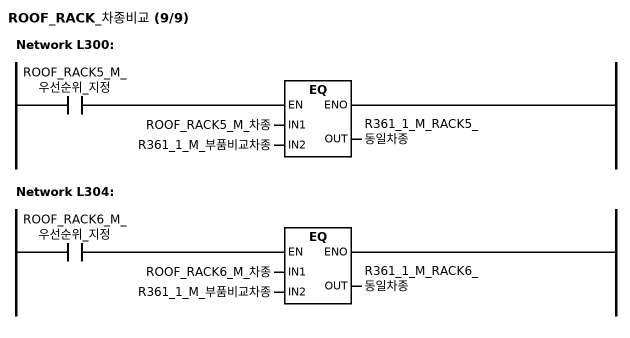
(* [picture p96: ROOF_RACK_차종비교 rungs L300-L304] *)
(* Rung L300 *)
IF ROOF_RACK5_M_우선순위_지정 THEN R361_1_M_RACK5_동일차종 := ROOF_RACK5_M_차종 = R361_1_M_부품비교차종; END_IF;
(* Rung L304 *)
IF ROOF_RACK6_M_우선순위_지정 THEN R361_1_M_RACK6_동일차종 := ROOF_RACK6_M_차종 = R361_1_M_부품비교차종; END_IF;
END_PROGRAM

PROGRAM ROOF_RACK_로보트 (* task: 스캔 프로그램 *)
VAR_EXTERNAL RETAIN
    ALWAYS_OFF : BOOL; (* AT %MW3.0 *) (* 항시 OFF *)
    ALWAYS_ON : BOOL; (* AT %MW3.1 *) (* 항시 ON *)
    MCP_M_부저_정지 : BOOL; (* AT %MW350.5 *) (* MCP 부저정지 *)
    MCP_M_비상정지 : BOOL; (* AT %MW350.7 *) (* MCP 비상정지 이상 *)
    R361_1_M_RACK3_동일차종 : BOOL; (* AT %MW1565.2 *)
    R361_1_M_RACK3_프로그램_OK : BOOL; (* AT %MW1563.2 *)
    R361_1_M_RACK4_동일차종 : BOOL; (* AT %MW1565.3 *)
    R361_1_M_RACK4_프로그램_OK : BOOL; (* AT %MW1563.3 *)
    R361_1_M_RACK5_동일차종 : BOOL; (* AT %MW1565.4 *)
    R361_1_M_RACK5_프로그램_OK : BOOL; (* AT %MW1563.4 *)
    R361_1_M_RACK6_동일차종 : BOOL; (* AT %MW1565.5 *)
    R361_1_M_RACK6_프로그램_OK : BOOL; (* AT %MW1563.5 *)
    R361_1_M_기동_랙번호 : WORD; (* AT %MW1534 *)
    R361_1_M_차종1_AX : BOOL; (* AT %MW10001.0 *) (* R361 1 M 차종1 AX *)
    R361_1_M_차종6_썬루프 : BOOL; (* AT %MW10003.4 *) (* R361 1 M 차종6 썬루프 *)
    R361_1_M_차종6_일반루프 : BOOL; (* AT %MW10003.3 *) (* R361 1 M 차종6 일반루프 *)
    R361_1_M_차종_OPT1_R_RACK_무 : BOOL; (* AT %MW10005.3 *) (* R361 1 M 차종 OPT1 R RACK 무 *)
    R361_1_M_차종_OPT1_R_RACK_유 : BOOL; (* AT %MW10005.2 *) (* R361 1 M 차종 OPT1 R RACK 유 *)
    R361_1_M_차종_유 : BOOL; (* AT %MW1502.0 *)
    R361_2_M_RACK1_동일차종 : BOOL; (* AT %MW1565.0 *)
    R361_2_M_RACK1_프로그램_OK : BOOL; (* AT %MW1563.0 *)
    R361_2_M_RACK2_동일차종 : BOOL; (* AT %MW1565.1 *)
    R361_2_M_RACK2_프로그램_OK : BOOL; (* AT %MW1563.1 *)
    R361_2_M_기동_랙번호 : WORD; (* AT %MW1535 *)
    R361_2_M_차종1_AX : BOOL; (* AT %MW10021.0 *) (* R361 2 M 차종1 AX *)
    R361_2_M_차종6_썬루프 : BOOL; (* AT %MW10023.4 *) (* R361 2 M 차종6 썬루프 *)
    R361_2_M_차종6_일반루프 : BOOL; (* AT %MW10023.3 *) (* R361 2 M 차종6 일반루프 *)
    R361_2_M_차종_OPT1_R_RACK_유 : BOOL; (* AT %MW10025.2 *) (* R361 2 M 차종 OPT1 R RACK 유 *)
    R361_2_M_차종_유 : BOOL; (* AT %MW1502.2 *)
    ROOF_RACK1_M_PLT_이상 : BOOL; (* AT %MW1514.0 *)
    ROOF_RACK1_M_랙감지_유 : BOOL; (* AT %MW1501.0 *)
    ROOF_RACK1_M_막장감지_유 : BOOL; (* AT %MW1503.0 *)
    ROOF_RACK1_M_우선순위_지정 : BOOL; (* AT %MW1564.0 *)
    ROOF_RACK1_M_차종_무 : BOOL; (* AT %MW1540.1 *)
    ROOF_RACK1_M_카운트_리셋요구_SET : BOOL; (* AT %MW1566.0 *)
    ROOF_RACK2_M_PLT_이상 : BOOL; (* AT %MW1514.1 *)
    ROOF_RACK2_M_랙감지_유 : BOOL; (* AT %MW1501.2 *)
    ROOF_RACK2_M_막장감지_유 : BOOL; (* AT %MW1503.2 *)
    ROOF_RACK2_M_우선순위_지정 : BOOL; (* AT %MW1564.1 *)
    ROOF_RACK2_M_차종_무 : BOOL; (* AT %MW1540.3 *)
    ROOF_RACK2_M_카운트_리셋요구_SET : BOOL; (* AT %MW1566.1 *)
    ROOF_RACK3_M_PLT_이상 : BOOL; (* AT %MW1514.2 *)
    ROOF_RACK3_M_랙감지_유 : BOOL; (* AT %MW1501.4 *)
    ROOF_RACK3_M_막장감지_유 : BOOL; (* AT %MW1503.4 *)
    ROOF_RACK3_M_우선순위_지정 : BOOL; (* AT %MW1564.2 *)
    ROOF_RACK3_M_차종_무 : BOOL; (* AT %MW1540.5 *)
    ROOF_RACK3_M_카운트_리셋요구_SET : BOOL; (* AT %MW1566.2 *)
    ROOF_RACK4_M_PLT_이상 : BOOL; (* AT %MW1514.3 *)
    ROOF_RACK4_M_랙감지_유 : BOOL; (* AT %MW1501.6 *)
    ROOF_RACK4_M_막장감지_유 : BOOL; (* AT %MW1503.6 *)
    ROOF_RACK4_M_우선순위_지정 : BOOL; (* AT %MW1564.3 *)
    ROOF_RACK4_M_차종_무 : BOOL; (* AT %MW1540.7 *)
    ROOF_RACK4_M_카운트_리셋요구_SET : BOOL; (* AT %MW1566.3 *)
    ROOF_RACK5_M_PLT_이상 : BOOL; (* AT %MW1514.4 *)
    ROOF_RACK5_M_랙감지_유 : BOOL; (* AT %MW1501.8 *)
    ROOF_RACK5_M_막장감지_유 : BOOL; (* AT %MW1503.8 *)
    ROOF_RACK5_M_우선순위_지정 : BOOL; (* AT %MW1564.4 *)
    ROOF_RACK5_M_차종_무 : BOOL; (* AT %MW1540.9 *)
    ROOF_RACK5_M_카운트_리셋요구_SET : BOOL; (* AT %MW1566.4 *)
    ROOF_RACK6_M_PLT_이상 : BOOL; (* AT %MW1514.5 *)
    ROOF_RACK6_M_랙감지_유 : BOOL; (* AT %MW1501.10 *)
    ROOF_RACK6_M_막장감지_유 : BOOL; (* AT %MW1503.10 *)
    ROOF_RACK6_M_우선순위_지정 : BOOL; (* AT %MW1564.5 *)
    ROOF_RACK6_M_차종_무 : BOOL; (* AT %MW1540.11 *)
    ROOF_RACK6_M_카운트_리셋요구_SET : BOOL; (* AT %MW1566.5 *)
    ROOF_RACK_M_수동모드 : BOOL; (* AT %MW1500.3 *)
    ROOF_RACK_M_자동_START : BOOL; (* AT %MW1500.5 *)
    ROOF_RACK_M_자동_운전중 : BOOL; (* AT %MW1500.4 *)
    ROOF_RACK_M_작업완료_SET_PLS : BOOL; (* AT %MW1500.8 *)
    ROOF_RACK_M_작업완료_리셋_PLS : BOOL; (* AT %MW1500.9 *)
    ROOF_RACK_M_총괄_이상 : BOOL; (* AT %MW1509.0 *)
    S364_M_R361_2_로딩완료 : BOOL; (* AT %MW2001.2 *)
    S364_M_공정_제품감지_무 : BOOL; (* AT %MW2002.5 *) (* S364_M_공정_제품감지_무 *)
    S364_M_공정_제품감지_유 : BOOL; (* AT %MW2002.4 *) (* S364_M_공정_제품감지_유 *)
    S364_M_공정_차종_AX : BOOL; (* AT %MW2002.3 *) (* S364_M_공정_차종_AX *)
    S364_M_공정_차종_무 : BOOL; (* AT %MW2002.1 *) (* S364_M_공정_차종_무 *)
    S364_M_공정_차종_유 : BOOL; (* AT %MW2002.0 *) (* S364_M_공정_차종_유 *)
    S364_M_자동_START : BOOL; (* AT %MW2000.5 *) (* S364 자동운전중 *)
    S364_M_자동_운전중 : BOOL; (* AT %MW2000.4 *) (* S364 자동운전중 *)
    S364_M_작업_완료 : BOOL; (* AT %MW2001.0 *) (* S364_M_작업_완료 *)
    S364_M_총괄_이상 : BOOL; (* AT %MW2009.0 *) (* S364_M_총괄_이상 *)
    S365_M_R361_1_안착완료 : BOOL; (* AT %MW2501.1 *)
    S365_M_공정_제품감지_무 : BOOL; (* AT %MW2501.4 *) (* S365_M_공정_제품감지_무 *)
    S365_M_공정_제품감지_유 : BOOL; (* AT %MW2501.3 *) (* S365_M_공정_제품감지_유 *)
    S365_M_공정_차종_무 : BOOL; (* AT %MW2502.1 *) (* S365_M_공정_차종_무 *)
    S365_M_공정_차종_유 : BOOL; (* AT %MW2502.0 *) (* S365_M_공정_차종_유 *)
    S365_M_작업_완료 : BOOL; (* AT %MW2501.0 *) (* S365_M_작업_완료 *)
    S366_M_R361_1_ROOF_로딩완료 : BOOL; (* AT %MW3001.2 *)
    S366_M_R361_1_동일차종_OK : BOOL; (* AT %MW3005.8 *)
    S366_M_R363_2_RAIL_로딩완료 : BOOL; (* AT %MW3001.1 *)
    S366_M_ROOF_로딩가능 : BOOL; (* AT %MW3004.9 *)
    S366_M_공정_FRT_PNL_제품감지_무 : BOOL; (* AT %MW3002.13 *)
    S366_M_공정_RR_PNL_제품감지_무 : BOOL; (* AT %MW3002.15 *)
    S366_M_공정_제품감지_유 : BOOL; (* AT %MW3001.6 *) (* S366_M_공정_제품감지_유 *)
    S366_M_작업_완료 : BOOL; (* AT %MW3001.0 *) (* S366_M_작업_완료 *)
    S367_M_R361_1_로딩가능 : BOOL; (* AT %MW3504.8 *)
    S367_M_공정_제품감지_무 : BOOL; (* AT %MW3501.6 *) (* S367_M_공정_제품감지_무 *)
    S367_M_공정_차종_무 : BOOL; (* AT %MW3502.1 *) (* S367_M_공정_차종_무 *)
    S367_M_작업_완료 : BOOL; (* AT %MW3501.0 *) (* S367_M_작업_완료 *)
    전체_M_GATE_비상정지_정상 : BOOL; (* AT %MW308.4 *) (* 전체 M GATE 비상정지 정상 *)
    전체_M_GATE_자동기동 : BOOL; (* AT %MW308.1 *) (* 전체_M_자동_운전 *)
    전체_M_운전준비_보조 : BOOL; (* AT %MW308.5 *)
    전체_M_이상_리셋 : BOOL; (* AT %MW308.2 *) (* ALL공정 PB 이상리셋 *)
    전체_공정_M_총괄_비상정지_정상 : BOOL; (* AT %MW304.1 *)
END_VAR
VAR
    INST : TON;
    INST1 : FB494_Robot_Hyundai_HMMI_v1;
    INST2 : FB494_Robot_Hyundai_HMMI_v1;
    INST3 : TON;
    INST4 : TON;
    INST5 : TON;
    INST6 : TON;
    INST7 : TON;
    INST8 : TON;
    INST9 : TON;
    R361_1_M_RB_PROG_NO : INT;
    R361_2_M_RB_PROG_NO : INT;
    로보트제외 : BOOL;
END_VAR
VAR_EXTERNAL
    MCP_PBL_운전준비_ON : BOOL; (* AT %MW87630.0 *) (* MCP_PBL_운전준비_ON *)
    R361_1_I_RB_INPUT : ARRAY[0..3] OF WORD; (* AT %MW84010 *) (* R361_1_I_RB_INPUT *)
    R361_1_I_RB__PLT_카운터리셋완료 : BOOL; (* AT %MW84013.10 *) (* R361_1_I_RB__PLT_카운터리셋완료 *)
    R361_1_I_RB_상호인터록_INT1 : BOOL; (* AT %MW84013.0 *) (* R361_1_I_RB_상호인터록_INT1 *)
    R361_1_M_I_RB_1차_작업완료 : BOOL; (* AT %MW20011.2 *) (* R361_1_M_I_RB_1차_작업완료 *)
    R361_1_M_I_RB_2차_작업완료 : BOOL; (* AT %MW20011.3 *) (* R361_1_M_I_RB_2차_작업완료 *)
    R361_1_M_I_RB_3차_작업완료 : BOOL; (* AT %MW20011.4 *) (* R361_1_M_I_RB_3차_작업완료 *)
    R361_1_M_I_RB_4차_작업완료 : BOOL; (* AT %MW20011.5 *) (* R361_1_M_I_RB_4차_작업완료 *)
    R361_1_M_I_RB_5차_작업완료 : BOOL; (* AT %MW20011.6 *) (* R361_1_M_I_RB_5차_작업완료 *)
    R361_1_M_I_RB_6차_작업완료 : BOOL; (* AT %MW20011.7 *) (* R361_1_M_I_RB_6차_작업완료 *)
    R361_1_M_I_RB_7차_작업완료 : BOOL; (* AT %MW20011.8 *) (* R361_1_M_I_RB_7차_작업완료 *)
    R361_1_M_I_RB_PAUSE_보조 : BOOL; (* AT %MW20010.5 *) (* R361_1_M_I_RB_PAUSE_보조 *)
    R361_1_M_I_RB_PLC_RUN_CHK_이상 : BOOL; (* AT %MW20010.7 *) (* R361_1_M_I_RB_PLC_RUN_CHK_이상 *)
    R361_1_M_I_RB_간섭무_1 : BOOL; (* AT %MW20012.0 *) (* R361_1_M_I_RB_간섭무_1 *)
    R361_1_M_I_RB_간섭무_10 : BOOL; (* AT %MW20012.9 *) (* R361_1_M_I_RB_간섭무_10 *)
    R361_1_M_I_RB_간섭무_11 : BOOL; (* AT %MW20012.10 *) (* R361_1_M_I_RB_간섭무_11 *)
    R361_1_M_I_RB_간섭무_12 : BOOL; (* AT %MW20012.11 *) (* R361_1_M_I_RB_간섭무_12 *)
    R361_1_M_I_RB_간섭무_2 : BOOL; (* AT %MW20012.1 *) (* R361_1_M_I_RB_간섭무_2 *)
    R361_1_M_I_RB_간섭무_3 : BOOL; (* AT %MW20012.2 *) (* R361_1_M_I_RB_간섭무_3 *)
    R361_1_M_I_RB_간섭무_4 : BOOL; (* AT %MW20012.3 *) (* R361_1_M_I_RB_간섭무_4 *)
    R361_1_M_I_RB_간섭무_5 : BOOL; (* AT %MW20012.4 *) (* R361_1_M_I_RB_간섭무_5 *)
    R361_1_M_I_RB_간섭무_6 : BOOL; (* AT %MW20012.5 *) (* R361_1_M_I_RB_간섭무_6 *)
    R361_1_M_I_RB_간섭무_7 : BOOL; (* AT %MW20012.6 *) (* R361_1_M_I_RB_간섭무_7 *)
    R361_1_M_I_RB_간섭무_8 : BOOL; (* AT %MW20012.7 *) (* R361_1_M_I_RB_간섭무_8 *)
    R361_1_M_I_RB_간섭무_9 : BOOL; (* AT %MW20012.8 *) (* R361_1_M_I_RB_간섭무_9 *)
    R361_1_M_I_RB_비상정지 : BOOL; (* AT %MW20010.4 *) (* R361_1_M_I_RB_비상정지 *)
    R361_1_M_I_RB_운전준비 : BOOL; (* AT %MW20010.0 *) (* R361_1_M_I_RB_운전준비 *)
    R361_1_M_I_RB_원위치 : BOOL; (* AT %MW20010.3 *) (* R361_1_M_I_RB_원위치 *)
    R361_1_M_I_RB_이상 : BOOL; (* AT %MW20010.2 *) (* R361_1_M_I_RB_이상 *)
    R361_1_M_I_RB_자동 : BOOL; (* AT %MW20010.1 *) (* R361_1_M_I_RB_자동 *)
    R361_1_M_I_RB_최종작업완료 : BOOL; (* AT %MW20011.0 *) (* R361_1_M_I_RB_최종작업완료 *)
    R361_1_M_I_RB_프로그램_이상 : BOOL; (* AT %MW20010.6 *) (* R361_1_M_I_RB_프로그램_이상 *)
    R361_1_M_O_RB_1_CYCLE_SET : BOOL; (* AT %MW21010.3 *) (* R361_1_M_O_RB_1_CYCLE_SET *)
    R361_1_M_O_RB_1차_작업완료_리셋 : BOOL; (* AT %MW21012.0 *) (* R361_1_M_O_RB_1차_작업완료_리셋 *)
    R361_1_M_O_RB_2차_작업완료_리셋 : BOOL; (* AT %MW21012.1 *) (* R361_1_M_O_RB_2차_작업완료_리셋 *)
    R361_1_M_O_RB_2차_진입OK : BOOL; (* AT %MW21011.8 *) (* R361_1_M_O_RB_2차_진입OK *)
    R361_1_M_O_RB_3차_작업완료_리셋 : BOOL; (* AT %MW21012.2 *) (* R361_1_M_O_RB_3차_작업완료_리셋 *)
    R361_1_M_O_RB_3차_진입OK : BOOL; (* AT %MW21011.9 *) (* R361_1_M_O_RB_3차_진입OK *)
    R361_1_M_O_RB_4차_작업완료_리셋 : BOOL; (* AT %MW21012.3 *) (* R361_1_M_O_RB_4차_작업완료_리셋 *)
    R361_1_M_O_RB_4차_진입OK : BOOL; (* AT %MW21011.10 *) (* R361_1_M_O_RB_4차_진입OK *)
    R361_1_M_O_RB_5차_작업완료_리셋 : BOOL; (* AT %MW21012.4 *) (* R361_1_M_O_RB_5차_작업완료_리셋 *)
    R361_1_M_O_RB_5차_진입OK : BOOL; (* AT %MW21011.11 *) (* R361_1_M_O_RB_5차_진입OK *)
    R361_1_M_O_RB_6차_작업완료_리셋 : BOOL; (* AT %MW21012.5 *) (* R361_1_M_O_RB_6차_작업완료_리셋 *)
    R361_1_M_O_RB_6차_진입OK : BOOL; (* AT %MW21011.12 *) (* R361_1_M_O_RB_6차_진입OK *)
    R361_1_M_O_RB_7차_작업완료_리셋 : BOOL; (* AT %MW21012.6 *) (* R361_1_M_O_RB_7차_작업완료_리셋 *)
    R361_1_M_O_RB_7차_진입OK : BOOL; (* AT %MW21011.13 *) (* R361_1_M_O_RB_7차_진입OK *)
    R361_1_M_O_RB_ATD_OK : BOOL; (* AT %MW21010.6 *) (* R361_1_M_O_RB_ATD_OK *)
    R361_1_M_O_RB_PLT_10_진입OK : BOOL; (* AT %MW21013.10 *) (* R361_1_M_O_RB_PLT_10_진입OK *)
    R361_1_M_O_RB_PLT_11_진입OK : BOOL; (* AT %MW21013.11 *) (* R361_1_M_O_RB_PLT_11_진입OK *)
    R361_1_M_O_RB_PLT_12_진입OK : BOOL; (* AT %MW21013.12 *) (* R361_1_M_O_RB_PLT_12_진입OK *)
    R361_1_M_O_RB_PLT_1_진입OK : BOOL; (* AT %MW21013.1 *) (* R361_1_M_O_RB_PLT_1_진입OK *)
    R361_1_M_O_RB_PLT_2_진입OK : BOOL; (* AT %MW21013.2 *) (* R361_1_M_O_RB_PLT_2_진입OK *)
    R361_1_M_O_RB_PLT_3_진입OK : BOOL; (* AT %MW21013.3 *) (* R361_1_M_O_RB_PLT_3_진입OK *)
    R361_1_M_O_RB_PLT_4_진입OK : BOOL; (* AT %MW21013.4 *) (* R361_1_M_O_RB_PLT_4_진입OK *)
    R361_1_M_O_RB_PLT_5_진입OK : BOOL; (* AT %MW21013.5 *) (* R361_1_M_O_RB_PLT_5_진입OK *)
    R361_1_M_O_RB_PLT_6_진입OK : BOOL; (* AT %MW21013.6 *) (* R361_1_M_O_RB_PLT_6_진입OK *)
    R361_1_M_O_RB_PLT_7_진입OK : BOOL; (* AT %MW21013.7 *) (* R361_1_M_O_RB_PLT_7_진입OK *)
    R361_1_M_O_RB_PLT_8_진입OK : BOOL; (* AT %MW21013.8 *) (* R361_1_M_O_RB_PLT_8_진입OK *)
    R361_1_M_O_RB_PLT_9_진입OK : BOOL; (* AT %MW21013.9 *) (* R361_1_M_O_RB_PLT_9_진입OK *)
    R361_1_M_O_RB_PLT_카운터리셋_보조 : BOOL; (* AT %MW21010.10 *) (* R361_1_M_O_RB_PLT_카운터리셋_보조 *)
    R361_1_M_O_RB_PROG_NO : WORD; (* AT %MW21014 *)
    R361_1_M_O_RB_RESTART_OK : BOOL; (* AT %MW21010.2 *) (* R361_1_M_O_RB_RESTART_OK *)
    R361_1_M_O_RB_START_OK : BOOL; (* AT %MW21010.0 *) (* R361_1_M_O_RB_START_OK *)
    R361_1_M_O_RB_TEST_MODE_5000회 : BOOL; (* AT %MW21010.12 *) (* R361_1_M_O_RB_TEST_MODE_5000회 *)
    R361_1_M_O_RB_TIP_교체_시작 : BOOL; (* AT %MW21010.7 *) (* R361_1_M_O_RB_TIP_교체_시작 *)
    R361_1_M_O_RB_TIP_교체_완료 : BOOL; (* AT %MW21010.8 *) (* R361_1_M_O_RB_TIP_교체_완료 *)
    R361_1_M_O_RB_VIP_MODE : BOOL; (* AT %MW21010.11 *) (* R361_1_M_O_RB_VIP_MODE *)
    R361_1_M_O_RB_냉각수_차단_요청 : BOOL; (* AT %MW21010.9 *) (* R361_1_M_O_RB_냉각수_차단_요청 *)
    R361_1_M_O_RB_진입OK_AX차종 : BOOL; (* AT %MW21011.0 *) (* R361_1_M_O_RB_진입OK_AX차종 *)
    R361_1_M_O_RB_진입OK_B차종 : BOOL; (* AT %MW21011.1 *) (* R361_1_M_O_RB_진입OK_B차종 *)
    R361_1_M_O_RB_진입OK_C차종 : BOOL; (* AT %MW21011.2 *) (* R361_1_M_O_RB_진입OK_C차종 *)
    R361_1_M_O_RB_진입OK_D차종 : BOOL; (* AT %MW21011.3 *) (* R361_1_M_O_RB_진입OK_D차종 *)
    R361_1_M_O_RB_진입OK_E차종 : BOOL; (* AT %MW21011.4 *) (* R361_1_M_O_RB_진입OK_E차종 *)
    R361_1_M_O_RB_진입OK_F차종 : BOOL; (* AT %MW21011.5 *) (* R361_1_M_O_RB_진입OK_F차종 *)
    R361_1_M_O_RB_진입OK_G차종 : BOOL; (* AT %MW21011.6 *) (* R361_1_M_O_RB_진입OK_G차종 *)
    R361_1_M_O_RB_진입OK_H차종 : BOOL; (* AT %MW21011.7 *) (* R361_1_M_O_RB_진입OK_H차종 *)
    R361_1_M_O_RB_최종_작업완료_리셋 : BOOL; (* AT %MW21010.5 *) (* R361_1_M_O_RB_최종_작업완료_리셋 *)
    R361_1_M_O_RB_프로그램_OK : BOOL; (* AT %MW21010.1 *) (* R361_1_M_O_RB_프로그램_OK *)
    R361_1_O_RB_OUTPUT : ARRAY[0..3] OF WORD; (* AT %MW94010 *) (* R361_1_O_RB_OUTPUT *)
    R361_1_O_RB_PLT_카운터_리셋_요구 : BOOL; (* AT %MW94013.10 *) (* R361_1_O_RB_PLT_카운터_리셋_요구 *)
    R361_2_I_RB_INPUT : ARRAY[0..3] OF WORD; (* AT %MW84020 *) (* R361_2_I_RB_INPUT *)
    R361_2_I_RB_PLT_최종UNLOAD_완료 : BOOL; (* AT %MW84023.12 *) (* R361_2_I_RB_PLT_최종UNLOAD_완료 *)
    R361_2_I_RB__PLT_카운터리셋완료 : BOOL; (* AT %MW84023.10 *) (* R361_2_I_RB__PLT_카운터리셋완료 *)
    R361_2_I_RB_상호인터록_INT1 : BOOL; (* AT %MW84023.0 *) (* R361_2_I_RB_상호인터록_INT1 *)
    R361_2_M_I_RB_1차_작업완료 : BOOL; (* AT %MW20021.2 *) (* R361_2_M_I_RB_1차_작업완료 *)
    R361_2_M_I_RB_2차_작업완료 : BOOL; (* AT %MW20021.3 *) (* R361_2_M_I_RB_2차_작업완료 *)
    R361_2_M_I_RB_3차_작업완료 : BOOL; (* AT %MW20021.4 *) (* R361_2_M_I_RB_3차_작업완료 *)
    R361_2_M_I_RB_4차_작업완료 : BOOL; (* AT %MW20021.5 *) (* R361_2_M_I_RB_4차_작업완료 *)
    R361_2_M_I_RB_5차_작업완료 : BOOL; (* AT %MW20021.6 *) (* R361_2_M_I_RB_5차_작업완료 *)
    R361_2_M_I_RB_6차_작업완료 : BOOL; (* AT %MW20021.7 *) (* R361_2_M_I_RB_6차_작업완료 *)
    R361_2_M_I_RB_7차_작업완료 : BOOL; (* AT %MW20021.8 *) (* R361_2_M_I_RB_7차_작업완료 *)
    R361_2_M_I_RB_PAUSE_보조 : BOOL; (* AT %MW20020.5 *) (* R361_2_M_I_RB_PAUSE_보조 *)
    R361_2_M_I_RB_PLC_RUN_CHK_이상 : BOOL; (* AT %MW20020.7 *) (* R361_2_M_I_RB_PLC_RUN_CHK_이상 *)
    R361_2_M_I_RB_간섭무_1 : BOOL; (* AT %MW20022.0 *) (* R361_2_M_I_RB_간섭무_1 *)
    R361_2_M_I_RB_간섭무_10 : BOOL; (* AT %MW20022.9 *) (* R361_2_M_I_RB_간섭무_10 *)
    R361_2_M_I_RB_간섭무_11 : BOOL; (* AT %MW20022.10 *) (* R361_2_M_I_RB_간섭무_11 *)
    R361_2_M_I_RB_간섭무_12 : BOOL; (* AT %MW20022.11 *) (* R361_2_M_I_RB_간섭무_12 *)
    R361_2_M_I_RB_간섭무_2 : BOOL; (* AT %MW20022.1 *) (* R361_2_M_I_RB_간섭무_2 *)
    R361_2_M_I_RB_간섭무_3 : BOOL; (* AT %MW20022.2 *) (* R361_2_M_I_RB_간섭무_3 *)
    R361_2_M_I_RB_간섭무_4 : BOOL; (* AT %MW20022.3 *) (* R361_2_M_I_RB_간섭무_4 *)
    R361_2_M_I_RB_간섭무_5 : BOOL; (* AT %MW20022.4 *) (* R361_2_M_I_RB_간섭무_5 *)
    R361_2_M_I_RB_간섭무_6 : BOOL; (* AT %MW20022.5 *) (* R361_2_M_I_RB_간섭무_6 *)
    R361_2_M_I_RB_간섭무_7 : BOOL; (* AT %MW20022.6 *) (* R361_2_M_I_RB_간섭무_7 *)
    R361_2_M_I_RB_간섭무_8 : BOOL; (* AT %MW20022.7 *) (* R361_2_M_I_RB_간섭무_8 *)
    R361_2_M_I_RB_간섭무_9 : BOOL; (* AT %MW20022.8 *) (* R361_2_M_I_RB_간섭무_9 *)
    R361_2_M_I_RB_비상정지 : BOOL; (* AT %MW20020.4 *) (* R361_2_M_I_RB_비상정지 *)
    R361_2_M_I_RB_운전준비 : BOOL; (* AT %MW20020.0 *) (* R361_2_M_I_RB_운전준비 *)
    R361_2_M_I_RB_원위치 : BOOL; (* AT %MW20020.3 *) (* R361_2_M_I_RB_원위치 *)
    R361_2_M_I_RB_이상 : BOOL; (* AT %MW20020.2 *) (* R361_2_M_I_RB_이상 *)
    R361_2_M_I_RB_자동 : BOOL; (* AT %MW20020.1 *) (* R361_2_M_I_RB_자동 *)
    R361_2_M_I_RB_최종작업완료 : BOOL; (* AT %MW20021.0 *) (* R361_2_M_I_RB_최종작업완료 *)
    R361_2_M_I_RB_프로그램_이상 : BOOL; (* AT %MW20020.6 *) (* R361_2_M_I_RB_프로그램_이상 *)
    R361_2_M_O_RB_1_CYCLE_SET : BOOL; (* AT %MW21020.3 *) (* R361_2_M_O_RB_1_CYCLE_SET *)
    R361_2_M_O_RB_1차_작업완료_리셋 : BOOL; (* AT %MW21022.0 *) (* R361_2_M_O_RB_1차_작업완료_리셋 *)
    R361_2_M_O_RB_2차_작업완료_리셋 : BOOL; (* AT %MW21022.1 *) (* R361_2_M_O_RB_2차_작업완료_리셋 *)
    R361_2_M_O_RB_2차_진입OK : BOOL; (* AT %MW21021.8 *) (* R361_2_M_O_RB_2차_진입OK *)
    R361_2_M_O_RB_3차_작업완료_리셋 : BOOL; (* AT %MW21022.2 *) (* R361_2_M_O_RB_3차_작업완료_리셋 *)
    R361_2_M_O_RB_3차_진입OK : BOOL; (* AT %MW21021.9 *) (* R361_2_M_O_RB_3차_진입OK *)
    R361_2_M_O_RB_4차_작업완료_리셋 : BOOL; (* AT %MW21022.3 *) (* R361_2_M_O_RB_4차_작업완료_리셋 *)
    R361_2_M_O_RB_4차_진입OK : BOOL; (* AT %MW21021.10 *) (* R361_2_M_O_RB_4차_진입OK *)
    R361_2_M_O_RB_5차_작업완료_리셋 : BOOL; (* AT %MW21022.4 *) (* R361_2_M_O_RB_5차_작업완료_리셋 *)
    R361_2_M_O_RB_5차_진입OK : BOOL; (* AT %MW21021.11 *) (* R361_2_M_O_RB_5차_진입OK *)
    R361_2_M_O_RB_6차_작업완료_리셋 : BOOL; (* AT %MW21022.5 *) (* R361_2_M_O_RB_6차_작업완료_리셋 *)
    R361_2_M_O_RB_6차_진입OK : BOOL; (* AT %MW21021.12 *) (* R361_2_M_O_RB_6차_진입OK *)
    R361_2_M_O_RB_7차_작업완료_리셋 : BOOL; (* AT %MW21022.6 *) (* R361_2_M_O_RB_7차_작업완료_리셋 *)
    R361_2_M_O_RB_7차_진입OK : BOOL; (* AT %MW21021.13 *) (* R361_2_M_O_RB_7차_진입OK *)
    R361_2_M_O_RB_ATD_OK : BOOL; (* AT %MW21020.6 *) (* R361_2_M_O_RB_ATD_OK *)
    R361_2_M_O_RB_PLT_10_진입OK : BOOL; (* AT %MW21023.10 *) (* R361_2_M_O_RB_PLT_10_진입OK *)
    R361_2_M_O_RB_PLT_11_진입OK : BOOL; (* AT %MW21023.11 *) (* R361_2_M_O_RB_PLT_11_진입OK *)
    R361_2_M_O_RB_PLT_12_진입OK : BOOL; (* AT %MW21023.12 *) (* R361_2_M_O_RB_PLT_12_진입OK *)
    R361_2_M_O_RB_PLT_1_진입OK : BOOL; (* AT %MW21023.1 *) (* R361_2_M_O_RB_PLT_1_진입OK *)
    R361_2_M_O_RB_PLT_2_진입OK : BOOL; (* AT %MW21023.2 *) (* R361_2_M_O_RB_PLT_2_진입OK *)
    R361_2_M_O_RB_PLT_3_진입OK : BOOL; (* AT %MW21023.3 *) (* R361_2_M_O_RB_PLT_3_진입OK *)
    R361_2_M_O_RB_PLT_4_진입OK : BOOL; (* AT %MW21023.4 *) (* R361_2_M_O_RB_PLT_4_진입OK *)
    R361_2_M_O_RB_PLT_5_진입OK : BOOL; (* AT %MW21023.5 *) (* R361_2_M_O_RB_PLT_5_진입OK *)
    R361_2_M_O_RB_PLT_6_진입OK : BOOL; (* AT %MW21023.6 *) (* R361_2_M_O_RB_PLT_6_진입OK *)
    R361_2_M_O_RB_PLT_7_진입OK : BOOL; (* AT %MW21023.7 *) (* R361_2_M_O_RB_PLT_7_진입OK *)
    R361_2_M_O_RB_PLT_8_진입OK : BOOL; (* AT %MW21023.8 *) (* R361_2_M_O_RB_PLT_8_진입OK *)
    R361_2_M_O_RB_PLT_9_진입OK : BOOL; (* AT %MW21023.9 *) (* R361_2_M_O_RB_PLT_9_진입OK *)
    R361_2_M_O_RB_PLT_카운터리셋_보조 : BOOL; (* AT %MW21020.10 *) (* R361_2_M_O_RB_PLT_카운터리셋_보조 *)
    R361_2_M_O_RB_PROG_NO : WORD; (* AT %MW21024 *)
    R361_2_M_O_RB_RESTART_OK : BOOL; (* AT %MW21020.2 *) (* R361_2_M_O_RB_RESTART_OK *)
    R361_2_M_O_RB_START_OK : BOOL; (* AT %MW21020.0 *) (* R361_2_M_O_RB_START_OK *)
    R361_2_M_O_RB_TEST_MODE_5000회 : BOOL; (* AT %MW21020.12 *) (* R361_2_M_O_RB_TEST_MODE_5000회 *)
    R361_2_M_O_RB_TIP_교체_시작 : BOOL; (* AT %MW21020.7 *) (* R361_2_M_O_RB_TIP_교체_시작 *)
    R361_2_M_O_RB_TIP_교체_완료 : BOOL; (* AT %MW21020.8 *) (* R361_2_M_O_RB_TIP_교체_완료 *)
    R361_2_M_O_RB_VIP_MODE : BOOL; (* AT %MW21020.11 *) (* R361_2_M_O_RB_VIP_MODE *)
    R361_2_M_O_RB_냉각수_차단_요청 : BOOL; (* AT %MW21020.9 *) (* R361_2_M_O_RB_냉각수_차단_요청 *)
    R361_2_M_O_RB_진입OK_AX차종 : BOOL; (* AT %MW21021.0 *) (* R361_2_M_O_RB_진입OK_AX차종 *)
    R361_2_M_O_RB_진입OK_B차종 : BOOL; (* AT %MW21021.1 *) (* R361_2_M_O_RB_진입OK_B차종 *)
    R361_2_M_O_RB_진입OK_C차종 : BOOL; (* AT %MW21021.2 *) (* R361_2_M_O_RB_진입OK_C차종 *)
    R361_2_M_O_RB_진입OK_D차종 : BOOL; (* AT %MW21021.3 *) (* R361_2_M_O_RB_진입OK_D차종 *)
    R361_2_M_O_RB_진입OK_E차종 : BOOL; (* AT %MW21021.4 *) (* R361_2_M_O_RB_진입OK_E차종 *)
    R361_2_M_O_RB_진입OK_F차종 : BOOL; (* AT %MW21021.5 *) (* R361_2_M_O_RB_진입OK_F차종 *)
    R361_2_M_O_RB_진입OK_G차종 : BOOL; (* AT %MW21021.6 *) (* R361_2_M_O_RB_진입OK_G차종 *)
    R361_2_M_O_RB_진입OK_H차종 : BOOL; (* AT %MW21021.7 *) (* R361_2_M_O_RB_진입OK_H차종 *)
    R361_2_M_O_RB_최종_작업완료_리셋 : BOOL; (* AT %MW21020.5 *) (* R361_2_M_O_RB_최종_작업완료_리셋 *)
    R361_2_M_O_RB_프로그램_OK : BOOL; (* AT %MW21020.1 *) (* R361_2_M_O_RB_프로그램_OK *)
    R361_2_O_RB_OUTPUT : ARRAY[0..3] OF WORD; (* AT %MW94020 *) (* R361_2_O_RB_OUTPUT *)
    R361_2_O_RB_PLT_카운터_리셋_요구 : BOOL; (* AT %MW94023.10 *) (* R361_2_O_RB_PLT_카운터_리셋_요구 *)
    R364_1_M_O_RB_6차_작업완료_리셋 : BOOL; (* AT %MW21052.5 *) (* R364_1_M_O_RB_6차_작업완료_리셋 *)
    R364_1_M_O_RB_최종_작업완료_리셋 : BOOL; (* AT %MW21050.5 *) (* R364_1_M_O_RB_최종_작업완료_리셋 *)
END_VAR
(* ladder body could not be read *)
END_PROGRAM

PROGRAM ROOF_RACK_이상 (* task: 스캔 프로그램 *)
VAR_EXTERNAL RETAIN
    ALWAYS_OFF : BOOL; (* AT %MW3.0 *) (* 항시 OFF *)
    R361_1_M_NODE_4_01_통신_이상 : BOOL; (* AT %MW1524.8 *)
    R361_1_M_RACK3_프로그램_OK : BOOL; (* AT %MW1563.2 *)
    R361_1_M_RACK4_프로그램_OK : BOOL; (* AT %MW1563.3 *)
    R361_1_M_RACK5_프로그램_OK : BOOL; (* AT %MW1563.4 *)
    R361_1_M_RACK6_프로그램_OK : BOOL; (* AT %MW1563.5 *)
    R361_2_M_NODE_4_02_통신_이상 : BOOL; (* AT %MW1524.9 *)
    R361_2_M_RACK1_프로그램_OK : BOOL; (* AT %MW1563.0 *)
    R361_2_M_RACK2_프로그램_OK : BOOL; (* AT %MW1563.1 *)
    ROOF_RACK1_3_M_NODE_7_40_통신_이상 : BOOL; (* AT %MW1524.0 *)
    ROOF_RACK1_M_LC_이상 : BOOL; (* AT %MW1512.0 *)
    ROOF_RACK1_M_PLT_이상 : BOOL; (* AT %MW1514.0 *)
    ROOF_RACK1_M_랙감지_유 : BOOL; (* AT %MW1501.0 *)
    ROOF_RACK1_M_막장감지_무 : BOOL; (* AT %MW1503.1 *)
    ROOF_RACK1_M_막장감지_유 : BOOL; (* AT %MW1503.0 *)
    ROOF_RACK1_M_발목감지_이상 : BOOL; (* AT %MW1512.8 *)
    ROOF_RACK1_M_차종_무 : BOOL; (* AT %MW1540.1 *)
    ROOF_RACK1_M_차종_이상 : BOOL; (* AT %MW1515.0 *)
    ROOF_RACK2_M_LC_이상 : BOOL; (* AT %MW1512.1 *)
    ROOF_RACK2_M_PLT_이상 : BOOL; (* AT %MW1514.1 *)
    ROOF_RACK2_M_랙감지_유 : BOOL; (* AT %MW1501.2 *)
    ROOF_RACK2_M_막장감지_유 : BOOL; (* AT %MW1503.2 *)
    ROOF_RACK2_M_발목감지_이상 : BOOL; (* AT %MW1512.9 *)
    ROOF_RACK2_M_차종_무 : BOOL; (* AT %MW1540.3 *)
    ROOF_RACK2_M_차종_이상 : BOOL; (* AT %MW1515.1 *)
    ROOF_RACK3_M_LC_이상 : BOOL; (* AT %MW1512.2 *)
    ROOF_RACK3_M_PLT_이상 : BOOL; (* AT %MW1514.2 *)
    ROOF_RACK3_M_랙감지_유 : BOOL; (* AT %MW1501.4 *)
    ROOF_RACK3_M_막장감지_유 : BOOL; (* AT %MW1503.4 *)
    ROOF_RACK3_M_발목감지_이상 : BOOL; (* AT %MW1512.10 *)
    ROOF_RACK3_M_차종_무 : BOOL; (* AT %MW1540.5 *)
    ROOF_RACK3_M_차종_이상 : BOOL; (* AT %MW1515.2 *)
    ROOF_RACK4_6_M_NODE_7_45_통신_이상 : BOOL; (* AT %MW1524.1 *)
    ROOF_RACK4_M_LC_이상 : BOOL; (* AT %MW1512.3 *)
    ROOF_RACK4_M_PLT_이상 : BOOL; (* AT %MW1514.3 *)
    ROOF_RACK4_M_랙감지_유 : BOOL; (* AT %MW1501.6 *)
    ROOF_RACK4_M_막장감지_유 : BOOL; (* AT %MW1503.6 *)
    ROOF_RACK4_M_발목감지_이상 : BOOL; (* AT %MW1512.11 *)
    ROOF_RACK4_M_차종_무 : BOOL; (* AT %MW1540.7 *)
    ROOF_RACK4_M_차종_이상 : BOOL; (* AT %MW1515.3 *)
    ROOF_RACK5_M_LC_이상 : BOOL; (* AT %MW1512.4 *)
    ROOF_RACK5_M_PLT_이상 : BOOL; (* AT %MW1514.4 *)
    ROOF_RACK5_M_랙감지_유 : BOOL; (* AT %MW1501.8 *)
    ROOF_RACK5_M_막장감지_유 : BOOL; (* AT %MW1503.8 *)
    ROOF_RACK5_M_발목감지_이상 : BOOL; (* AT %MW1512.12 *)
    ROOF_RACK5_M_차종_무 : BOOL; (* AT %MW1540.9 *)
    ROOF_RACK5_M_차종_이상 : BOOL; (* AT %MW1515.4 *)
    ROOF_RACK6_M_LC_이상 : BOOL; (* AT %MW1512.5 *)
    ROOF_RACK6_M_PLT_이상 : BOOL; (* AT %MW1514.5 *)
    ROOF_RACK6_M_랙감지_유 : BOOL; (* AT %MW1501.10 *)
    ROOF_RACK6_M_막장감지_유 : BOOL; (* AT %MW1503.10 *)
    ROOF_RACK6_M_발목감지_이상 : BOOL; (* AT %MW1512.13 *)
    ROOF_RACK6_M_차종_무 : BOOL; (* AT %MW1540.11 *)
    ROOF_RACK6_M_차종_이상 : BOOL; (* AT %MW1515.5 *)
    ROOF_RACK_1_3_M_CP_이상 : BOOL; (* AT %MW1517.0 *)
    ROOF_RACK_4_6_M_CP_이상 : BOOL; (* AT %MW1517.1 *)
    ROOF_RACK_M_총괄_CP_이상 : BOOL; (* AT %MW1509.7 *)
    ROOF_RACK_M_총괄_CT_이상 : BOOL; (* AT %MW1510.4 *)
    ROOF_RACK_M_총괄_EOCR_이상 : BOOL; (* AT %MW1509.8 *)
    ROOF_RACK_M_총괄_INV_이상 : BOOL; (* AT %MW1509.9 *)
    ROOF_RACK_M_총괄_LS_이상 : BOOL; (* AT %MW1509.15 *)
    ROOF_RACK_M_총괄_MATCH_이상 : BOOL; (* AT %MW1510.0 *)
    ROOF_RACK_M_총괄_MC_이상 : BOOL; (* AT %MW1509.13 *)
    ROOF_RACK_M_총괄_MOTOR_이상 : BOOL; (* AT %MW1510.3 *)
    ROOF_RACK_M_총괄_NFB_이상 : BOOL; (* AT %MW1509.11 *)
    ROOF_RACK_M_총괄_ROBOT_이상 : BOOL; (* AT %MW1510.1 *)
    ROOF_RACK_M_총괄_SAFETY_이상 : BOOL; (* AT %MW1509.2 *)
    ROOF_RACK_M_총괄_공기압_이상 : BOOL; (* AT %MW1509.3 *)
    ROOF_RACK_M_총괄_사양_이상 : BOOL; (* AT %MW1509.6 *)
    ROOF_RACK_M_총괄_오버런_이상 : BOOL; (* AT %MW1509.12 *)
    ROOF_RACK_M_총괄_용접타점수_이상 : BOOL; (* AT %MW1510.2 *)
    ROOF_RACK_M_총괄_이상 : BOOL; (* AT %MW1509.0 *)
    ROOF_RACK_M_총괄_제품감지_이상 : BOOL; (* AT %MW1509.4 *)
    ROOF_RACK_M_총괄_차종_이상 : BOOL; (* AT %MW1509.5 *)
    ROOF_RACK_M_총괄_통신_이상 : BOOL; (* AT %MW1509.14 *)
    S362_M_총괄_CP_이상 : BOOL; (* AT %MW1009.7 *) (* S362 CP OFF 이상 *)
    S362_M_총괄_CT_이상 : BOOL; (* AT %MW1010.4 *) (* S362   TACK TIME 이상 *)
    S362_M_총괄_EOCR_이상 : BOOL; (* AT %MW1009.8 *) (* S362_M_총괄_EOCR_이상 *)
    S362_M_총괄_INV_이상 : BOOL; (* AT %MW1009.9 *) (* S362 인버터 이상 *)
    S362_M_총괄_LS_이상 : BOOL; (* AT %MW1009.15 *) (* S362 LS 이상 *)
    S362_M_총괄_MATCH_이상 : BOOL; (* AT %MW1010.0 *) (* S362 매트SW 이상 *)
    S362_M_총괄_MC_이상 : BOOL; (* AT %MW1009.13 *) (* S362 MC 이상 *)
    S362_M_총괄_NFB_이상 : BOOL; (* AT %MW1009.11 *) (* S362 NFB 이상 *)
    S362_M_총괄_ROBOT_이상 : BOOL; (* AT %MW1010.1 *) (* S362 ROBOT 이상 *)
    S362_M_총괄_SAFETY_이상 : BOOL; (* AT %MW1009.2 *) (* S362 SAFETY 이상 *)
    S362_M_총괄_공기압_이상 : BOOL; (* AT %MW1009.3 *) (* S362 공기압 이상 *)
    S362_M_총괄_사양_이상 : BOOL; (* AT %MW1009.6 *) (* S362 사양 이상 *)
    S362_M_총괄_오버런_이상 : BOOL; (* AT %MW1009.12 *) (* S362 OVER RUN 이상 *)
    S362_M_총괄_용접타점수_이상 : BOOL; (* AT %MW1010.2 *) (* S362 용접타점수 이상 *)
    S362_M_총괄_이상 : BOOL; (* AT %MW1009.0 *) (* S362_M_총괄_이상 *)
    S362_M_총괄_제품감지_이상 : BOOL; (* AT %MW1009.4 *) (* S362 제품감지 이상 *)
    S362_M_총괄_차종_이상 : BOOL; (* AT %MW1009.5 *) (* S362 차종 이상 *)
    S362_M_총괄_통신_이상 : BOOL; (* AT %MW1009.14 *) (* S362 통신이상 *)
    전체_M_이상_리셋 : BOOL; (* AT %MW308.2 *) (* ALL공정 PB 이상리셋 *)
END_VAR
VAR
    INST : TON;
    INST1 : TON;
    INST10 : TON;
    INST11 : TON;
    INST12 : TON;
    INST13 : TON;
    INST14 : TON;
    INST15 : TON;
    INST16 : TON;
    INST17 : TON;
    INST18 : TON;
    INST19 : TON;
    INST2 : TON;
    INST20 : TON;
    INST21 : TON;
    INST22 : TON;
    INST23 : TON;
    INST24 : TON;
    INST25 : TON;
    INST26 : TON;
    INST27 : TON;
    INST28 : TON;
    INST29 : TON;
    INST3 : TON;
    INST30 : TON;
    INST31 : TON;
    INST32 : TON;
    INST4 : TON;
    INST5 : TON;
    INST6 : TON;
    INST7 : TON;
    INST8 : TON;
    INST9 : TON;
END_VAR
VAR_EXTERNAL
    R361_1_I_RB_PLT_최종UNLOAD_완료 : BOOL; (* AT %MW84013.12 *) (* R361_1_I_RB_PLT_최종UNLOAD_완료 *)
    R361_1_M_I_RB_간섭무_1 : BOOL; (* AT %MW20012.0 *) (* R361_1_M_I_RB_간섭무_1 *)
    R361_1_M_I_RB_간섭무_2 : BOOL; (* AT %MW20012.1 *) (* R361_1_M_I_RB_간섭무_2 *)
    R361_1_M_I_RB_간섭무_3 : BOOL; (* AT %MW20012.2 *) (* R361_1_M_I_RB_간섭무_3 *)
    R361_1_M_I_RB_간섭무_4 : BOOL; (* AT %MW20012.3 *) (* R361_1_M_I_RB_간섭무_4 *)
    R361_1_M_I_RB_이상 : BOOL; (* AT %MW20010.2 *) (* R361_1_M_I_RB_이상 *)
    R361_1_M_I_RB_프로그램_이상 : BOOL; (* AT %MW20010.6 *) (* R361_1_M_I_RB_프로그램_이상 *)
    R361_2_I_RB_PLT_최종UNLOAD_완료 : BOOL; (* AT %MW84023.12 *) (* R361_2_I_RB_PLT_최종UNLOAD_완료 *)
    R361_2_M_I_RB_간섭무_1 : BOOL; (* AT %MW20022.0 *) (* R361_2_M_I_RB_간섭무_1 *)
    R361_2_M_I_RB_간섭무_2 : BOOL; (* AT %MW20022.1 *) (* R361_2_M_I_RB_간섭무_2 *)
    R361_2_M_I_RB_이상 : BOOL; (* AT %MW20020.2 *) (* R361_2_M_I_RB_이상 *)
    R361_2_M_I_RB_프로그램_이상 : BOOL; (* AT %MW20020.6 *) (* R361_2_M_I_RB_프로그램_이상 *)
    ROOF_RACK1_3_PLC_BOX_CP_TRIP : BOOL; (* AT %MW87401.15 *) (* ROOF RACK1 3 PLC BOX CP TRIP *)
    ROOF_RACK1_LC_정상1 : BOOL; (* AT %MW87403.0 *) (* ROOF RACK1 LC 정상1 *)
    ROOF_RACK1_LC_정상2 : BOOL; (* AT %MW87403.1 *) (* ROOF RACK1 LC 정상2 *)
    ROOF_RACK1_PRS_랙감지1 : BOOL; (* AT %MW87400.0 *) (* ROOF RACK1 PRS 랙감지1 *)
    ROOF_RACK1_PRS_랙감지2 : BOOL; (* AT %MW87400.1 *) (* ROOF RACK1 PRS 랙감지2 *)
    ROOF_RACK1_PRS_막장감지 : BOOL; (* AT %MW87400.2 *) (* ROOF RACK1 PRS 막장감지 *)
    ROOF_RACK1_발목감지_정상1 : BOOL; (* AT %MW87403.2 *) (* ROOF RACK1 발목감지 정상1 *)
    ROOF_RACK1_발목감지_정상2 : BOOL; (* AT %MW87403.3 *) (* ROOF RACK1 발목감지 정상2 *)
    ROOF_RACK2_LC_정상1 : BOOL; (* AT %MW87403.4 *) (* ROOF RACK2 LC 정상1 *)
    ROOF_RACK2_LC_정상2 : BOOL; (* AT %MW87403.5 *) (* ROOF RACK2 LC 정상2 *)
    ROOF_RACK2_PRS_랙감지1 : BOOL; (* AT %MW87400.8 *) (* ROOF RACK2 PRS 랙감지1 *)
    ROOF_RACK2_PRS_랙감지2 : BOOL; (* AT %MW87400.9 *) (* ROOF RACK2 PRS 랙감지2 *)
    ROOF_RACK2_PRS_막장감지 : BOOL; (* AT %MW87400.10 *) (* ROOF RACK2 PRS 막장감지 *)
    ROOF_RACK2_발목감지_정상1 : BOOL; (* AT %MW87403.6 *) (* ROOF RACK2 발목감지 정상1 *)
    ROOF_RACK2_발목감지_정상2 : BOOL; (* AT %MW87403.7 *) (* ROOF RACK2 발목감지 정상2 *)
    ROOF_RACK3_LC_정상1 : BOOL; (* AT %MW87403.8 *) (* ROOF RACK3 LC 정상1 *)
    ROOF_RACK3_LC_정상2 : BOOL; (* AT %MW87403.9 *) (* ROOF RACK3 LC 정상2 *)
    ROOF_RACK3_PRS_랙감지1 : BOOL; (* AT %MW87401.0 *) (* ROOF RACK3 PRS 랙감지1 *)
    ROOF_RACK3_PRS_랙감지2 : BOOL; (* AT %MW87401.1 *) (* ROOF RACK3 PRS 랙감지2 *)
    ROOF_RACK3_PRS_막장감지 : BOOL; (* AT %MW87401.2 *) (* ROOF RACK3 PRS 막장감지 *)
    ROOF_RACK3_발목감지_정상1 : BOOL; (* AT %MW87403.10 *) (* ROOF RACK3 발목감지 정상1 *)
    ROOF_RACK3_발목감지_정상2 : BOOL; (* AT %MW87403.11 *) (* ROOF RACK3 발목감지 정상2 *)
    ROOF_RACK4_6_PLC_BOX_CP_TRIP : BOOL; (* AT %MW87451.15 *) (* ROOF RACK4 6 PLC BOX CP TRIP *)
    ROOF_RACK4_LC_정상1 : BOOL; (* AT %MW87453.0 *) (* ROOF RACK4 LC 정상1 *)
    ROOF_RACK4_LC_정상2 : BOOL; (* AT %MW87453.1 *) (* ROOF RACK4 LC 정상2 *)
    ROOF_RACK4_PRS_랙감지1 : BOOL; (* AT %MW87450.0 *) (* ROOF RACK4 PRS 랙감지1 *)
    ROOF_RACK4_PRS_랙감지2 : BOOL; (* AT %MW87450.1 *) (* ROOF RACK4 PRS 랙감지2 *)
    ROOF_RACK4_PRS_막장감지 : BOOL; (* AT %MW87450.2 *) (* ROOF RACK4 PRS 막장감지 *)
    ROOF_RACK4_발목감지_정상1 : BOOL; (* AT %MW87453.2 *) (* ROOF RACK4 발목감지 정상1 *)
    ROOF_RACK4_발목감지_정상2 : BOOL; (* AT %MW87453.3 *) (* ROOF RACK4 발목감지 정상2 *)
    ROOF_RACK5_LC_정상1 : BOOL; (* AT %MW87453.4 *) (* ROOF RACK5 LC 정상1 *)
    ROOF_RACK5_LC_정상2 : BOOL; (* AT %MW87453.5 *) (* ROOF RACK5 LC 정상2 *)
    ROOF_RACK5_PRS_랙감지1 : BOOL; (* AT %MW87450.8 *) (* ROOF RACK5 PRS 랙감지1 *)
    ROOF_RACK5_PRS_랙감지2 : BOOL; (* AT %MW87450.9 *) (* ROOF RACK5 PRS 랙감지2 *)
    ROOF_RACK5_PRS_막장감지 : BOOL; (* AT %MW87450.10 *) (* ROOF RACK5 PRS 막장감지 *)
    ROOF_RACK5_발목감지_정상1 : BOOL; (* AT %MW87453.6 *) (* ROOF RACK5 발목감지 정상1 *)
    ROOF_RACK5_발목감지_정상2 : BOOL; (* AT %MW87453.7 *) (* ROOF RACK5 발목감지 정상2 *)
    ROOF_RACK6_LC_정상1 : BOOL; (* AT %MW87453.8 *) (* ROOF RACK6 LC 정상1 *)
    ROOF_RACK6_LC_정상2 : BOOL; (* AT %MW87453.9 *) (* ROOF RACK6 LC 정상2 *)
    ROOF_RACK6_PRS_랙감지1 : BOOL; (* AT %MW87451.0 *) (* ROOF RACK6 PRS 랙감지1 *)
    ROOF_RACK6_PRS_랙감지2 : BOOL; (* AT %MW87451.1 *) (* ROOF RACK6 PRS 랙감지2 *)
    ROOF_RACK6_PRS_막장감지 : BOOL; (* AT %MW87451.2 *) (* ROOF RACK6 PRS 막장감지 *)
    ROOF_RACK6_발목감지_정상1 : BOOL; (* AT %MW87453.10 *) (* ROOF RACK6 발목감지 정상1 *)
    ROOF_RACK6_발목감지_정상2 : BOOL; (* AT %MW87453.11 *) (* ROOF RACK6 발목감지 정상2 *)
    _0004_EB01_CFG_ER : BOOL; (* AT %MW184022.0 *) (* EB 구성 에러 *)
    _0004_EB01_DEER : BOOL; (* AT %MW184022.1 *) (* EB 운전 중 탈락 *)
    _0004_EB02_CFG_ER : BOOL; (* AT %MW184024.8 *) (* EB 구성 에러 *)
    _0004_EB02_DEER : BOOL; (* AT %MW184024.9 *) (* EB 운전 중 탈락 *)
    _0006_EB20_CFG_ER : BOOL; (* AT %MW186034.0 *) (* EB 구성 에러 *)
    _0006_EB20_DEER : BOOL; (* AT %MW186034.1 *) (* EB 운전 중 탈락 *)
    _0006_EB20_IO_DEER : BOOL; (* AT %MW186035.2 *) (* EB IO 탈락 에러 *)
    _0006_EB20_IO_TYER : BOOL; (* AT %MW186035.1 *) (* EB IO 타입 에러 *)
    _0007_EB40_CFG_ER : BOOL; (* AT %MW187070.0 *) (* EB 구성 에러 *)
    _0007_EB40_DEER : BOOL; (* AT %MW187070.1 *) (* EB 운전 중 탈락 *)
    _0007_EB40_IO_DEER : BOOL; (* AT %MW187071.2 *) (* EB IO 탈락 에러 *)
    _0007_EB40_IO_TYER : BOOL; (* AT %MW187071.1 *) (* EB IO 타입 에러 *)
    _0007_EB45_CFG_ER : BOOL; (* AT %MW187076.0 *) (* EB 구성 에러 *)
    _0007_EB45_DEER : BOOL; (* AT %MW187076.1 *) (* EB 운전 중 탈락 *)
    _0007_EB45_IO_DEER : BOOL; (* AT %MW187077.2 *) (* EB IO 탈락 에러 *)
    _0007_EB45_IO_TYER : BOOL; (* AT %MW187077.1 *) (* EB IO 타입 에러 *)
END_VAR

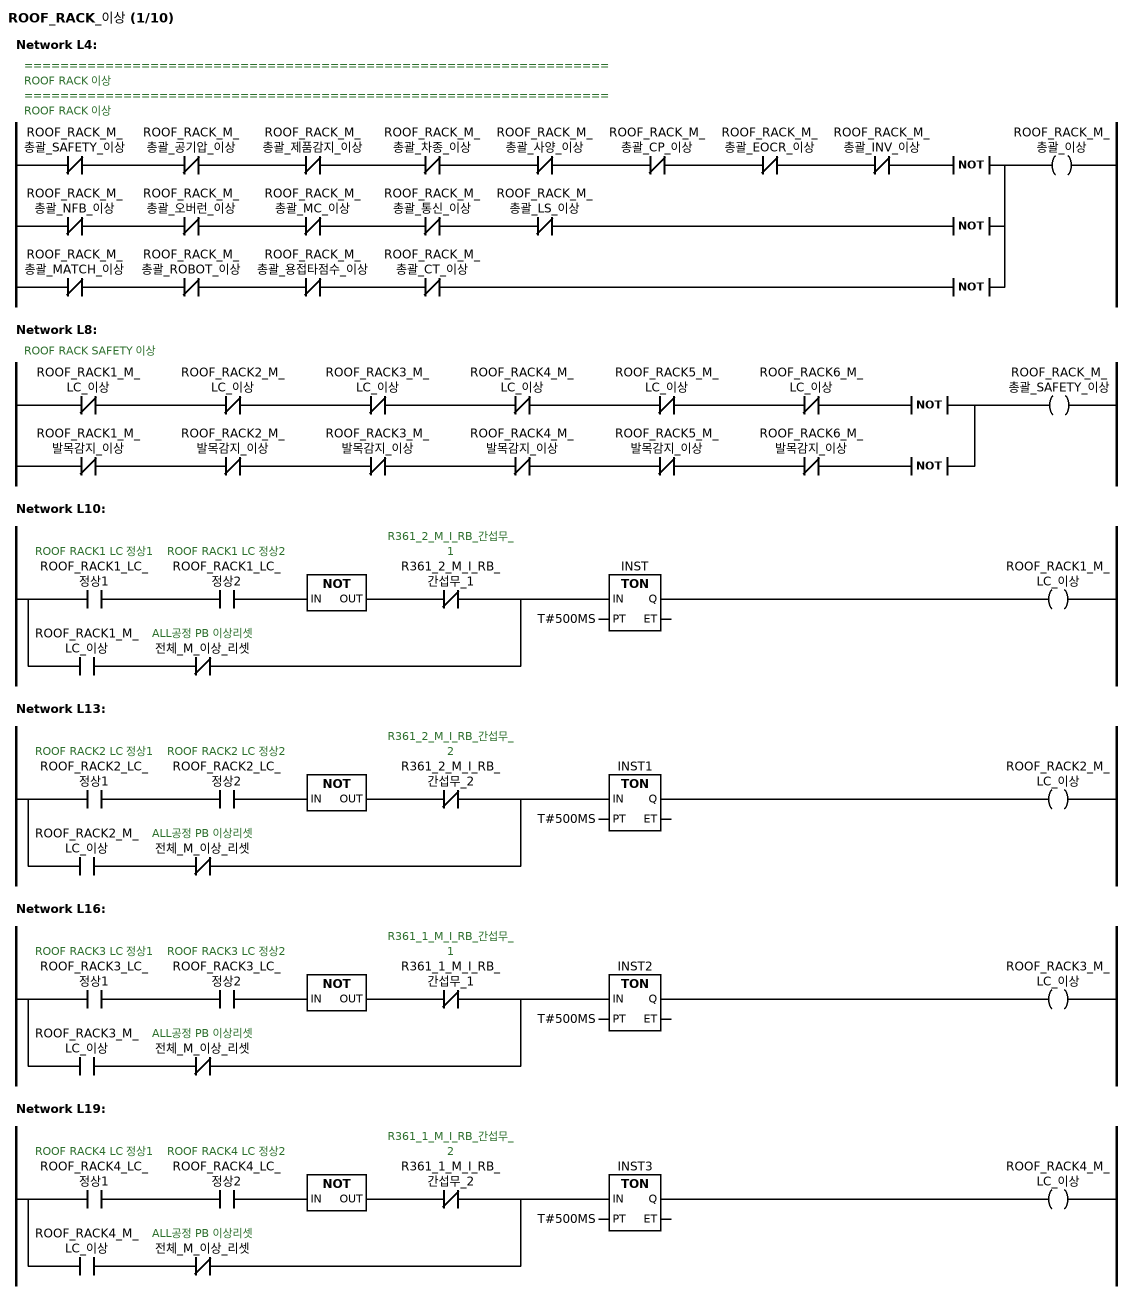
(* ================================================================= *)
(* ROOF RACK 이상 *)
(* ================================================================= *)
(* ROOF RACK 이상 *)
(* Rung L4 *)
ROOF_RACK_M_총괄_이상 := NOT (NOT ROOF_RACK_M_총괄_SAFETY_이상 AND NOT ROOF_RACK_M_총괄_공기압_이상 AND NOT ROOF_RACK_M_총괄_제품감지_이상 AND NOT ROOF_RACK_M_총괄_차종_이상 AND NOT ROOF_RACK_M_총괄_사양_이상 AND NOT ROOF_RACK_M_총괄_CP_이상 AND NOT ROOF_RACK_M_총괄_EOCR_이상 AND NOT ROOF_RACK_M_총괄_INV_이상) OR NOT (NOT ROOF_RACK_M_총괄_NFB_이상 AND NOT ROOF_RACK_M_총괄_오버런_이상 AND NOT ROOF_RACK_M_총괄_MC_이상 AND NOT ROOF_RACK_M_총괄_통신_이상 AND NOT ROOF_RACK_M_총괄_LS_이상) OR NOT (NOT ROOF_RACK_M_총괄_MATCH_이상 AND NOT ROOF_RACK_M_총괄_ROBOT_이상 AND NOT ROOF_RACK_M_총괄_용접타점수_이상 AND NOT ROOF_RACK_M_총괄_CT_이상);
(* ROOF RACK SAFETY 이상 *)
(* Rung L8 *)
ROOF_RACK_M_총괄_SAFETY_이상 := NOT (NOT ROOF_RACK1_M_LC_이상 AND NOT ROOF_RACK2_M_LC_이상 AND NOT ROOF_RACK3_M_LC_이상 AND NOT ROOF_RACK4_M_LC_이상 AND NOT ROOF_RACK5_M_LC_이상 AND NOT ROOF_RACK6_M_LC_이상) OR NOT (NOT ROOF_RACK1_M_발목감지_이상 AND NOT ROOF_RACK2_M_발목감지_이상 AND NOT ROOF_RACK3_M_발목감지_이상 AND NOT ROOF_RACK4_M_발목감지_이상 AND NOT ROOF_RACK5_M_발목감지_이상 AND NOT ROOF_RACK6_M_발목감지_이상);
(* Rung L10 *)
INST(IN := ((NOT (ROOF_RACK1_LC_정상1 AND ROOF_RACK1_LC_정상2)) AND NOT R361_2_M_I_RB_간섭무_1) OR (ROOF_RACK1_M_LC_이상 AND NOT 전체_M_이상_리셋), PT := T#500MS);
ROOF_RACK1_M_LC_이상 := INST.Q;
(* Rung L13 *)
INST1(IN := ((NOT (ROOF_RACK2_LC_정상1 AND ROOF_RACK2_LC_정상2)) AND NOT R361_2_M_I_RB_간섭무_2) OR (ROOF_RACK2_M_LC_이상 AND NOT 전체_M_이상_리셋), PT := T#500MS);
ROOF_RACK2_M_LC_이상 := INST1.Q;
(* Rung L16 *)
INST2(IN := ((NOT (ROOF_RACK3_LC_정상1 AND ROOF_RACK3_LC_정상2)) AND NOT R361_1_M_I_RB_간섭무_1) OR (ROOF_RACK3_M_LC_이상 AND NOT 전체_M_이상_리셋), PT := T#500MS);
ROOF_RACK3_M_LC_이상 := INST2.Q;
(* Rung L19 *)
INST3(IN := ((NOT (ROOF_RACK4_LC_정상1 AND ROOF_RACK4_LC_정상2)) AND NOT R361_1_M_I_RB_간섭무_2) OR (ROOF_RACK4_M_LC_이상 AND NOT 전체_M_이상_리셋), PT := T#500MS);
ROOF_RACK4_M_LC_이상 := INST3.Q;

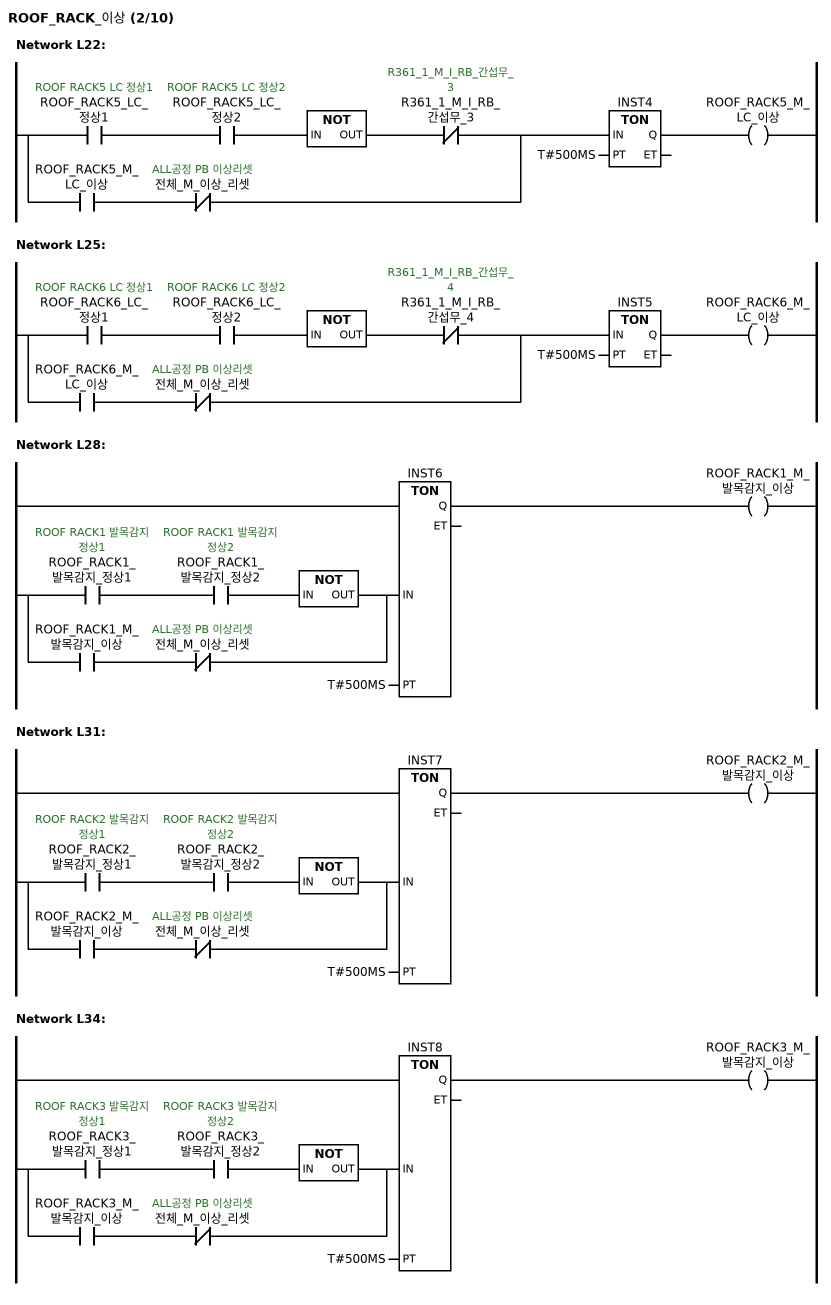
(* Rung L22 *)
INST4(IN := ((NOT (ROOF_RACK5_LC_정상1 AND ROOF_RACK5_LC_정상2)) AND NOT R361_1_M_I_RB_간섭무_3) OR (ROOF_RACK5_M_LC_이상 AND NOT 전체_M_이상_리셋), PT := T#500MS);
ROOF_RACK5_M_LC_이상 := INST4.Q;
(* Rung L25 *)
INST5(IN := ((NOT (ROOF_RACK6_LC_정상1 AND ROOF_RACK6_LC_정상2)) AND NOT R361_1_M_I_RB_간섭무_4) OR (ROOF_RACK6_M_LC_이상 AND NOT 전체_M_이상_리셋), PT := T#500MS);
ROOF_RACK6_M_LC_이상 := INST5.Q;
(* Rung L28 *)
INST6(IN := (NOT (ROOF_RACK1_발목감지_정상1 AND ROOF_RACK1_발목감지_정상2)) OR (ROOF_RACK1_M_발목감지_이상 AND NOT 전체_M_이상_리셋), PT := T#500MS);
ROOF_RACK1_M_발목감지_이상 := INST6.Q;
(* Rung L31 *)
INST7(IN := (NOT (ROOF_RACK2_발목감지_정상1 AND ROOF_RACK2_발목감지_정상2)) OR (ROOF_RACK2_M_발목감지_이상 AND NOT 전체_M_이상_리셋), PT := T#500MS);
ROOF_RACK2_M_발목감지_이상 := INST7.Q;
(* Rung L34 *)
INST8(IN := (NOT (ROOF_RACK3_발목감지_정상1 AND ROOF_RACK3_발목감지_정상2)) OR (ROOF_RACK3_M_발목감지_이상 AND NOT 전체_M_이상_리셋), PT := T#500MS);
ROOF_RACK3_M_발목감지_이상 := INST8.Q;

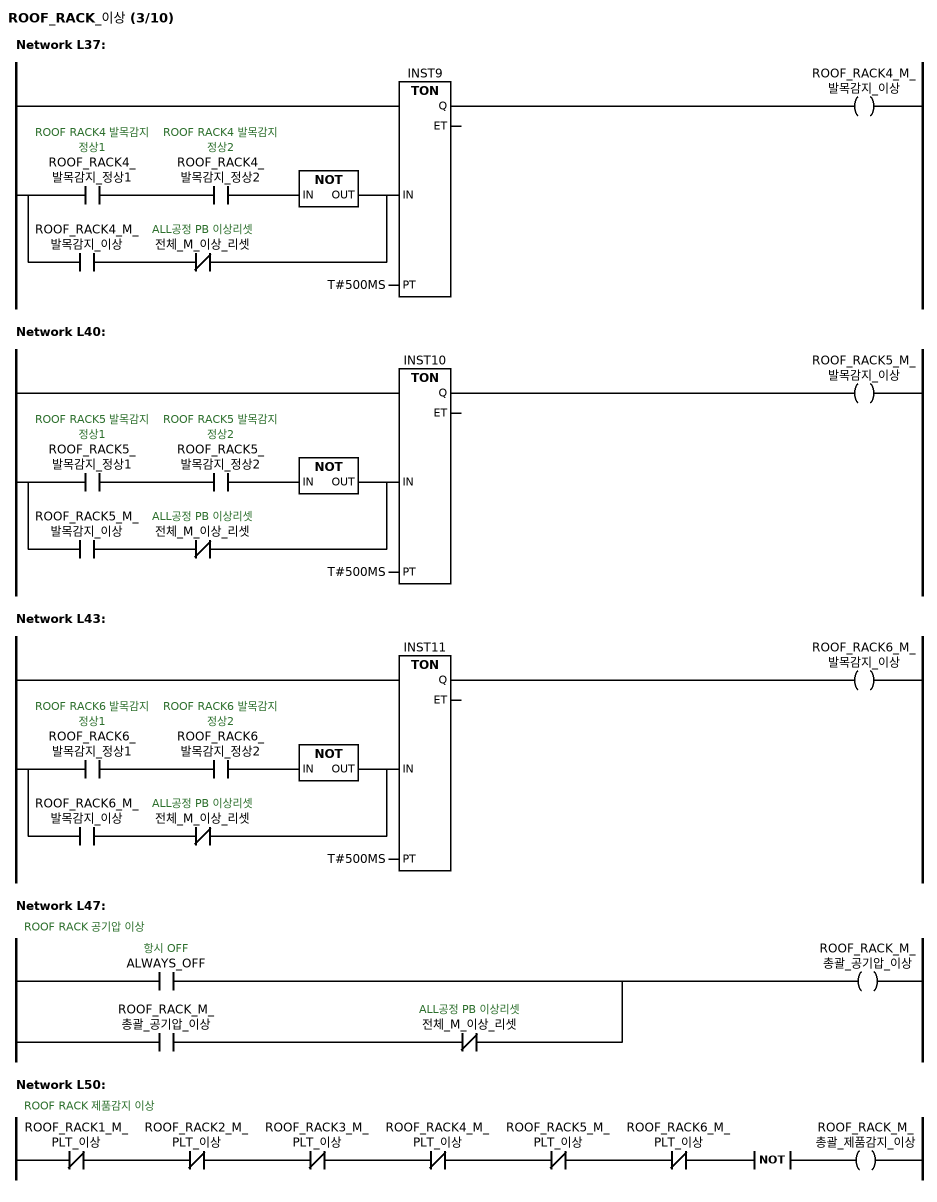
(* Rung L37 *)
INST9(IN := (NOT (ROOF_RACK4_발목감지_정상1 AND ROOF_RACK4_발목감지_정상2)) OR (ROOF_RACK4_M_발목감지_이상 AND NOT 전체_M_이상_리셋), PT := T#500MS);
ROOF_RACK4_M_발목감지_이상 := INST9.Q;
(* Rung L40 *)
INST10(IN := (NOT (ROOF_RACK5_발목감지_정상1 AND ROOF_RACK5_발목감지_정상2)) OR (ROOF_RACK5_M_발목감지_이상 AND NOT 전체_M_이상_리셋), PT := T#500MS);
ROOF_RACK5_M_발목감지_이상 := INST10.Q;
(* Rung L43 *)
INST11(IN := (NOT (ROOF_RACK6_발목감지_정상1 AND ROOF_RACK6_발목감지_정상2)) OR (ROOF_RACK6_M_발목감지_이상 AND NOT 전체_M_이상_리셋), PT := T#500MS);
ROOF_RACK6_M_발목감지_이상 := INST11.Q;
(* ROOF RACK 공기압 이상 *)
(* Rung L47 *)
ROOF_RACK_M_총괄_공기압_이상 := ALWAYS_OFF OR (ROOF_RACK_M_총괄_공기압_이상 AND NOT 전체_M_이상_리셋);
(* ROOF RACK 제품감지 이상 *)
(* Rung L50 *)
ROOF_RACK_M_총괄_제품감지_이상 := NOT (NOT ROOF_RACK1_M_PLT_이상 AND NOT ROOF_RACK2_M_PLT_이상 AND NOT ROOF_RACK3_M_PLT_이상 AND NOT ROOF_RACK4_M_PLT_이상 AND NOT ROOF_RACK5_M_PLT_이상 AND NOT ROOF_RACK6_M_PLT_이상);

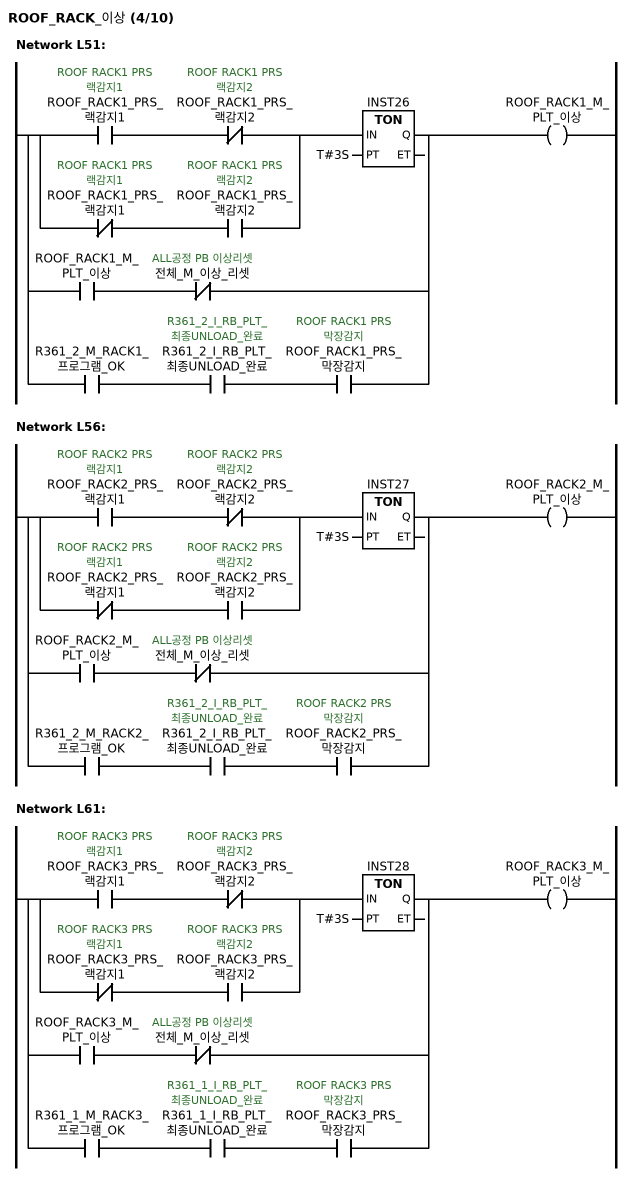
(* Rung L51 *)
INST26(IN := (ROOF_RACK1_PRS_랙감지1 AND NOT ROOF_RACK1_PRS_랙감지2) OR (NOT ROOF_RACK1_PRS_랙감지1 AND ROOF_RACK1_PRS_랙감지2), PT := T#3S);
ROOF_RACK1_M_PLT_이상 := INST26.Q OR (ROOF_RACK1_M_PLT_이상 AND NOT 전체_M_이상_리셋) OR (R361_2_M_RACK1_프로그램_OK AND R361_2_I_RB_PLT_최종UNLOAD_완료 AND ROOF_RACK1_PRS_막장감지);
(* Rung L56 *)
INST27(IN := (ROOF_RACK2_PRS_랙감지1 AND NOT ROOF_RACK2_PRS_랙감지2) OR (NOT ROOF_RACK2_PRS_랙감지1 AND ROOF_RACK2_PRS_랙감지2), PT := T#3S);
ROOF_RACK2_M_PLT_이상 := INST27.Q OR (ROOF_RACK2_M_PLT_이상 AND NOT 전체_M_이상_리셋) OR (R361_2_M_RACK2_프로그램_OK AND R361_2_I_RB_PLT_최종UNLOAD_완료 AND ROOF_RACK2_PRS_막장감지);
(* Rung L61 *)
INST28(IN := (ROOF_RACK3_PRS_랙감지1 AND NOT ROOF_RACK3_PRS_랙감지2) OR (NOT ROOF_RACK3_PRS_랙감지1 AND ROOF_RACK3_PRS_랙감지2), PT := T#3S);
ROOF_RACK3_M_PLT_이상 := INST28.Q OR (ROOF_RACK3_M_PLT_이상 AND NOT 전체_M_이상_리셋) OR (R361_1_M_RACK3_프로그램_OK AND R361_1_I_RB_PLT_최종UNLOAD_완료 AND ROOF_RACK3_PRS_막장감지);

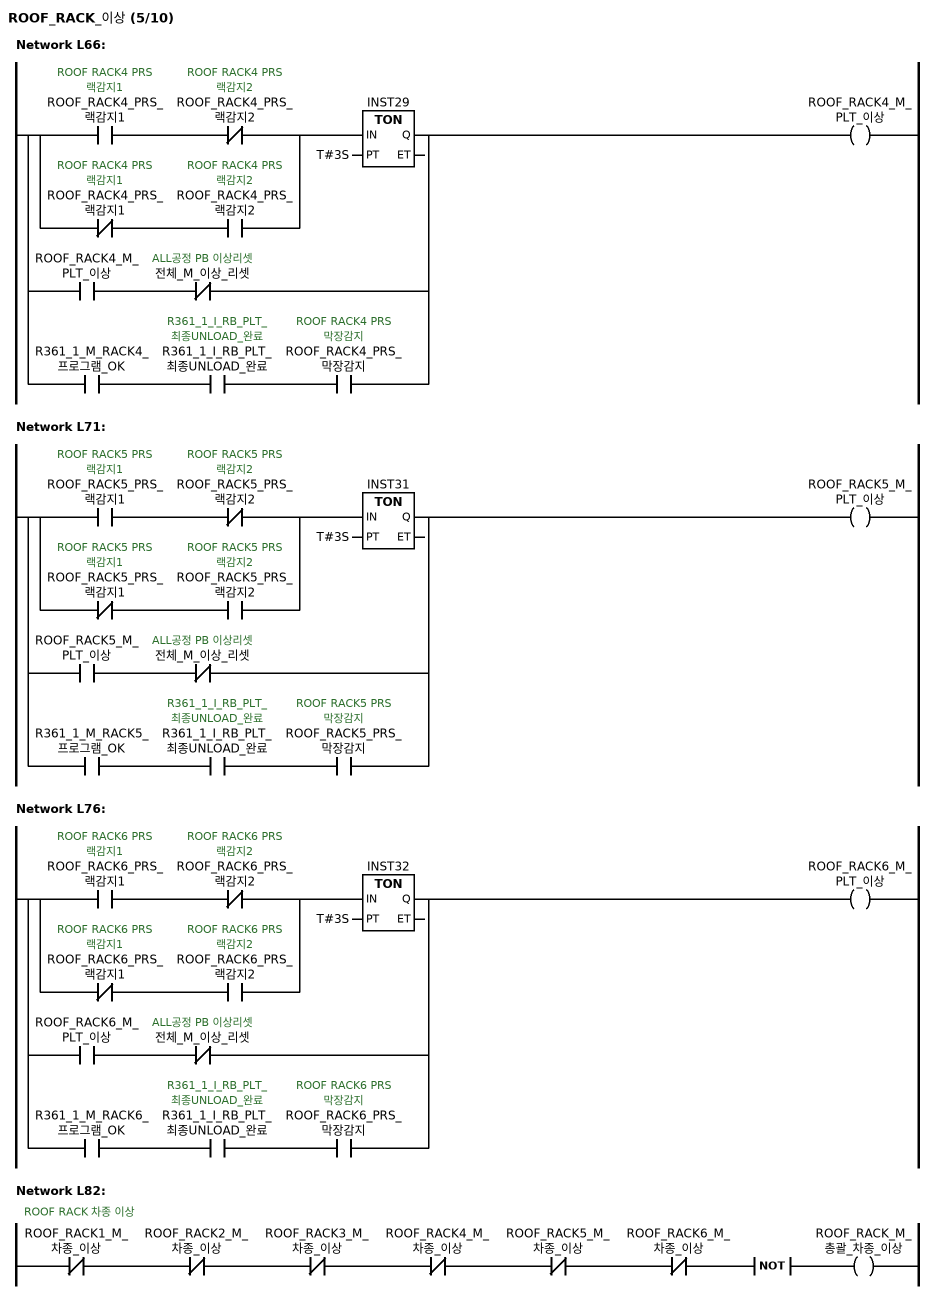
(* Rung L66 *)
INST29(IN := (ROOF_RACK4_PRS_랙감지1 AND NOT ROOF_RACK4_PRS_랙감지2) OR (NOT ROOF_RACK4_PRS_랙감지1 AND ROOF_RACK4_PRS_랙감지2), PT := T#3S);
ROOF_RACK4_M_PLT_이상 := INST29.Q OR (ROOF_RACK4_M_PLT_이상 AND NOT 전체_M_이상_리셋) OR (R361_1_M_RACK4_프로그램_OK AND R361_1_I_RB_PLT_최종UNLOAD_완료 AND ROOF_RACK4_PRS_막장감지);
(* Rung L71 *)
INST31(IN := (ROOF_RACK5_PRS_랙감지1 AND NOT ROOF_RACK5_PRS_랙감지2) OR (NOT ROOF_RACK5_PRS_랙감지1 AND ROOF_RACK5_PRS_랙감지2), PT := T#3S);
ROOF_RACK5_M_PLT_이상 := INST31.Q OR (ROOF_RACK5_M_PLT_이상 AND NOT 전체_M_이상_리셋) OR (R361_1_M_RACK5_프로그램_OK AND R361_1_I_RB_PLT_최종UNLOAD_완료 AND ROOF_RACK5_PRS_막장감지);
(* Rung L76 *)
INST32(IN := (ROOF_RACK6_PRS_랙감지1 AND NOT ROOF_RACK6_PRS_랙감지2) OR (NOT ROOF_RACK6_PRS_랙감지1 AND ROOF_RACK6_PRS_랙감지2), PT := T#3S);
ROOF_RACK6_M_PLT_이상 := INST32.Q OR (ROOF_RACK6_M_PLT_이상 AND NOT 전체_M_이상_리셋) OR (R361_1_M_RACK6_프로그램_OK AND R361_1_I_RB_PLT_최종UNLOAD_완료 AND ROOF_RACK6_PRS_막장감지);
(* ROOF RACK 차종 이상 *)
(* Rung L82 *)
ROOF_RACK_M_총괄_차종_이상 := NOT (NOT ROOF_RACK1_M_차종_이상 AND NOT ROOF_RACK2_M_차종_이상 AND NOT ROOF_RACK3_M_차종_이상 AND NOT ROOF_RACK4_M_차종_이상 AND NOT ROOF_RACK5_M_차종_이상 AND NOT ROOF_RACK6_M_차종_이상);

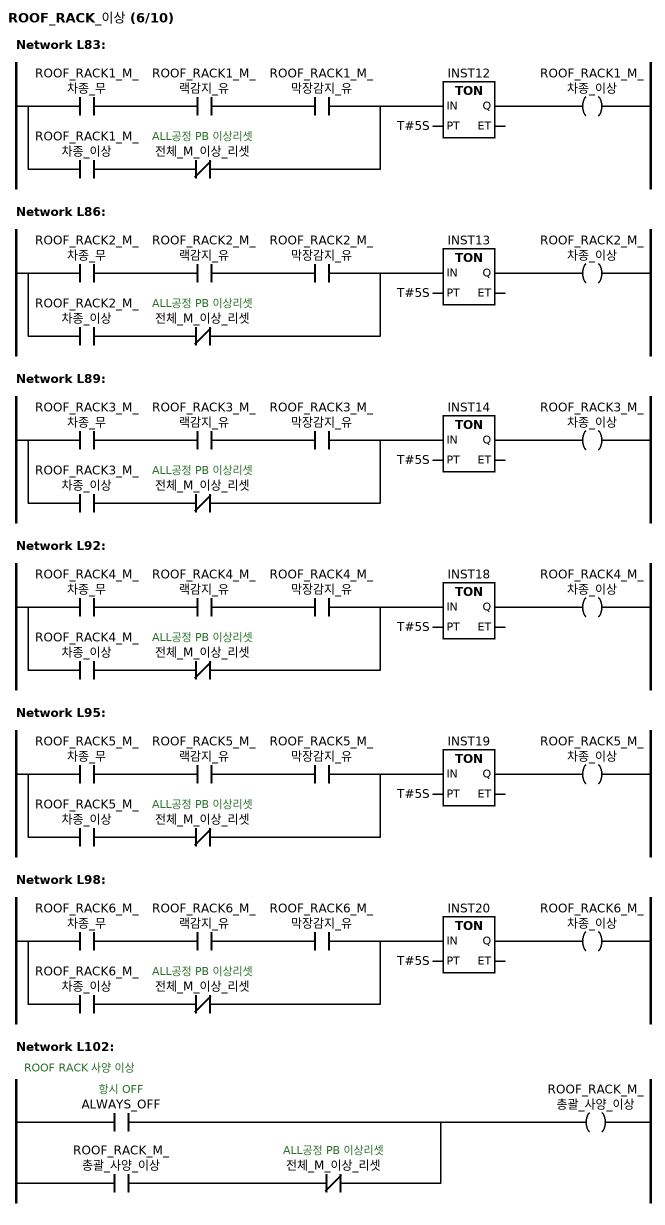
(* Rung L83 *)
INST12(IN := (ROOF_RACK1_M_차종_무 AND ROOF_RACK1_M_랙감지_유 AND ROOF_RACK1_M_막장감지_유) OR (ROOF_RACK1_M_차종_이상 AND NOT 전체_M_이상_리셋), PT := T#5S);
ROOF_RACK1_M_차종_이상 := INST12.Q;
(* Rung L86 *)
INST13(IN := (ROOF_RACK2_M_차종_무 AND ROOF_RACK2_M_랙감지_유 AND ROOF_RACK2_M_막장감지_유) OR (ROOF_RACK2_M_차종_이상 AND NOT 전체_M_이상_리셋), PT := T#5S);
ROOF_RACK2_M_차종_이상 := INST13.Q;
(* Rung L89 *)
INST14(IN := (ROOF_RACK3_M_차종_무 AND ROOF_RACK3_M_랙감지_유 AND ROOF_RACK3_M_막장감지_유) OR (ROOF_RACK3_M_차종_이상 AND NOT 전체_M_이상_리셋), PT := T#5S);
ROOF_RACK3_M_차종_이상 := INST14.Q;
(* Rung L92 *)
INST18(IN := (ROOF_RACK4_M_차종_무 AND ROOF_RACK4_M_랙감지_유 AND ROOF_RACK4_M_막장감지_유) OR (ROOF_RACK4_M_차종_이상 AND NOT 전체_M_이상_리셋), PT := T#5S);
ROOF_RACK4_M_차종_이상 := INST18.Q;
(* Rung L95 *)
INST19(IN := (ROOF_RACK5_M_차종_무 AND ROOF_RACK5_M_랙감지_유 AND ROOF_RACK5_M_막장감지_유) OR (ROOF_RACK5_M_차종_이상 AND NOT 전체_M_이상_리셋), PT := T#5S);
ROOF_RACK5_M_차종_이상 := INST19.Q;
(* Rung L98 *)
INST20(IN := (ROOF_RACK6_M_차종_무 AND ROOF_RACK6_M_랙감지_유 AND ROOF_RACK6_M_막장감지_유) OR (ROOF_RACK6_M_차종_이상 AND NOT 전체_M_이상_리셋), PT := T#5S);
ROOF_RACK6_M_차종_이상 := INST20.Q;
(* ROOF RACK 사양 이상 *)
(* Rung L102 *)
ROOF_RACK_M_총괄_사양_이상 := ALWAYS_OFF OR (ROOF_RACK_M_총괄_사양_이상 AND NOT 전체_M_이상_리셋);

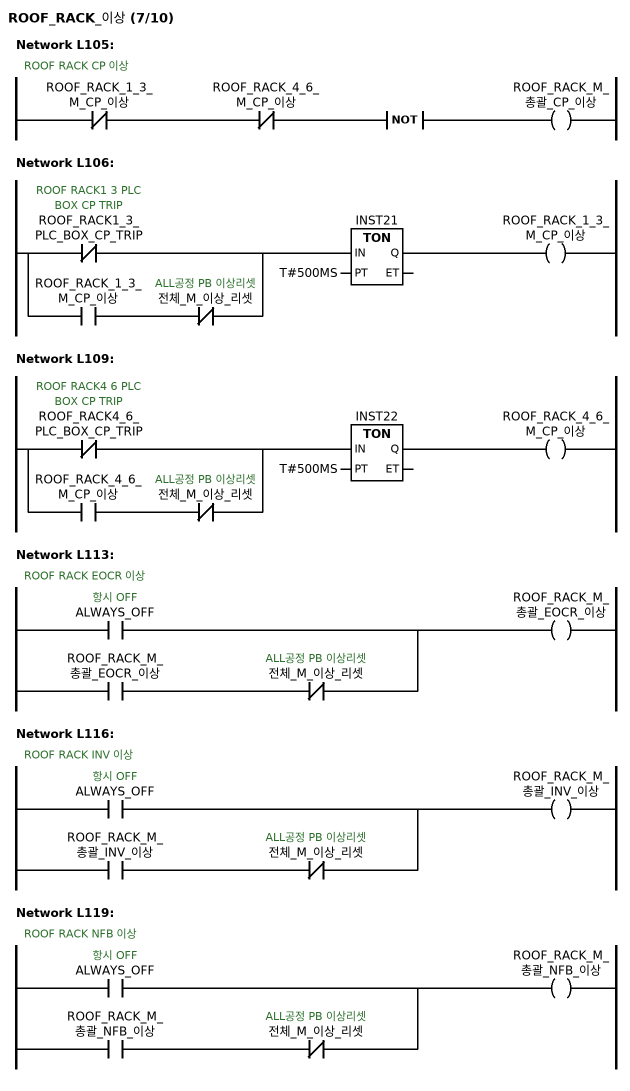
(* ROOF RACK CP 이상 *)
(* Rung L105 *)
ROOF_RACK_M_총괄_CP_이상 := NOT (NOT ROOF_RACK_1_3_M_CP_이상 AND NOT ROOF_RACK_4_6_M_CP_이상);
(* Rung L106 *)
INST21(IN := NOT ROOF_RACK1_3_PLC_BOX_CP_TRIP OR (ROOF_RACK_1_3_M_CP_이상 AND NOT 전체_M_이상_리셋), PT := T#500MS);
ROOF_RACK_1_3_M_CP_이상 := INST21.Q;
(* Rung L109 *)
INST22(IN := NOT ROOF_RACK4_6_PLC_BOX_CP_TRIP OR (ROOF_RACK_4_6_M_CP_이상 AND NOT 전체_M_이상_리셋), PT := T#500MS);
ROOF_RACK_4_6_M_CP_이상 := INST22.Q;
(* ROOF RACK EOCR 이상 *)
(* Rung L113 *)
ROOF_RACK_M_총괄_EOCR_이상 := ALWAYS_OFF OR (ROOF_RACK_M_총괄_EOCR_이상 AND NOT 전체_M_이상_리셋);
(* ROOF RACK INV 이상 *)
(* Rung L116 *)
ROOF_RACK_M_총괄_INV_이상 := ALWAYS_OFF OR (ROOF_RACK_M_총괄_INV_이상 AND NOT 전체_M_이상_리셋);
(* ROOF RACK NFB 이상 *)
(* Rung L119 *)
ROOF_RACK_M_총괄_NFB_이상 := ALWAYS_OFF OR (ROOF_RACK_M_총괄_NFB_이상 AND NOT 전체_M_이상_리셋);

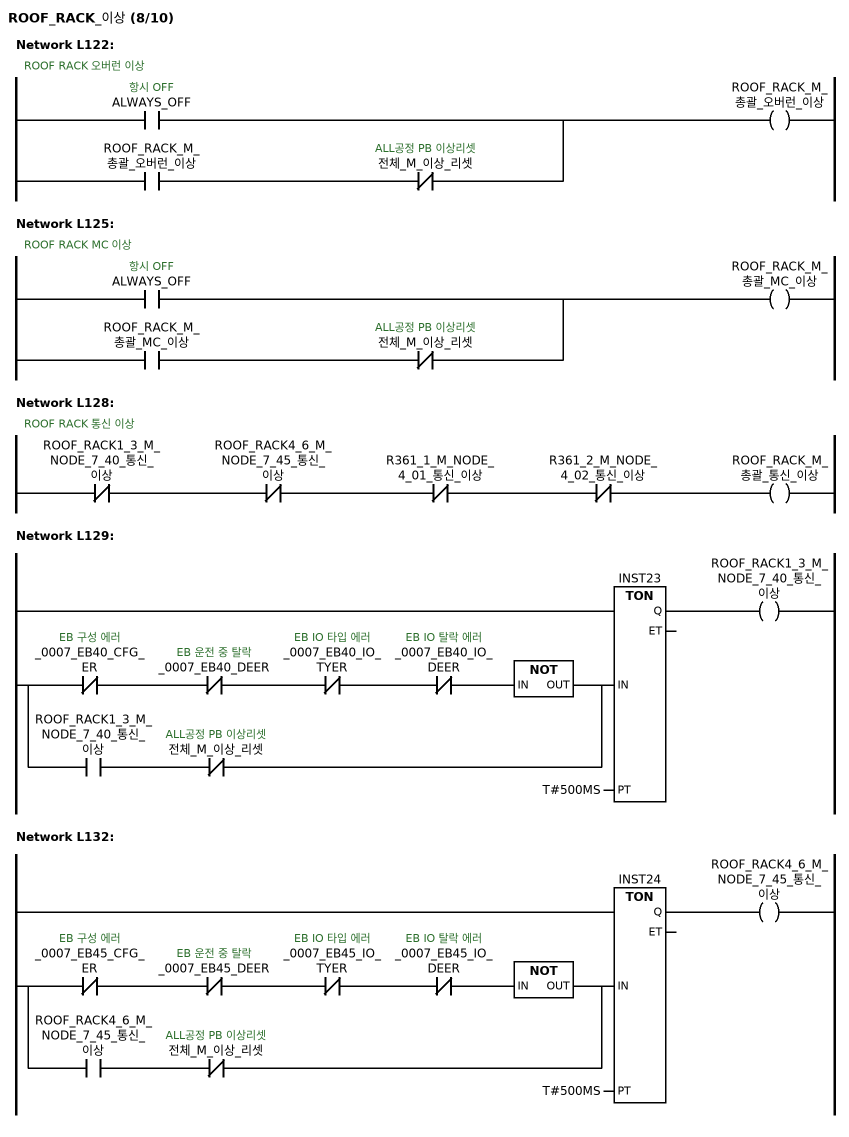
(* ROOF RACK 오버런 이상 *)
(* Rung L122 *)
ROOF_RACK_M_총괄_오버런_이상 := ALWAYS_OFF OR (ROOF_RACK_M_총괄_오버런_이상 AND NOT 전체_M_이상_리셋);
(* ROOF RACK MC 이상 *)
(* Rung L125 *)
ROOF_RACK_M_총괄_MC_이상 := ALWAYS_OFF OR (ROOF_RACK_M_총괄_MC_이상 AND NOT 전체_M_이상_리셋);
(* ROOF RACK 통신 이상 *)
(* Rung L128 *)
ROOF_RACK_M_총괄_통신_이상 := NOT ROOF_RACK1_3_M_NODE_7_40_통신_이상 AND NOT ROOF_RACK4_6_M_NODE_7_45_통신_이상 AND NOT R361_1_M_NODE_4_01_통신_이상 AND NOT R361_2_M_NODE_4_02_통신_이상;
(* Rung L129 *)
INST23(IN := (NOT (NOT _0007_EB40_CFG_ER AND NOT _0007_EB40_DEER AND NOT _0007_EB40_IO_TYER AND NOT _0007_EB40_IO_DEER)) OR (ROOF_RACK1_3_M_NODE_7_40_통신_이상 AND NOT 전체_M_이상_리셋), PT := T#500MS);
ROOF_RACK1_3_M_NODE_7_40_통신_이상 := INST23.Q;
(* Rung L132 *)
INST24(IN := (NOT (NOT _0007_EB45_CFG_ER AND NOT _0007_EB45_DEER AND NOT _0007_EB45_IO_TYER AND NOT _0007_EB45_IO_DEER)) OR (ROOF_RACK4_6_M_NODE_7_45_통신_이상 AND NOT 전체_M_이상_리셋), PT := T#500MS);
ROOF_RACK4_6_M_NODE_7_45_통신_이상 := INST24.Q;

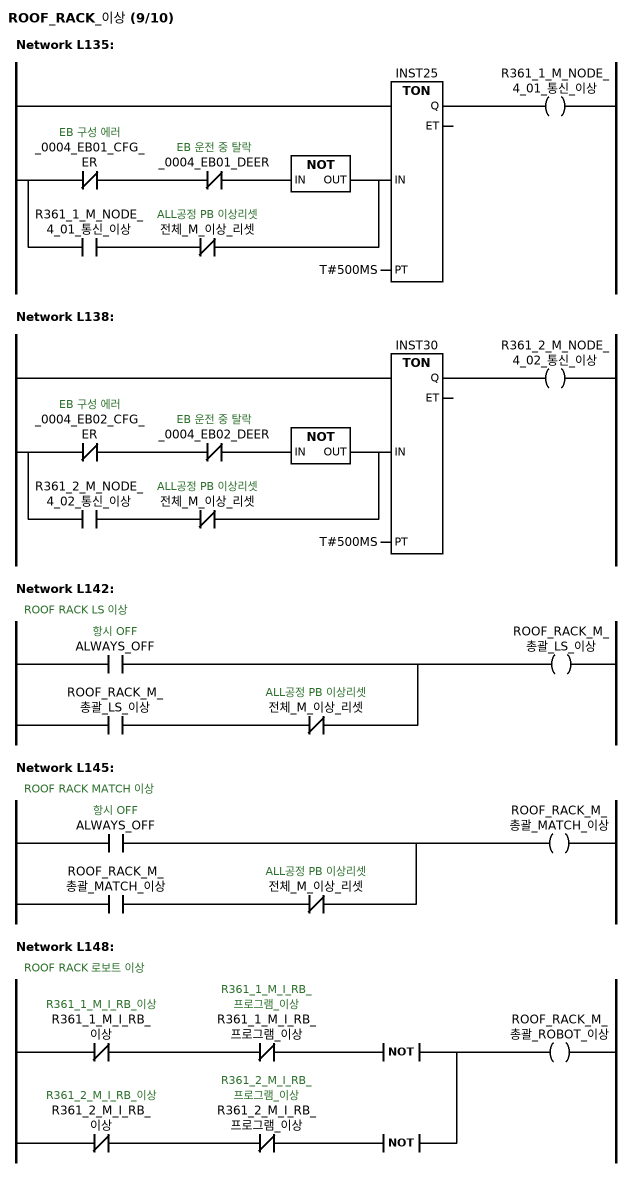
(* Rung L135 *)
INST25(IN := (NOT (NOT _0004_EB01_CFG_ER AND NOT _0004_EB01_DEER)) OR (R361_1_M_NODE_4_01_통신_이상 AND NOT 전체_M_이상_리셋), PT := T#500MS);
R361_1_M_NODE_4_01_통신_이상 := INST25.Q;
(* Rung L138 *)
INST30(IN := (NOT (NOT _0004_EB02_CFG_ER AND NOT _0004_EB02_DEER)) OR (R361_2_M_NODE_4_02_통신_이상 AND NOT 전체_M_이상_리셋), PT := T#500MS);
R361_2_M_NODE_4_02_통신_이상 := INST30.Q;
(* ROOF RACK LS 이상 *)
(* Rung L142 *)
ROOF_RACK_M_총괄_LS_이상 := ALWAYS_OFF OR (ROOF_RACK_M_총괄_LS_이상 AND NOT 전체_M_이상_리셋);
(* ROOF RACK MATCH 이상 *)
(* Rung L145 *)
ROOF_RACK_M_총괄_MATCH_이상 := ALWAYS_OFF OR (ROOF_RACK_M_총괄_MATCH_이상 AND NOT 전체_M_이상_리셋);
(* ROOF RACK 로보트 이상 *)
(* Rung L148 *)
ROOF_RACK_M_총괄_ROBOT_이상 := NOT (NOT R361_1_M_I_RB_이상 AND NOT R361_1_M_I_RB_프로그램_이상) OR NOT (NOT R361_2_M_I_RB_이상 AND NOT R361_2_M_I_RB_프로그램_이상);

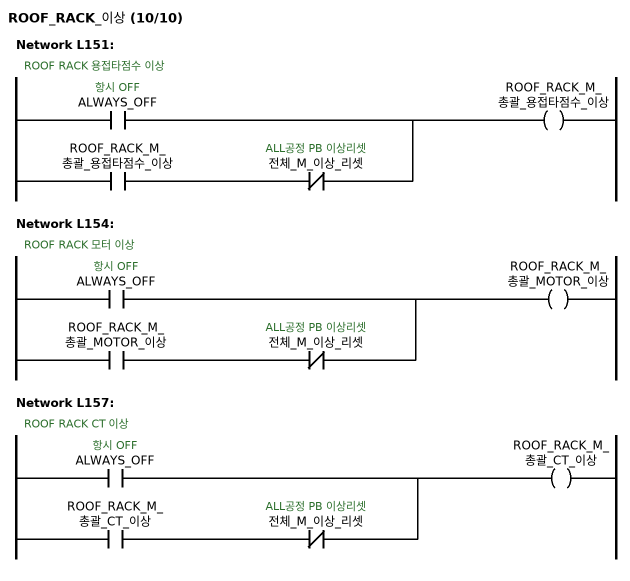
(* ROOF RACK 용접타점수 이상 *)
(* Rung L151 *)
ROOF_RACK_M_총괄_용접타점수_이상 := ALWAYS_OFF OR (ROOF_RACK_M_총괄_용접타점수_이상 AND NOT 전체_M_이상_리셋);
(* ROOF RACK 모터 이상 *)
(* Rung L154 *)
ROOF_RACK_M_총괄_MOTOR_이상 := ALWAYS_OFF OR (ROOF_RACK_M_총괄_MOTOR_이상 AND NOT 전체_M_이상_리셋);
(* ROOF RACK CT 이상 *)
(* Rung L157 *)
ROOF_RACK_M_총괄_CT_이상 := ALWAYS_OFF OR (ROOF_RACK_M_총괄_CT_이상 AND NOT 전체_M_이상_리셋);
END_PROGRAM

PROGRAM S362_S363_유틸리티 (* task: 스캔 프로그램 *)
VAR
    A_차종 : BOOL;
    C_차종 : BOOL;
    INST : TON;
    INST33 : TON;
    INV_TURN기억 : BOOL;
    LOCK_A : BOOL;
    LOCK_B : BOOL;
    PART_SET : BOOL;
    S362_READY : TON;
    T362_AUTO : TON;
END_VAR
VAR_EXTERNAL
    EGIS_CWS : BOOL;
    HOP_PBL_운전준비_ON : BOOL; (* AT %MW87500.0 *) (* HOP_PBL_운전준비_ON *)
    HOP_PLB_362_4_자동_운전 : BOOL; (* AT %MW87500.4 *) (* HOP PLB 362~4 자동기동 *)
    HOP_SSP_362_4_수동_선택 : BOOL; (* AT %MW87500.3 *) (* HOP 362~4 수동선택 *)
    HOP_SSP_362_4_자동_선택 : BOOL; (* AT %MW87500.2 *) (* HOP 362~4 자동선택 *)
    MCP_PBL_362_4_자동_운전 : BOOL; (* AT %MW87630.4 *) (* MCP PBL 362~4 자동기동 *)
    MCP_PBL_운전준비_ON : BOOL; (* AT %MW87630.0 *) (* MCP_PBL_운전준비_ON *)
    MCP_SPB_작업완료_RESET : BOOL; (* AT %MW87631.6 *) (* MCP_SPB_작업완료_RESET *)
    MCP_SPB_작업완료_SET : BOOL; (* AT %MW87631.7 *) (* MCP_SPB_작업완료_SET *)
    MCP_SSP_362_4_수동_선택 : BOOL; (* AT %MW87630.2 *) (* MCP 362~4 수동선택 *)
    MCP_SSP_362_4_자동_선택 : BOOL; (* AT %MW87630.3 *) (* MCP 362~4 자동동선택 *)
    R363_1_M_I_RB_1차_작업완료 : BOOL; (* AT %MW20031.2 *) (* R363_1_M_I_RB_1차_작업완료 *)
    R363_1_M_I_RB_간섭무_1 : BOOL; (* AT %MW20032.0 *) (* R363_1_M_I_RB_간섭무_1 *)
    R363_1_M_I_RB_원위치 : BOOL; (* AT %MW20030.3 *) (* R363_1_M_I_RB_원위치 *)
    R363_2_M_I_RB_1차_작업완료 : BOOL; (* AT %MW20041.2 *) (* R363_2_M_I_RB_1차_작업완료 *)
    R363_2_M_I_RB_간섭무_1 : BOOL; (* AT %MW20042.0 *) (* R363_2_M_I_RB_간섭무_1 *)
    R363_2_M_I_RB_원위치 : BOOL; (* AT %MW20040.3 *) (* R363_2_M_I_RB_원위치 *)
    S362_6_INV1_RETURN : BOOL; (* AT %MW95014.1 *) (* S362_6_INV1_RETURN *)
    S362_6_INV1_SAFETY1_ON : BOOL; (* AT %MW95014.5 *) (* S362_6_INV1_SAFETY1_ON *)
    S362_6_INV1_SAFETY2_ON : BOOL; (* AT %MW95014.6 *) (* S362_6_INV1_SAFETY2_ON *)
    S362_6_INV1_TURN : BOOL; (* AT %MW95014.0 *) (* S362_6_INV1_TURN *)
    S362_6_INV1_이상_리셋 : BOOL; (* AT %MW95014.3 *) (* S362_6_INV1_이상_리셋 *)
    S362_6_INV2_RETURN : BOOL; (* AT %MW95014.9 *) (* S362_6_INV2_RETURN *)
    S362_6_INV2_SAFETY1_ON : BOOL; (* AT %MW95014.13 *) (* S362_6_INV2_SAFETY1_ON *)
    S362_6_INV2_SAFETY2_ON : BOOL; (* AT %MW95014.14 *) (* S362_6_INV2_SAFETY2_ON *)
    S362_6_INV2_TURN : BOOL; (* AT %MW95014.8 *) (* S362_6_INV2_TURN *)
    S362_6_INV2_이상_리셋 : BOOL; (* AT %MW95014.11 *) (* S362_6_INV2_이상_리셋 *)
    S362_LC_정상1 : BOOL; (* AT %MW87105.3 *)
    S362_LC_정상2 : BOOL; (* AT %MW87105.4 *)
    S362_MAT_정상1 : BOOL; (* AT %MW87105.6 *)
    S362_MAT_정상2 : BOOL; (* AT %MW87105.7 *)
    S362_PB_AX_작업_완료 : BOOL; (* AT %MW87102.9 *) (* S362_PB_AX_작업_완료 *)
    S362_PRS_AX_COM_LH_CHECK : BOOL; (* AT %MW87101.1 *) (* S362_PRS_AX_COM_LH_CHECK *)
    S362_PRS_AX_COM_RH_CHECK : BOOL; (* AT %MW87101.0 *) (* S362_PRS_AX_COM_RH_CHECK *)
    S362_PRS_AX_GR_LH_CHECK : BOOL; (* AT %MW87101.3 *) (* S362_PRS_AX_GR_LH_CHECK *)
    S362_PRS_AX_GR_RH_CHECK : BOOL; (* AT %MW87101.2 *) (* S362_PRS_AX_GR_RH_CHECK *)
    S362_PRS_AX_RAIL_LH_CHECK : BOOL; (* AT %MW87101.7 *) (* S362_PRS_AX_RAIL_LH_CHECK *)
    S362_PRS_AX_RAIL_RH_CHECK : BOOL; (* AT %MW87101.6 *) (* S362_PRS_AX_RAIL_RH_CHECK *)
    S362_PRS_AX_SR_LH_CHECK : BOOL; (* AT %MW87101.5 *) (* S362_PRS_AX_SR_LH_CHECK *)
    S362_PRS_AX_SR_RH_CHECK : BOOL; (* AT %MW87101.4 *) (* S362_PRS_AX_SR_RH_CHECK *)
END_VAR
VAR_EXTERNAL RETAIN
    HMI_M_선택_MOD_S362 : BOOL; (* AT %MW6.0 *) (* HMI M 선택 MOD S362 *)
    R361_1_M_차종_유 : BOOL; (* AT %MW1502.0 *)
    R361_2_M_차종_유 : BOOL; (* AT %MW1502.2 *)
    R363_2_M_SEQ : WORD; (* AT %MW10040 *) (* R363 2 M SEQ *)
    R363_2_M_차종1_AX : BOOL; (* AT %MW10041.0 *) (* R363 2 M 차종1 AX *)
    R363_2_M_차종1_B : BOOL; (* AT %MW10041.1 *) (* R363 2 M 차종1 B *)
    R363_2_M_차종1_C : BOOL; (* AT %MW10041.2 *) (* R363 2 M 차종1 C *)
    R363_2_M_차종1_D : BOOL; (* AT %MW10041.3 *) (* R363 2 M 차종1 D *)
    R363_2_M_차종1_E : BOOL; (* AT %MW10041.4 *) (* R363 2 M 차종1 E *)
    R363_2_M_차종1_F : BOOL; (* AT %MW10041.5 *) (* R363 2 M 차종1 F *)
    R363_2_M_차종1_G : BOOL; (* AT %MW10041.6 *) (* R363 2 M 차종1 G *)
    R363_2_M_차종1_H : BOOL; (* AT %MW10041.7 *) (* R363 2 M 차종1 H *)
    R363_2_M_차종2_3DR : BOOL; (* AT %MW10041.8 *) (* R363 2 M 차종2 3DR *)
    R363_2_M_차종2_4DR : BOOL; (* AT %MW10041.9 *) (* R363 2 M 차종2 4DR *)
    R363_2_M_차종2_5DR : BOOL; (* AT %MW10041.10 *) (* R363 2 M 차종2 5DR *)
    R363_2_M_차종2_SP1 : BOOL; (* AT %MW10041.12 *) (* R363 2 M 차종2 SP1 *)
    R363_2_M_차종2_SP2 : BOOL; (* AT %MW10041.13 *) (* R363 2 M 차종2 SP2 *)
    R363_2_M_차종2_WGN : BOOL; (* AT %MW10041.11 *) (* R363 2 M 차종2 WGN *)
    R363_2_M_차종3_LHD : BOOL; (* AT %MW10041.14 *) (* R363 2 M 차종3 LHD *)
    R363_2_M_차종3_RHD : BOOL; (* AT %MW10041.15 *) (* R363 2 M 차종3 RHD *)
    R363_2_M_차종4_EEC : BOOL; (* AT %MW10042.3 *) (* R363 2 M 차종4 EEC *)
    R363_2_M_차종4_SP1 : BOOL; (* AT %MW10042.8 *) (* R363 2 M 차종4 SP1 *)
    R363_2_M_차종4_SP2 : BOOL; (* AT %MW10042.9 *) (* R363 2 M 차종4 SP2 *)
    R363_2_M_차종4_SP3 : BOOL; (* AT %MW10042.11 *) (* R363 2 M 차종4 SP3 *)
    R363_2_M_차종4_SP4 : BOOL; (* AT %MW10042.12 *) (* R363 2 M 차종4 SP4 *)
    R363_2_M_차종4_SP5 : BOOL; (* AT %MW10042.13 *) (* R363 2 M 차종4 SP5 *)
    R363_2_M_차종4_SP6 : BOOL; (* AT %MW10042.14 *) (* R363 2 M 차종4 SP6 *)
    R363_2_M_차종4_SP7 : BOOL; (* AT %MW10042.15 *) (* R363 2 M 차종4 SP7 *)
    R363_2_M_차종4_내수 : BOOL; (* AT %MW10042.0 *) (* R363 2 M 차종4 내수 *)
    R363_2_M_차종4_러시아 : BOOL; (* AT %MW10042.10 *) (* R363 2 M 차종4 러시아 *)
    R363_2_M_차종4_북미 : BOOL; (* AT %MW10042.2 *) (* R363 2 M 차종4 북미 *)
    R363_2_M_차종4_브라질 : BOOL; (* AT %MW10042.7 *) (* R363 2 M 차종4 브라질 *)
    R363_2_M_차종4_수출 : BOOL; (* AT %MW10042.1 *) (* R363 2 M 차종4 수출 *)
    R363_2_M_차종4_중국 : BOOL; (* AT %MW10042.6 *) (* R363 2 M 차종4 중국 *)
    R363_2_M_차종4_중동 : BOOL; (* AT %MW10042.5 *) (* R363 2 M 차종4 중동 *)
    R363_2_M_차종4_호주 : BOOL; (* AT %MW10042.4 *) (* R363 2 M 차종4 호주 *)
    R363_2_M_차종5_AT : BOOL; (* AT %MW10043.1 *) (* R363 2 M 차종5 AT *)
    R363_2_M_차종5_MT : BOOL; (* AT %MW10043.0 *) (* R363 2 M 차종5 MT *)
    R363_2_M_차종5_SP1 : BOOL; (* AT %MW10043.2 *) (* R363 2 M 차종5 SP1 *)
    R363_2_M_차종6_DSROOF : BOOL; (* AT %MW10043.6 *) (* R363 2 M 차종6 DSROOF *)
    R363_2_M_차종6_SP1 : BOOL; (* AT %MW10043.7 *) (* R363 2 M 차종6 SP1 *)
    R363_2_M_차종6_썬루프 : BOOL; (* AT %MW10043.4 *) (* R363 2 M 차종6 썬루프 *)
    R363_2_M_차종6_일반루프 : BOOL; (* AT %MW10043.3 *) (* R363 2 M 차종6 일반루프 *)
    R363_2_M_차종6_파노라마루프 : BOOL; (* AT %MW10043.5 *) (* R363 2 M 차종6 파노라마루프 *)
    R363_2_M_차종7_DSL : BOOL; (* AT %MW10043.9 *) (* R363 2 M 차종7 DSL *)
    R363_2_M_차종7_GSL : BOOL; (* AT %MW10043.8 *) (* R363 2 M 차종7 GSL *)
    R363_2_M_차종7_SP1 : BOOL; (* AT %MW10043.10 *) (* R363 2 M 차종7 SP1 *)
    R363_2_M_차종7_SP2 : BOOL; (* AT %MW10043.11 *) (* R363 2 M 차종7 SP2 *)
    R363_2_M_차종7_SP3 : BOOL; (* AT %MW10043.12 *) (* R363 2 M 차종7 SP3 *)
    R363_2_M_차종7_SP4 : BOOL; (* AT %MW10043.13 *) (* R363 2 M 차종7 SP4 *)
    R363_2_M_차종7_SP5 : BOOL; (* AT %MW10043.14 *) (* R363 2 M 차종7 SP5 *)
    R363_2_M_차종7_SP6 : BOOL; (* AT %MW10043.15 *) (* R363 2 M 차종7 SP6 *)
    R363_2_M_차종8_2WD : BOOL; (* AT %MW10044.0 *) (* R363 2 M 차종8 2WD *)
    R363_2_M_차종8_4WD : BOOL; (* AT %MW10044.1 *) (* R363 2 M 차종8 4WD *)
    R363_2_M_차종8_SP1 : BOOL; (* AT %MW10044.2 *) (* R363 2 M 차종8 SP1 *)
    R363_2_M_차종9_MPI : BOOL; (* AT %MW10044.3 *) (* R363 2 M 차종9 MPI *)
    R363_2_M_차종9_SP1 : BOOL; (* AT %MW10044.5 *) (* R363 2 M 차종9 SP1 *)
    R363_2_M_차종9_SP10 : BOOL; (* AT %MW10044.14 *) (* R363 2 M 차종9 SP10 *)
    R363_2_M_차종9_SP11 : BOOL; (* AT %MW10044.15 *) (* R363 2 M 차종9 SP11 *)
    R363_2_M_차종9_SP2 : BOOL; (* AT %MW10044.6 *) (* R363 2 M 차종9 SP2 *)
    R363_2_M_차종9_SP3 : BOOL; (* AT %MW10044.7 *) (* R363 2 M 차종9 SP3 *)
    R363_2_M_차종9_SP4 : BOOL; (* AT %MW10044.8 *) (* R363 2 M 차종9 SP4 *)
    R363_2_M_차종9_SP5 : BOOL; (* AT %MW10044.9 *) (* R363 2 M 차종9 SP5 *)
    R363_2_M_차종9_SP6 : BOOL; (* AT %MW10044.10 *) (* R363 2 M 차종9 SP6 *)
    R363_2_M_차종9_SP7 : BOOL; (* AT %MW10044.11 *) (* R363 2 M 차종9 SP7 *)
    R363_2_M_차종9_SP8 : BOOL; (* AT %MW10044.12 *) (* R363 2 M 차종9 SP8 *)
    R363_2_M_차종9_SP9 : BOOL; (* AT %MW10044.13 *) (* R363 2 M 차종9 SP9 *)
    R363_2_M_차종9_T_GDI : BOOL; (* AT %MW10044.4 *) (* R363 2 M 차종9 T GDI *)
    R363_2_M_차종_OPT1_R_RACK_무 : BOOL; (* AT %MW10045.3 *) (* R363 2 M 차종 OPT1 R RACK 무 *)
    R363_2_M_차종_OPT1_R_RACK_유 : BOOL; (* AT %MW10045.2 *) (* R363 2 M 차종 OPT1 R RACK 유 *)
    R363_2_M_차종_OPT1_S_REP_EATER_무 : BOOL; (* AT %MW10045.7 *) (* R363 2 M 차종 OPT1 S REP EATER 무 *)
    R363_2_M_차종_OPT1_S_REP_EATER_유 : BOOL; (* AT %MW10045.6 *) (* R363 2 M 차종 OPT1 S REP EATER 유 *)
    R363_2_M_차종_OPT1_VAN_무 : BOOL; (* AT %MW10045.9 *) (* R363 2 M 차종 OPT1 VAN 무 *)
    R363_2_M_차종_OPT1_VAN_유 : BOOL; (* AT %MW10045.8 *) (* R363 2 M 차종 OPT1 VAN 유 *)
    R363_2_M_차종_OPT1_슬라이딩_무 : BOOL; (* AT %MW10045.1 *) (* R363 2 M 차종 OPT1 슬라이딩 무 *)
    R363_2_M_차종_OPT1_슬라이딩_유 : BOOL; (* AT %MW10045.0 *) (* R363 2 M 차종 OPT1 슬라이딩 유 *)
    R363_2_M_차종_OPT1_폴딩_무 : BOOL; (* AT %MW10045.5 *) (* R363 2 M 차종 OPT1 폴딩 무 *)
    R363_2_M_차종_OPT1_폴딩_유 : BOOL; (* AT %MW10045.4 *) (* R363 2 M 차종 OPT1 폴딩 유 *)
    R363_2_M_차종_무 : BOOL; (* AT %MW1002.3 *)
    R363_2_M_차종_유 : BOOL; (* AT %MW1002.2 *) (* S362_M_공정_차종_보조 *)
    S362_M_BYPASS_보조 : BOOL; (* AT %MW1003.15 *) (* S362 M BYPASS 보조 *)
    S362_M_LC_정상 : BOOL; (* AT %MW1007.5 *) (* S362_M_LC_정상 *)
    S362_M_LH_TURN_1_포지션단 : BOOL; (* AT %MW1104.3 *) (* S362_M_LH_TURN_1_포지션단 *)
    S362_M_LH_TURN_2_포지션단 : BOOL; (* AT %MW1104.4 *) (* S362_M_LH_TURN_2_포지션단 *)
    S362_M_LH_TURN_3_포지션단 : BOOL; (* AT %MW1104.5 *) (* S362_M_LH_TURN_3_포지션단 *)
    S362_M_LH_TURN_4_포지션단 : BOOL; (* AT %MW1104.6 *) (* S362_M_LH_TURN_4_포지션단 *)
    S362_M_MAT_정상 : BOOL; (* AT %MW1007.6 *) (* S362_M_MAT_정상 *)
    S362_M_OP_LC_이상 : BOOL; (* AT %MW1012.0 *) (* S362_M_OP_LC_이상 *)
    S362_M_OP_MAT_이상 : BOOL; (* AT %MW1012.1 *) (* S362_M_OP_MAT_이상 *)
    S362_M_R363_1_실링완료 : BOOL; (* AT %MW1001.2 *)
    S362_M_R363_2_언로딩_완료 : BOOL; (* AT %MW1001.3 *)
    S362_M_RH_TURN_1_포지션단 : BOOL; (* AT %MW1112.3 *) (* S362_M_RH_TURN_1_포지션단 *)
    S362_M_RH_TURN_2_포지션단 : BOOL; (* AT %MW1112.4 *) (* S362_M_RH_TURN_2_포지션단 *)
    S362_M_RH_TURN_3_포지션단 : BOOL; (* AT %MW1112.5 *) (* S362_M_RH_TURN_3_포지션단 *)
    S362_M_RH_TURN_4_포지션단 : BOOL; (* AT %MW1112.6 *) (* S362_M_RH_TURN_4_포지션단 *)
    S362_M_SAFETY_불간섭 : BOOL; (* AT %MW1004.4 *) (* S362_M_SAFETY_불간섭 *)
    S362_M_SEQ : WORD; (* AT %MW10100 *) (* S362 M SEQ *)
    S362_M_SLD_LOCK_전진단 : BOOL; (* AT %MW1102.3 *) (* S362_M_SLD_LOCK_전진단 *)
    S362_M_SLD_LOCK_후진단 : BOOL; (* AT %MW1102.4 *) (* S362_M_SLD_LOCK_후진단 *)
    S362_M_SLIDE_전진단 : BOOL; (* AT %MW1101.3 *) (* S362_M_SLIDE_전진단 *)
    S362_M_SLIDE_후진단 : BOOL; (* AT %MW1101.4 *) (* S362_M_SLIDE_후진단 *)
    S362_M_TURN_LOCK_전진단 : BOOL; (* AT %MW1100.3 *) (* S362_M_TURN_LOCK_전진단 *)
    S362_M_TURN_LOCK_후진단 : BOOL; (* AT %MW1100.4 *) (* S362_M_TURN_LOCK_후진단 *)
    S362_M_공정_AX_RAIL_제품감지_무 : BOOL; (* AT %MW1001.13 *) (* S362 M 공정 AX RAIL 제품감지 무 *)
    S362_M_공정_AX_RAIL_제품감지_유 : BOOL; (* AT %MW1001.12 *) (* S362 M 공정 AX RAIL 제품감지 유 *)
    S362_M_공정_AX_공용_제품감지_무 : BOOL; (* AT %MW1001.7 *) (* S362 M 공정 AX 공용 제품감지 무 *)
    S362_M_공정_AX_공용_제품감지_유 : BOOL; (* AT %MW1001.6 *) (* S362 M 공정 AX 공용 제품감지 유 *)
    S362_M_공정_AX_썬루프_제품감지_무 : BOOL; (* AT %MW1001.11 *) (* S362 M 공정 AX 썬루프 제품감지 무 *)
    S362_M_공정_AX_썬루프_제품감지_유 : BOOL; (* AT %MW1001.10 *) (* S362 M 공정 AX 썬루프 제품감지 유 *)
    S362_M_공정_AX_일반루프_제품감지_무 : BOOL; (* AT %MW1001.9 *) (* S362 M 공정 AX 일반루프 제품감지 무 *)
    S362_M_공정_AX_일반루프_제품감지_유 : BOOL; (* AT %MW1001.8 *) (* S362 M 공정 AX 일반루프 제품감지 유 *)
    S362_M_공정_불간섭 : BOOL; (* AT %MW1004.1 *) (* S362_M_공정_불간섭 *)
    S362_M_공정_원위치 : BOOL; (* AT %MW1004.0 *) (* S362_M_공정_원위치 *)
    S362_M_공정_제품감지_무 : BOOL; (* AT %MW1001.5 *) (* S362_M_공정_제품감지_무 *)
    S362_M_공정_제품감지_유 : BOOL; (* AT %MW1001.4 *) (* S362_M_공정_제품감지_유 *)
    S362_M_공정_차종_무 : BOOL; (* AT %MW1002.1 *) (* S362_M_공정_차종_무 *)
    S362_M_공정_차종_유 : BOOL; (* AT %MW1002.0 *) (* S362_M_공정_차종_유 *)
    S362_M_수동모드 : BOOL; (* AT %MW1000.3 *) (* S362 선택 수동모드 *)
    S362_M_운전준비_ON : BOOL; (* AT %MW1000.0 *) (* S362 운전준비 ON *)
    S362_M_자동_START : BOOL; (* AT %MW1000.5 *) (* S362 자동운전중 *)
    S362_M_자동_운전중 : BOOL; (* AT %MW1000.4 *) (* S362 자동운전중 *)
    S362_M_자동모드 : BOOL; (* AT %MW1000.1 *) (* S362 선택 자동모드 *)
    S362_M_작업_완료 : BOOL; (* AT %MW1001.0 *) (* S362_M_작업_완료 *)
    S362_M_작업완료_SET_PLS : BOOL; (* AT %MW1000.8 *) (* S362 M 작업완료 SET PLS *)
    S362_M_작업완료_리셋_PLS : BOOL; (* AT %MW1000.9 *) (* S362 M 작업완료 리셋 PLS *)
    S362_M_작업자_작업_가능 : BOOL; (* AT %MW1004.8 *) (* S362 M 작업자 작업 가능 *)
    S362_M_작업자_작업완료 : BOOL; (* AT %MW1001.1 *)
    S362_M_차종1_AX : BOOL; (* AT %MW10101.0 *) (* S362 M 차종1 AX *)
    S362_M_차종1_B : BOOL; (* AT %MW10101.1 *) (* S362 M 차종1 B *)
    S362_M_차종1_C : BOOL; (* AT %MW10101.2 *) (* S362 M 차종1 C *)
    S362_M_차종1_D : BOOL; (* AT %MW10101.3 *) (* S362 M 차종1 D *)
    S362_M_차종1_E : BOOL; (* AT %MW10101.4 *) (* S362 M 차종1 E *)
    S362_M_차종1_F : BOOL; (* AT %MW10101.5 *) (* S362 M 차종1 F *)
    S362_M_차종1_G : BOOL; (* AT %MW10101.6 *) (* S362 M 차종1 G *)
    S362_M_차종1_H : BOOL; (* AT %MW10101.7 *) (* S362 M 차종1 H *)
    S362_M_차종2_3DR : BOOL; (* AT %MW10101.8 *) (* S362 M 차종2 3DR *)
    S362_M_차종2_4DR : BOOL; (* AT %MW10101.9 *) (* S362 M 차종2 4DR *)
    S362_M_차종2_5DR : BOOL; (* AT %MW10101.10 *) (* S362 M 차종2 5DR *)
    S362_M_차종2_SP1 : BOOL; (* AT %MW10101.12 *) (* S362 M 차종2 SP1 *)
    S362_M_차종2_SP2 : BOOL; (* AT %MW10101.13 *) (* S362 M 차종2 SP2 *)
    S362_M_차종2_WGN : BOOL; (* AT %MW10101.11 *) (* S362 M 차종2 WGN *)
    S362_M_차종3_LHD : BOOL; (* AT %MW10101.14 *) (* S362 M 차종3 LHD *)
    S362_M_차종3_RHD : BOOL; (* AT %MW10101.15 *) (* S362 M 차종3 RHD *)
    S362_M_차종4_EEC : BOOL; (* AT %MW10102.3 *) (* S362 M 차종4 EEC *)
    S362_M_차종4_SP1 : BOOL; (* AT %MW10102.8 *) (* S362 M 차종4 SP1 *)
    S362_M_차종4_SP2 : BOOL; (* AT %MW10102.9 *) (* S362 M 차종4 SP2 *)
    S362_M_차종4_SP3 : BOOL; (* AT %MW10102.11 *) (* S362 M 차종4 SP3 *)
    S362_M_차종4_SP4 : BOOL; (* AT %MW10102.12 *) (* S362 M 차종4 SP4 *)
    S362_M_차종4_SP5 : BOOL; (* AT %MW10102.13 *) (* S362 M 차종4 SP5 *)
    S362_M_차종4_SP6 : BOOL; (* AT %MW10102.14 *) (* S362 M 차종4 SP6 *)
    S362_M_차종4_SP7 : BOOL; (* AT %MW10102.15 *) (* S362 M 차종4 SP7 *)
    S362_M_차종4_내수 : BOOL; (* AT %MW10102.0 *) (* S362 M 차종4 내수 *)
    S362_M_차종4_러시아 : BOOL; (* AT %MW10102.10 *) (* S362 M 차종4 러시아 *)
    S362_M_차종4_북미 : BOOL; (* AT %MW10102.2 *) (* S362 M 차종4 북미 *)
    S362_M_차종4_브라질 : BOOL; (* AT %MW10102.7 *) (* S362 M 차종4 브라질 *)
    S362_M_차종4_수출 : BOOL; (* AT %MW10102.1 *) (* S362 M 차종4 수출 *)
    S362_M_차종4_중국 : BOOL; (* AT %MW10102.6 *) (* S362 M 차종4 중국 *)
    S362_M_차종4_중동 : BOOL; (* AT %MW10102.5 *) (* S362 M 차종4 중동 *)
    S362_M_차종4_호주 : BOOL; (* AT %MW10102.4 *) (* S362 M 차종4 호주 *)
    S362_M_차종5_AT : BOOL; (* AT %MW10103.1 *) (* S362 M 차종5 AT *)
    S362_M_차종5_MT : BOOL; (* AT %MW10103.0 *) (* S362 M 차종5 MT *)
    S362_M_차종5_SP1 : BOOL; (* AT %MW10103.2 *) (* S362 M 차종5 SP1 *)
    S362_M_차종6_DSROOF : BOOL; (* AT %MW10103.6 *) (* S362 M 차종6 DSROOF *)
    S362_M_차종6_SP1 : BOOL; (* AT %MW10103.7 *) (* S362 M 차종6 SP1 *)
    S362_M_차종6_썬루프 : BOOL; (* AT %MW10103.4 *) (* S362 M 차종6 썬루프 *)
    S362_M_차종6_일반루프 : BOOL; (* AT %MW10103.3 *) (* S362 M 차종6 일반루프 *)
    S362_M_차종6_파노라마루프 : BOOL; (* AT %MW10103.5 *) (* S362 M 차종6 파노라마루프 *)
    S362_M_차종7_DSL : BOOL; (* AT %MW10103.9 *) (* S362 M 차종7 DSL *)
    S362_M_차종7_GSL : BOOL; (* AT %MW10103.8 *) (* S362 M 차종7 GSL *)
    S362_M_차종7_SP1 : BOOL; (* AT %MW10103.10 *) (* S362 M 차종7 SP1 *)
    S362_M_차종7_SP2 : BOOL; (* AT %MW10103.11 *) (* S362 M 차종7 SP2 *)
    S362_M_차종7_SP3 : BOOL; (* AT %MW10103.12 *) (* S362 M 차종7 SP3 *)
    S362_M_차종7_SP4 : BOOL; (* AT %MW10103.13 *) (* S362 M 차종7 SP4 *)
    S362_M_차종7_SP5 : BOOL; (* AT %MW10103.14 *) (* S362 M 차종7 SP5 *)
    S362_M_차종7_SP6 : BOOL; (* AT %MW10103.15 *) (* S362 M 차종7 SP6 *)
    S362_M_차종8_2WD : BOOL; (* AT %MW10104.0 *) (* S362 M 차종8 2WD *)
    S362_M_차종8_4WD : BOOL; (* AT %MW10104.1 *) (* S362 M 차종8 4WD *)
    S362_M_차종8_SP1 : BOOL; (* AT %MW10104.2 *) (* S362 M 차종8 SP1 *)
    S362_M_차종9_MPI : BOOL; (* AT %MW10104.3 *) (* S362 M 차종9 MPI *)
    S362_M_차종9_SP1 : BOOL; (* AT %MW10104.5 *) (* S362 M 차종9 SP1 *)
    S362_M_차종9_SP10 : BOOL; (* AT %MW10104.14 *) (* S362 M 차종9 SP10 *)
    S362_M_차종9_SP11 : BOOL; (* AT %MW10104.15 *) (* S362 M 차종9 SP11 *)
    S362_M_차종9_SP2 : BOOL; (* AT %MW10104.6 *) (* S362 M 차종9 SP2 *)
    S362_M_차종9_SP3 : BOOL; (* AT %MW10104.7 *) (* S362 M 차종9 SP3 *)
    S362_M_차종9_SP4 : BOOL; (* AT %MW10104.8 *) (* S362 M 차종9 SP4 *)
    S362_M_차종9_SP5 : BOOL; (* AT %MW10104.9 *) (* S362 M 차종9 SP5 *)
    S362_M_차종9_SP6 : BOOL; (* AT %MW10104.10 *) (* S362 M 차종9 SP6 *)
    S362_M_차종9_SP7 : BOOL; (* AT %MW10104.11 *) (* S362 M 차종9 SP7 *)
    S362_M_차종9_SP8 : BOOL; (* AT %MW10104.12 *) (* S362 M 차종9 SP8 *)
    S362_M_차종9_SP9 : BOOL; (* AT %MW10104.13 *) (* S362 M 차종9 SP9 *)
    S362_M_차종9_T_GDI : BOOL; (* AT %MW10104.4 *) (* S362 M 차종9 T GDI *)
    S362_M_차종_OPT1_R_RACK_무 : BOOL; (* AT %MW10105.3 *) (* S362 M 차종 OPT1 R RACK 무 *)
    S362_M_차종_OPT1_R_RACK_유 : BOOL; (* AT %MW10105.2 *) (* S362 M 차종 OPT1 R RACK 유 *)
    S362_M_차종_OPT1_S_REP_EATER_무 : BOOL; (* AT %MW10105.7 *) (* S362 M 차종 OPT1 S REP EATER 무 *)
    S362_M_차종_OPT1_S_REP_EATER_유 : BOOL; (* AT %MW10105.6 *) (* S362 M 차종 OPT1 S REP EATER 유 *)
    S362_M_차종_OPT1_VAN_무 : BOOL; (* AT %MW10105.9 *) (* S362 M 차종 OPT1 VAN 무 *)
    S362_M_차종_OPT1_VAN_유 : BOOL; (* AT %MW10105.8 *) (* S362 M 차종 OPT1 VAN 유 *)
    S362_M_차종_OPT1_슬라이딩_무 : BOOL; (* AT %MW10105.1 *) (* S362 M 차종 OPT1 슬라이딩 무 *)
    S362_M_차종_OPT1_슬라이딩_유 : BOOL; (* AT %MW10105.0 *) (* S362 M 차종 OPT1 슬라이딩 유 *)
    S362_M_차종_OPT1_폴딩_무 : BOOL; (* AT %MW10105.5 *) (* S362 M 차종 OPT1 폴딩 무 *)
    S362_M_차종_OPT1_폴딩_유 : BOOL; (* AT %MW10105.4 *) (* S362 M 차종 OPT1 폴딩 유 *)
    S362_M_차종_공대차 : BOOL; (* AT %MW10110.12 *) (* S362 M 차종 공대차 *)
    S362_M_차종_공차 : BOOL; (* AT %MW10110.10 *) (* S362 M 차종 공차 *)
    S362_M_차종_불량차 : BOOL; (* AT %MW10110.11 *) (* S362 M 차종 불량차 *)
    S362_M_총괄_이상 : BOOL; (* AT %MW1009.0 *) (* S362_M_총괄_이상 *)
    S364_M_총괄_이상 : BOOL; (* AT %MW2009.0 *) (* S364_M_총괄_이상 *)
    전체_M_GATE_자동기동 : BOOL; (* AT %MW308.1 *) (* 전체_M_자동_운전 *)
    전체_M_이상_리셋 : BOOL; (* AT %MW308.2 *) (* ALL공정 PB 이상리셋 *)
    전체_라인_M_총괄_SAFETY_이상 : BOOL; (* AT %MW300.2 *) (* ALL공정 SAFETY  이상총괄 *)
    전체_라인_M_총괄_공기압_이상 : BOOL; (* AT %MW300.3 *) (* ALL공정 공기압 이상총괄 *)
    전체_라인_M_총괄_비상정지_이상 : BOOL; (* AT %MW300.1 *) (* ALL공정 비상정지 이상총괄 *)
    전체_라인_M_총괄_이상 : BOOL; (* AT %MW300.0 *) (* ALL공정 총괄이상 *)
END_VAR
VAR
    _t1 : BOOL;
    _t2 : BOOL;
    _e3 : R_TRIG;
    _p4 : BOOL;
END_VAR

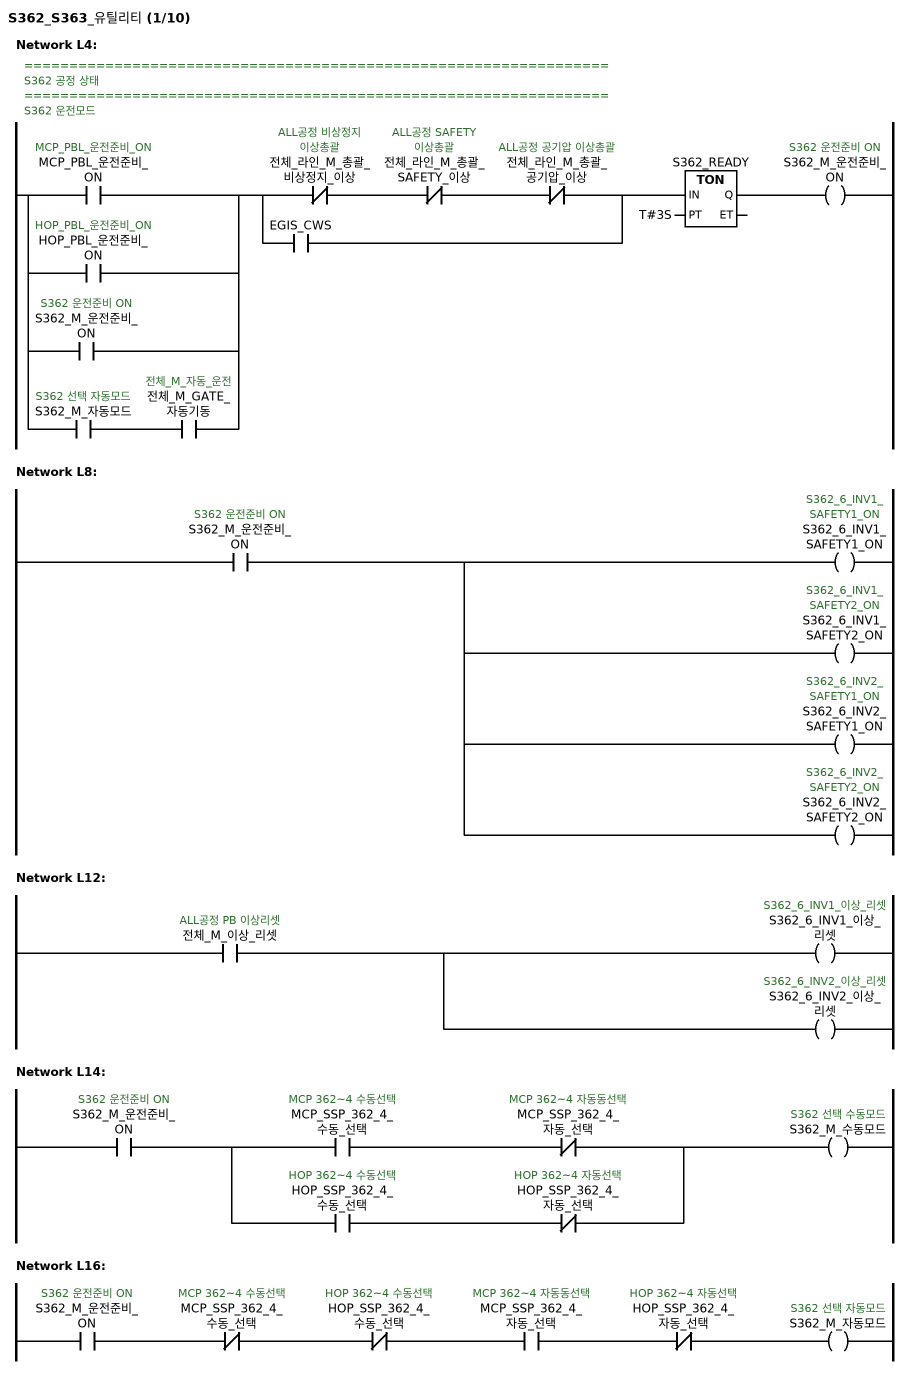
(* ================================================================= *)
(* S362 공정 상태 *)
(* ================================================================= *)
(* S362 운전모드 *)
(* Rung L4 *)
S362_READY(IN := (MCP_PBL_운전준비_ON OR HOP_PBL_운전준비_ON OR S362_M_운전준비_ON OR (S362_M_자동모드 AND 전체_M_GATE_자동기동)) AND ((NOT 전체_라인_M_총괄_비상정지_이상 AND NOT 전체_라인_M_총괄_SAFETY_이상 AND NOT 전체_라인_M_총괄_공기압_이상) OR EGIS_CWS), PT := T#3S);
S362_M_운전준비_ON := S362_READY.Q;
(* Rung L8 *)
S362_6_INV1_SAFETY1_ON := S362_M_운전준비_ON;
S362_6_INV1_SAFETY2_ON := S362_M_운전준비_ON;
S362_6_INV2_SAFETY1_ON := S362_M_운전준비_ON;
S362_6_INV2_SAFETY2_ON := S362_M_운전준비_ON;
(* Rung L12 *)
S362_6_INV1_이상_리셋 := 전체_M_이상_리셋;
S362_6_INV2_이상_리셋 := 전체_M_이상_리셋;
(* Rung L14 *)
S362_M_수동모드 := S362_M_운전준비_ON AND ((MCP_SSP_362_4_수동_선택 AND NOT MCP_SSP_362_4_자동_선택) OR (HOP_SSP_362_4_수동_선택 AND NOT HOP_SSP_362_4_자동_선택));
(* Rung L16 *)
S362_M_자동모드 := S362_M_운전준비_ON AND NOT MCP_SSP_362_4_수동_선택 AND NOT HOP_SSP_362_4_수동_선택 AND MCP_SSP_362_4_자동_선택 AND NOT HOP_SSP_362_4_자동_선택;

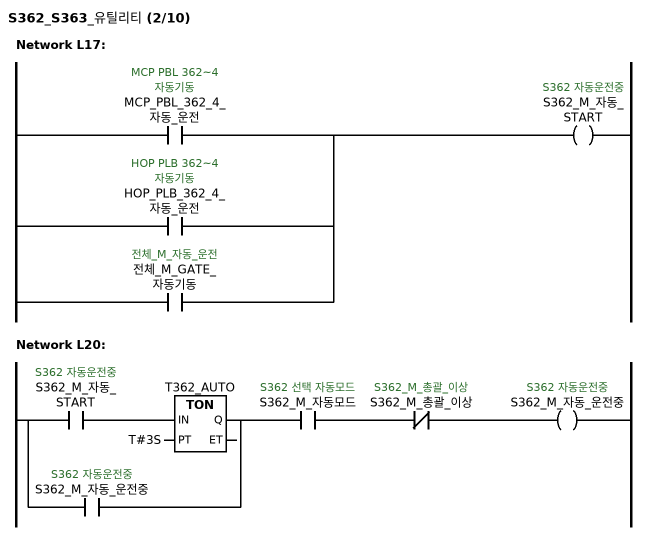
(* Rung L17 *)
S362_M_자동_START := MCP_PBL_362_4_자동_운전 OR HOP_PLB_362_4_자동_운전 OR 전체_M_GATE_자동기동;
(* Rung L20 *)
T362_AUTO(IN := S362_M_자동_START, PT := T#3S);
S362_M_자동_운전중 := (T362_AUTO.Q OR S362_M_자동_운전중) AND S362_M_자동모드 AND NOT S362_M_총괄_이상;

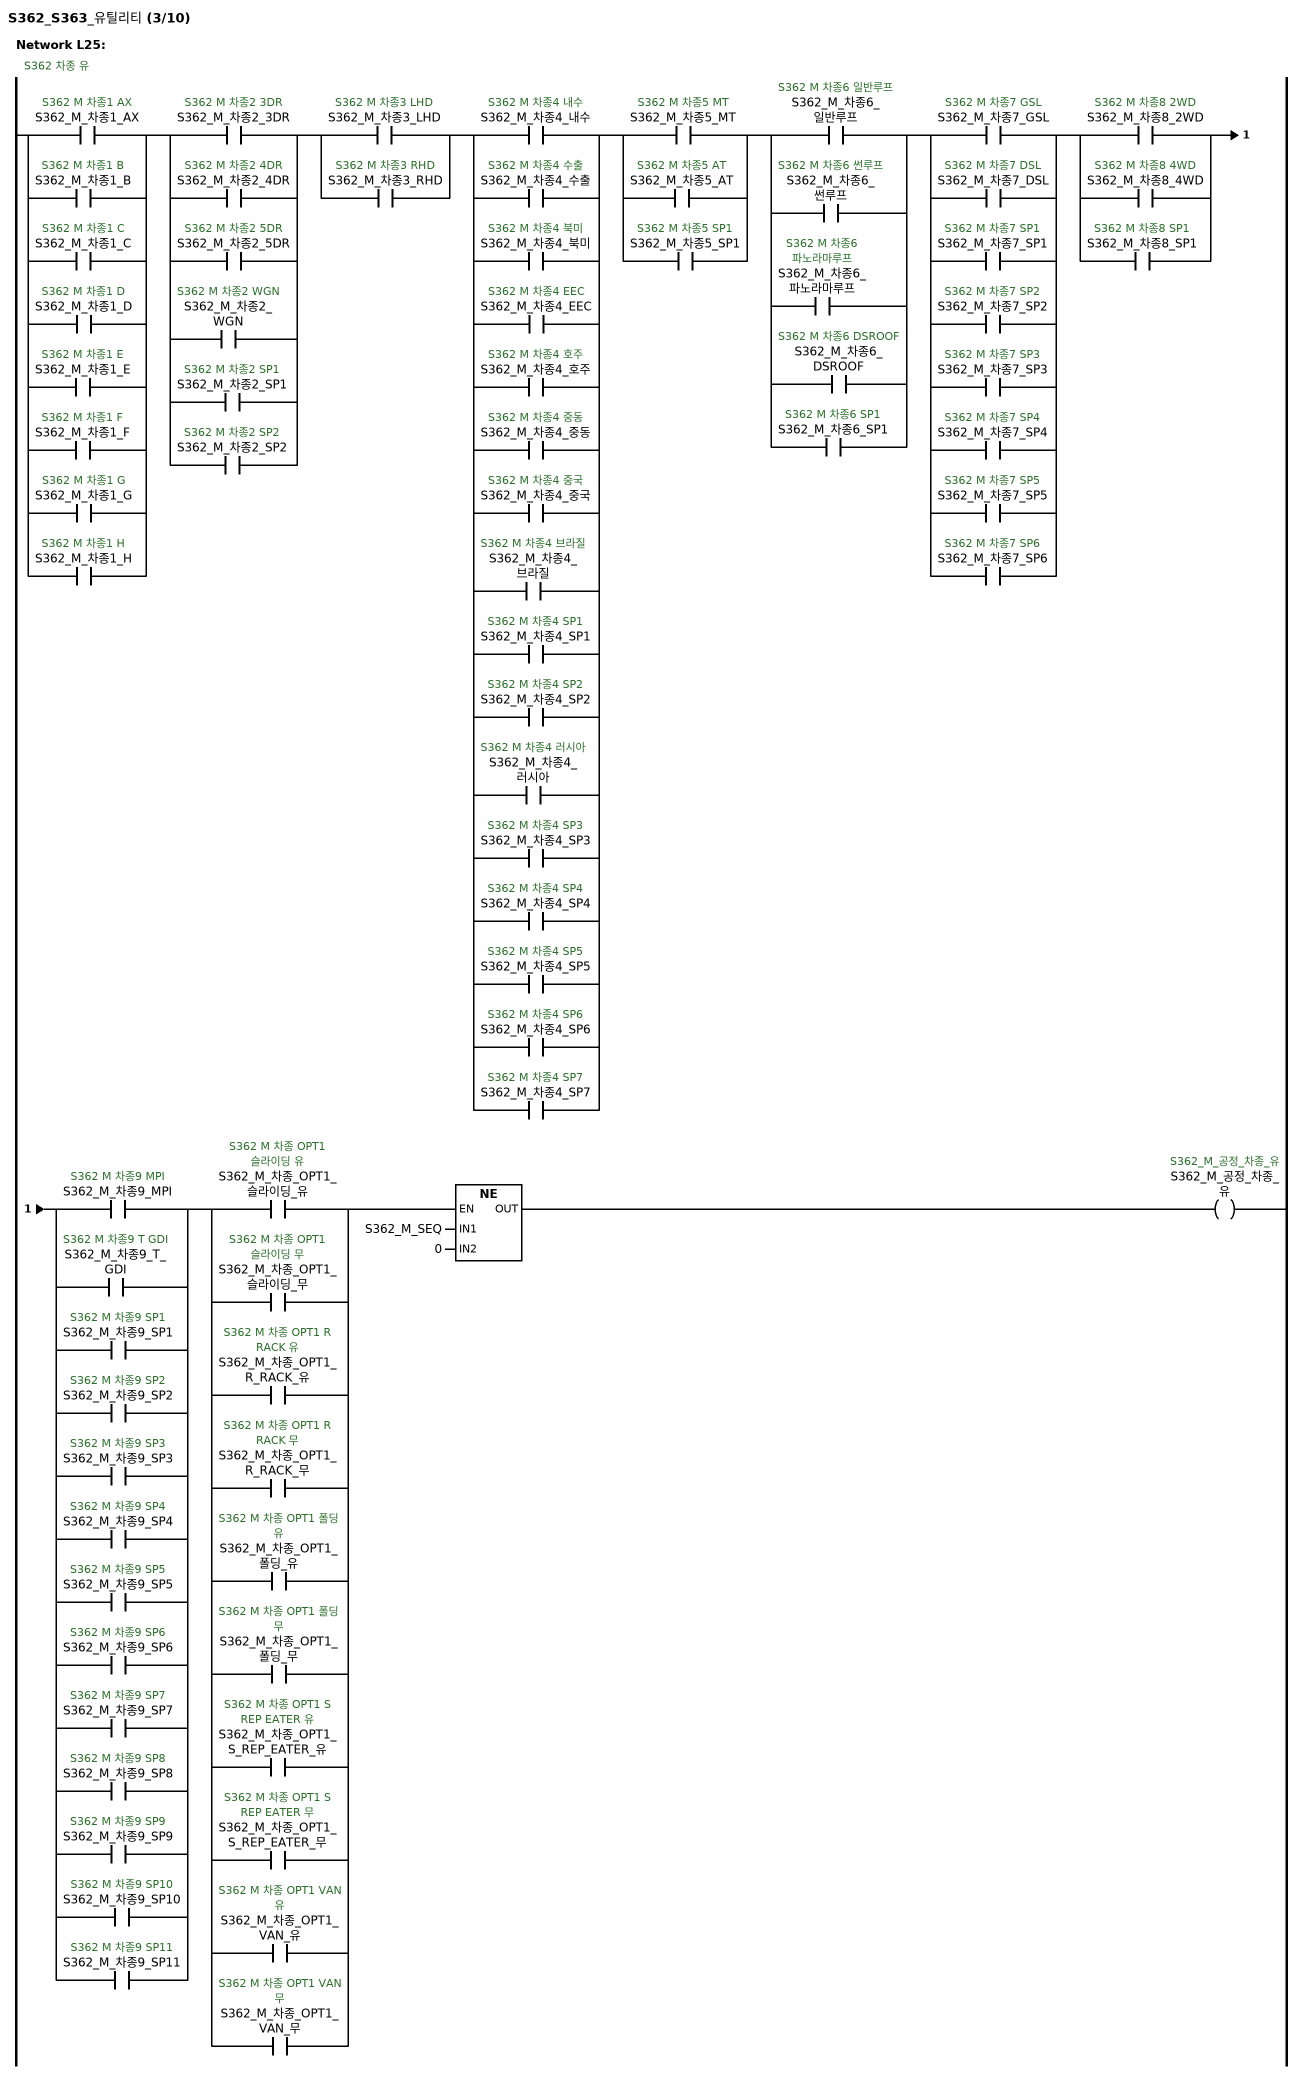
(* S362 차종 유 *)
(* Rung L25 *)
IF (S362_M_차종1_AX OR S362_M_차종1_B OR S362_M_차종1_C OR S362_M_차종1_D OR S362_M_차종1_E OR S362_M_차종1_F OR S362_M_차종1_G OR S362_M_차종1_H) AND (S362_M_차종2_3DR OR S362_M_차종2_4DR OR S362_M_차종2_5DR OR S362_M_차종2_WGN OR S362_M_차종2_SP1 OR S362_M_차종2_SP2) AND (S362_M_차종3_LHD OR S362_M_차종3_RHD) AND (S362_M_차종4_내수 OR S362_M_차종4_수출 OR S362_M_차종4_북미 OR S362_M_차종4_EEC OR S362_M_차종4_호주 OR S362_M_차종4_중동 OR S362_M_차종4_중국 OR S362_M_차종4_브라질 OR S362_M_차종4_SP1 OR S362_M_차종4_SP2 OR S362_M_차종4_러시아 OR S362_M_차종4_SP3 OR S362_M_차종4_SP4 OR S362_M_차종4_SP5 OR S362_M_차종4_SP6 OR S362_M_차종4_SP7) AND (S362_M_차종5_MT OR S362_M_차종5_AT OR S362_M_차종5_SP1) AND (S362_M_차종6_일반루프 OR S362_M_차종6_썬루프 OR S362_M_차종6_파노라마루프 OR S362_M_차종6_DSROOF OR S362_M_차종6_SP1) AND (S362_M_차종7_GSL OR S362_M_차종7_DSL OR S362_M_차종7_SP1 OR S362_M_차종7_SP2 OR S362_M_차종7_SP3 OR S362_M_차종7_SP4 OR S362_M_차종7_SP5 OR S362_M_차종7_SP6) AND (S362_M_차종8_2WD OR S362_M_차종8_4WD OR S362_M_차종8_SP1) AND (S362_M_차종9_MPI OR S362_M_차종9_T_GDI OR S362_M_차종9_SP1 OR S362_M_차종9_SP2 OR S362_M_차종9_SP3 OR S362_M_차종9_SP4 OR S362_M_차종9_SP5 OR S362_M_차종9_SP6 OR S362_M_차종9_SP7 OR S362_M_차종9_SP8 OR S362_M_차종9_SP9 OR S362_M_차종9_SP10 OR S362_M_차종9_SP11) AND (S362_M_차종_OPT1_슬라이딩_유 OR S362_M_차종_OPT1_슬라이딩_무 OR S362_M_차종_OPT1_R_RACK_유 OR S362_M_차종_OPT1_R_RACK_무 OR S362_M_차종_OPT1_폴딩_유 OR S362_M_차종_OPT1_폴딩_무 OR S362_M_차종_OPT1_S_REP_EATER_유 OR S362_M_차종_OPT1_S_REP_EATER_무 OR S362_M_차종_OPT1_VAN_유 OR S362_M_차종_OPT1_VAN_무) THEN
    _t1 := S362_M_SEQ <> 0;
END_IF;
S362_M_공정_차종_유 := _t1;

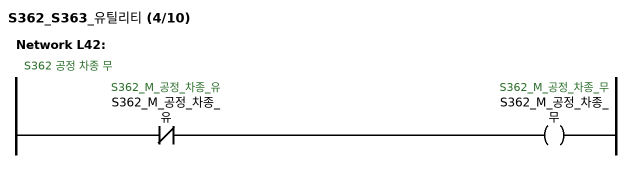
(* S362 공정 차종 무 *)
(* Rung L42 *)
S362_M_공정_차종_무 := NOT S362_M_공정_차종_유;

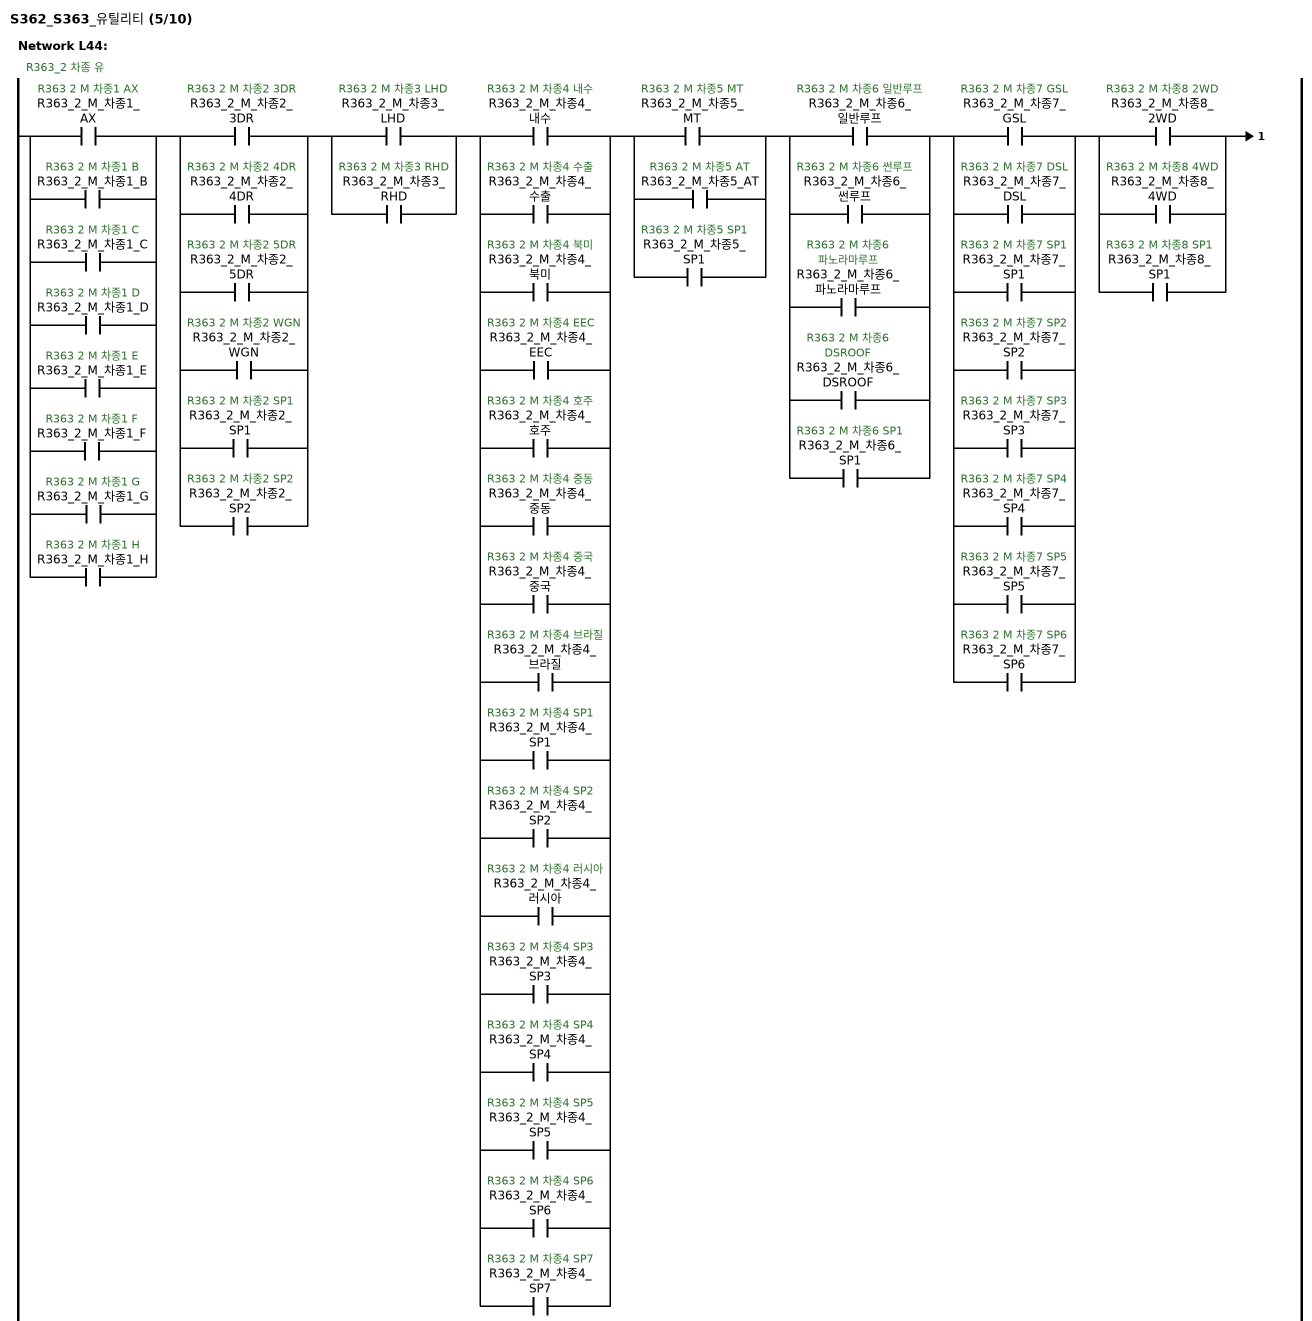

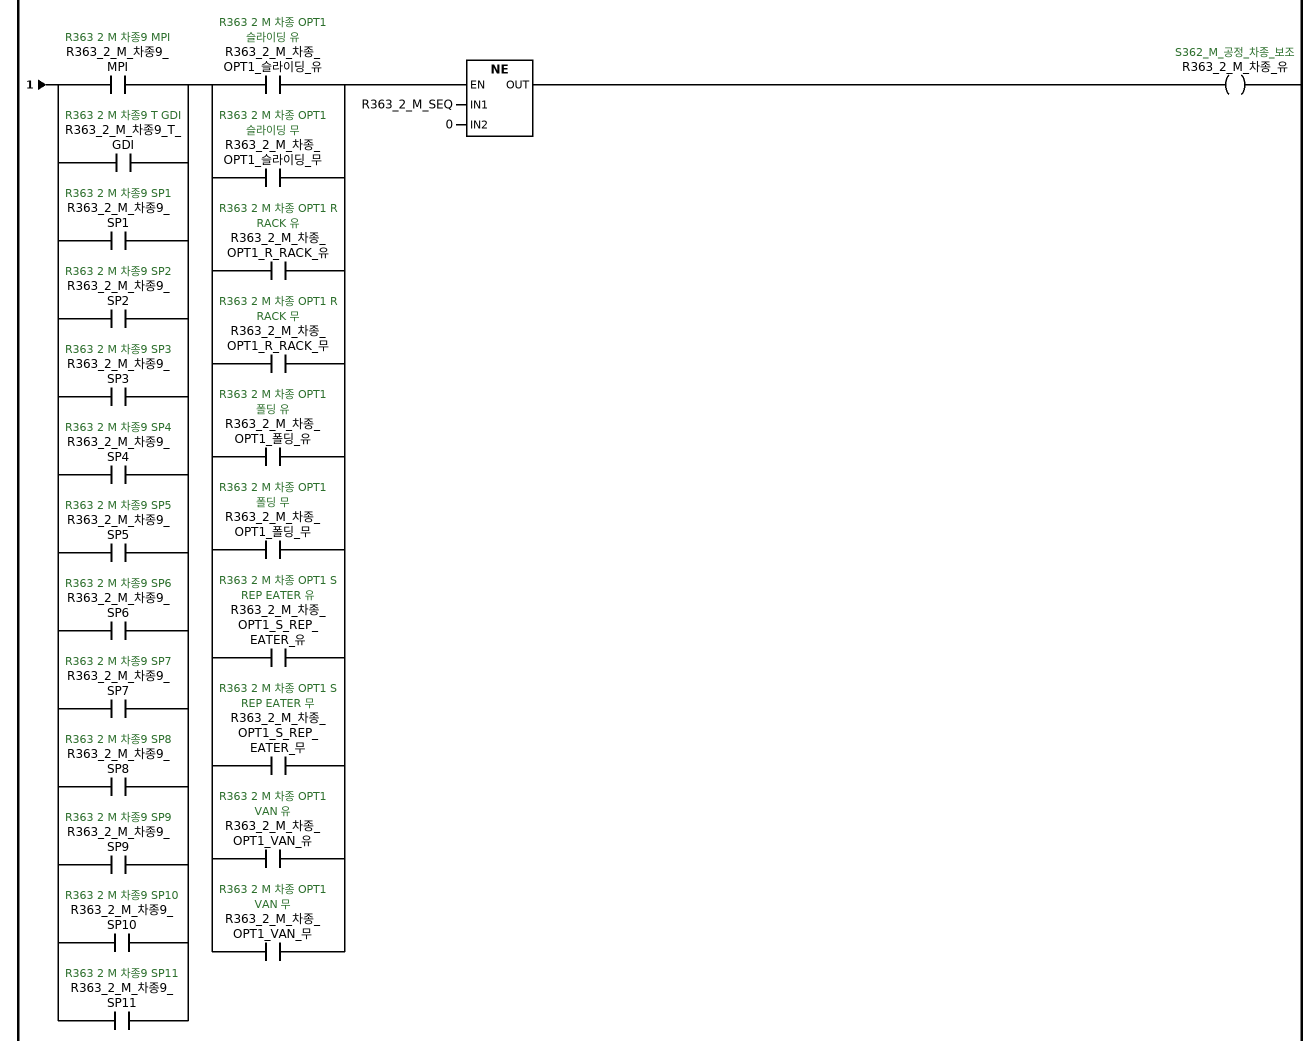
(* R363_2 차종 유 *)
(* Rung L44 *)
IF (R363_2_M_차종1_AX OR R363_2_M_차종1_B OR R363_2_M_차종1_C OR R363_2_M_차종1_D OR R363_2_M_차종1_E OR R363_2_M_차종1_F OR R363_2_M_차종1_G OR R363_2_M_차종1_H) AND (R363_2_M_차종2_3DR OR R363_2_M_차종2_4DR OR R363_2_M_차종2_5DR OR R363_2_M_차종2_WGN OR R363_2_M_차종2_SP1 OR R363_2_M_차종2_SP2) AND (R363_2_M_차종3_LHD OR R363_2_M_차종3_RHD) AND (R363_2_M_차종4_내수 OR R363_2_M_차종4_수출 OR R363_2_M_차종4_북미 OR R363_2_M_차종4_EEC OR R363_2_M_차종4_호주 OR R363_2_M_차종4_중동 OR R363_2_M_차종4_중국 OR R363_2_M_차종4_브라질 OR R363_2_M_차종4_SP1 OR R363_2_M_차종4_SP2 OR R363_2_M_차종4_러시아 OR R363_2_M_차종4_SP3 OR R363_2_M_차종4_SP4 OR R363_2_M_차종4_SP5 OR R363_2_M_차종4_SP6 OR R363_2_M_차종4_SP7) AND (R363_2_M_차종5_MT OR R363_2_M_차종5_AT OR R363_2_M_차종5_SP1) AND (R363_2_M_차종6_일반루프 OR R363_2_M_차종6_썬루프 OR R363_2_M_차종6_파노라마루프 OR R363_2_M_차종6_DSROOF OR R363_2_M_차종6_SP1) AND (R363_2_M_차종7_GSL OR R363_2_M_차종7_DSL OR R363_2_M_차종7_SP1 OR R363_2_M_차종7_SP2 OR R363_2_M_차종7_SP3 OR R363_2_M_차종7_SP4 OR R363_2_M_차종7_SP5 OR R363_2_M_차종7_SP6) AND (R363_2_M_차종8_2WD OR R363_2_M_차종8_4WD OR R363_2_M_차종8_SP1) AND (R363_2_M_차종9_MPI OR R363_2_M_차종9_T_GDI OR R363_2_M_차종9_SP1 OR R363_2_M_차종9_SP2 OR R363_2_M_차종9_SP3 OR R363_2_M_차종9_SP4 OR R363_2_M_차종9_SP5 OR R363_2_M_차종9_SP6 OR R363_2_M_차종9_SP7 OR R363_2_M_차종9_SP8 OR R363_2_M_차종9_SP9 OR R363_2_M_차종9_SP10 OR R363_2_M_차종9_SP11) AND (R363_2_M_차종_OPT1_슬라이딩_유 OR R363_2_M_차종_OPT1_슬라이딩_무 OR R363_2_M_차종_OPT1_R_RACK_유 OR R363_2_M_차종_OPT1_R_RACK_무 OR R363_2_M_차종_OPT1_폴딩_유 OR R363_2_M_차종_OPT1_폴딩_무 OR R363_2_M_차종_OPT1_S_REP_EATER_유 OR R363_2_M_차종_OPT1_S_REP_EATER_무 OR R363_2_M_차종_OPT1_VAN_유 OR R363_2_M_차종_OPT1_VAN_무) THEN
    _t2 := R363_2_M_SEQ <> 0;
END_IF;
R363_2_M_차종_유 := _t2;

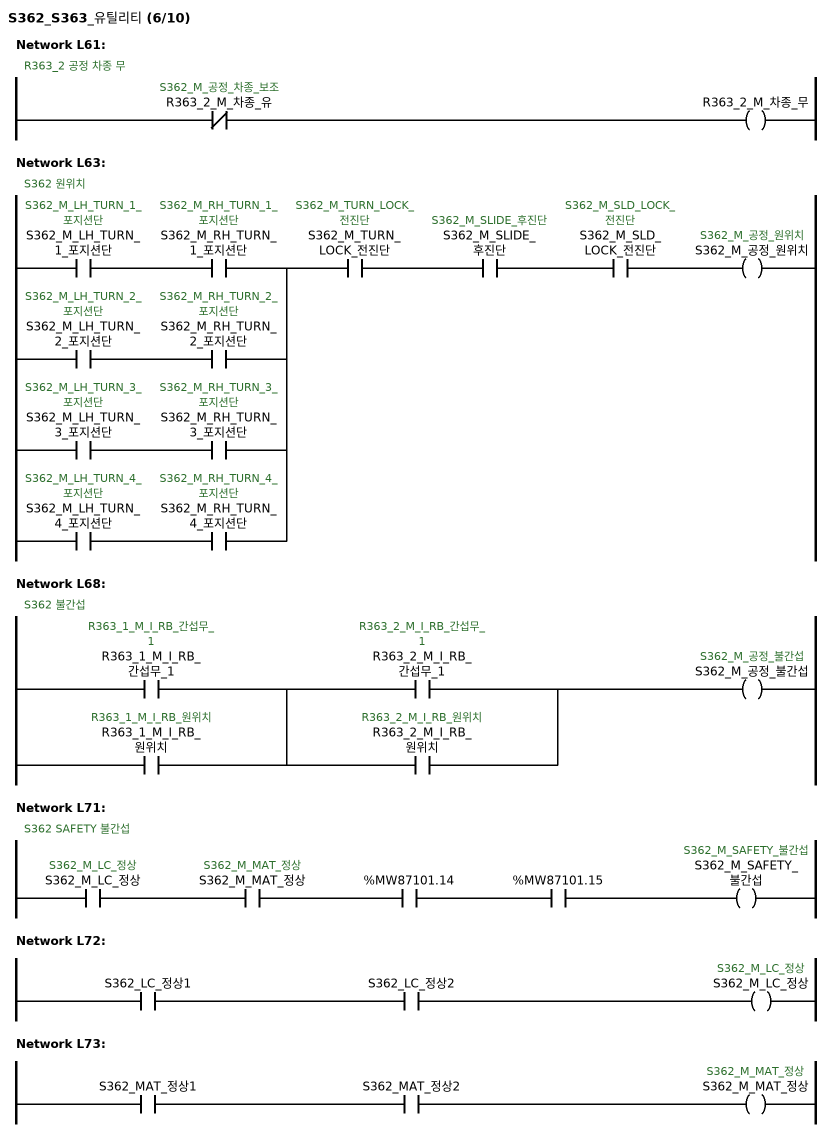
(* R363_2 공정 차종 무 *)
(* Rung L61 *)
R363_2_M_차종_무 := NOT R363_2_M_차종_유;
(* S362 원위치 *)
(* Rung L63 *)
S362_M_공정_원위치 := ((S362_M_LH_TURN_1_포지션단 AND S362_M_RH_TURN_1_포지션단) OR (S362_M_LH_TURN_2_포지션단 AND S362_M_RH_TURN_2_포지션단) OR (S362_M_LH_TURN_3_포지션단 AND S362_M_RH_TURN_3_포지션단) OR (S362_M_LH_TURN_4_포지션단 AND S362_M_RH_TURN_4_포지션단)) AND S362_M_TURN_LOCK_전진단 AND S362_M_SLIDE_후진단 AND S362_M_SLD_LOCK_전진단;
(* S362 불간섭 *)
(* Rung L68 *)
S362_M_공정_불간섭 := (R363_1_M_I_RB_간섭무_1 OR R363_1_M_I_RB_원위치) AND (R363_2_M_I_RB_간섭무_1 OR R363_2_M_I_RB_원위치);
(* S362 SAFETY 불간섭 *)
(* Rung L71 *)
S362_M_SAFETY_불간섭 := S362_M_LC_정상 AND S362_M_MAT_정상 AND %MW87101.14 AND %MW87101.15;
(* Rung L72 *)
S362_M_LC_정상 := S362_LC_정상1 AND S362_LC_정상2;
(* Rung L73 *)
S362_M_MAT_정상 := S362_MAT_정상1 AND S362_MAT_정상2;

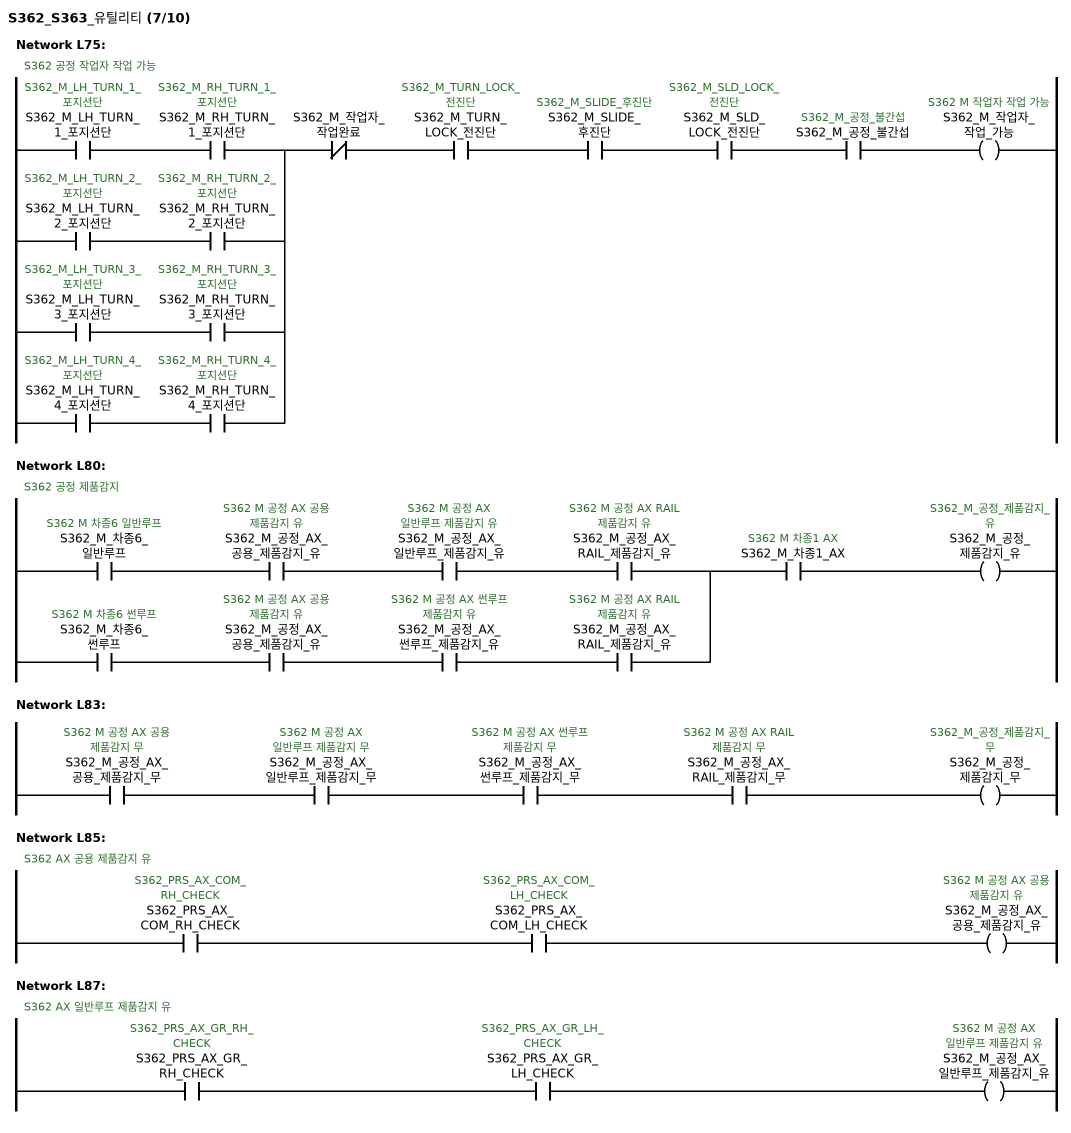
(* S362 공정 작업자 작업 가능 *)
(* Rung L75 *)
S362_M_작업자_작업_가능 := ((S362_M_LH_TURN_1_포지션단 AND S362_M_RH_TURN_1_포지션단) OR (S362_M_LH_TURN_2_포지션단 AND S362_M_RH_TURN_2_포지션단) OR (S362_M_LH_TURN_3_포지션단 AND S362_M_RH_TURN_3_포지션단) OR (S362_M_LH_TURN_4_포지션단 AND S362_M_RH_TURN_4_포지션단)) AND NOT S362_M_작업자_작업완료 AND S362_M_TURN_LOCK_전진단 AND S362_M_SLIDE_후진단 AND S362_M_SLD_LOCK_전진단 AND S362_M_공정_불간섭;
(* S362 공정 제품감지 *)
(* Rung L80 *)
S362_M_공정_제품감지_유 := ((S362_M_차종6_일반루프 AND S362_M_공정_AX_공용_제품감지_유 AND S362_M_공정_AX_일반루프_제품감지_유 AND S362_M_공정_AX_RAIL_제품감지_유) OR (S362_M_차종6_썬루프 AND S362_M_공정_AX_공용_제품감지_유 AND S362_M_공정_AX_썬루프_제품감지_유 AND S362_M_공정_AX_RAIL_제품감지_유)) AND S362_M_차종1_AX;
(* Rung L83 *)
S362_M_공정_제품감지_무 := S362_M_공정_AX_공용_제품감지_무 AND S362_M_공정_AX_일반루프_제품감지_무 AND S362_M_공정_AX_썬루프_제품감지_무 AND S362_M_공정_AX_RAIL_제품감지_무;
(* S362 AX 공용 제품감지 유 *)
(* Rung L85 *)
S362_M_공정_AX_공용_제품감지_유 := S362_PRS_AX_COM_RH_CHECK AND S362_PRS_AX_COM_LH_CHECK;
(* S362 AX 일반루프 제품감지 유 *)
(* Rung L87 *)
S362_M_공정_AX_일반루프_제품감지_유 := S362_PRS_AX_GR_RH_CHECK AND S362_PRS_AX_GR_LH_CHECK;

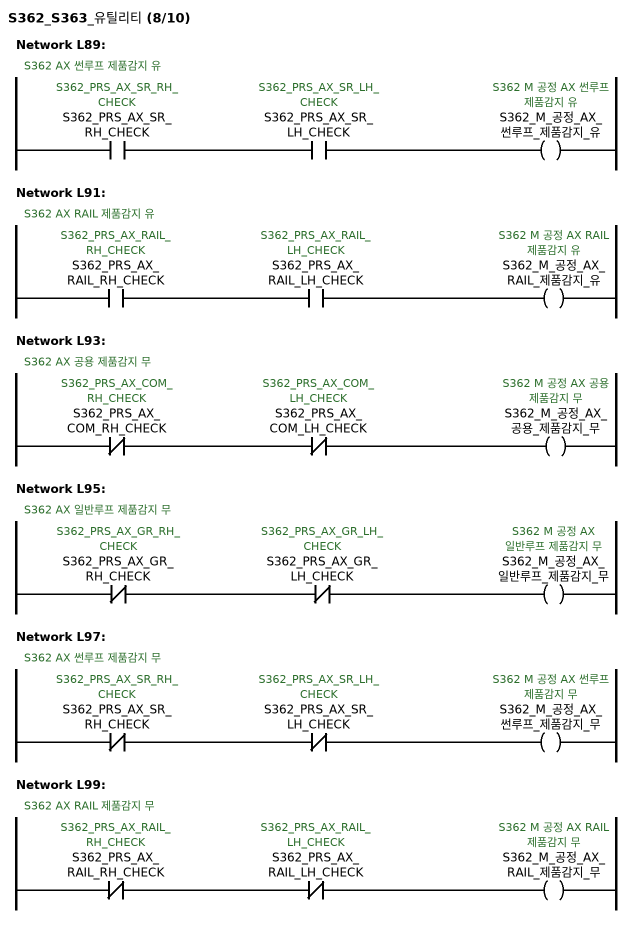
(* S362 AX 썬루프 제품감지 유 *)
(* Rung L89 *)
S362_M_공정_AX_썬루프_제품감지_유 := S362_PRS_AX_SR_RH_CHECK AND S362_PRS_AX_SR_LH_CHECK;
(* S362 AX RAIL 제품감지 유 *)
(* Rung L91 *)
S362_M_공정_AX_RAIL_제품감지_유 := S362_PRS_AX_RAIL_RH_CHECK AND S362_PRS_AX_RAIL_LH_CHECK;
(* S362 AX 공용 제품감지 무 *)
(* Rung L93 *)
S362_M_공정_AX_공용_제품감지_무 := NOT S362_PRS_AX_COM_RH_CHECK AND NOT S362_PRS_AX_COM_LH_CHECK;
(* S362 AX 일반루프 제품감지 무 *)
(* Rung L95 *)
S362_M_공정_AX_일반루프_제품감지_무 := NOT S362_PRS_AX_GR_RH_CHECK AND NOT S362_PRS_AX_GR_LH_CHECK;
(* S362 AX 썬루프 제품감지 무 *)
(* Rung L97 *)
S362_M_공정_AX_썬루프_제품감지_무 := NOT S362_PRS_AX_SR_RH_CHECK AND NOT S362_PRS_AX_SR_LH_CHECK;
(* S362 AX RAIL 제품감지 무 *)
(* Rung L99 *)
S362_M_공정_AX_RAIL_제품감지_무 := NOT S362_PRS_AX_RAIL_RH_CHECK AND NOT S362_PRS_AX_RAIL_LH_CHECK;

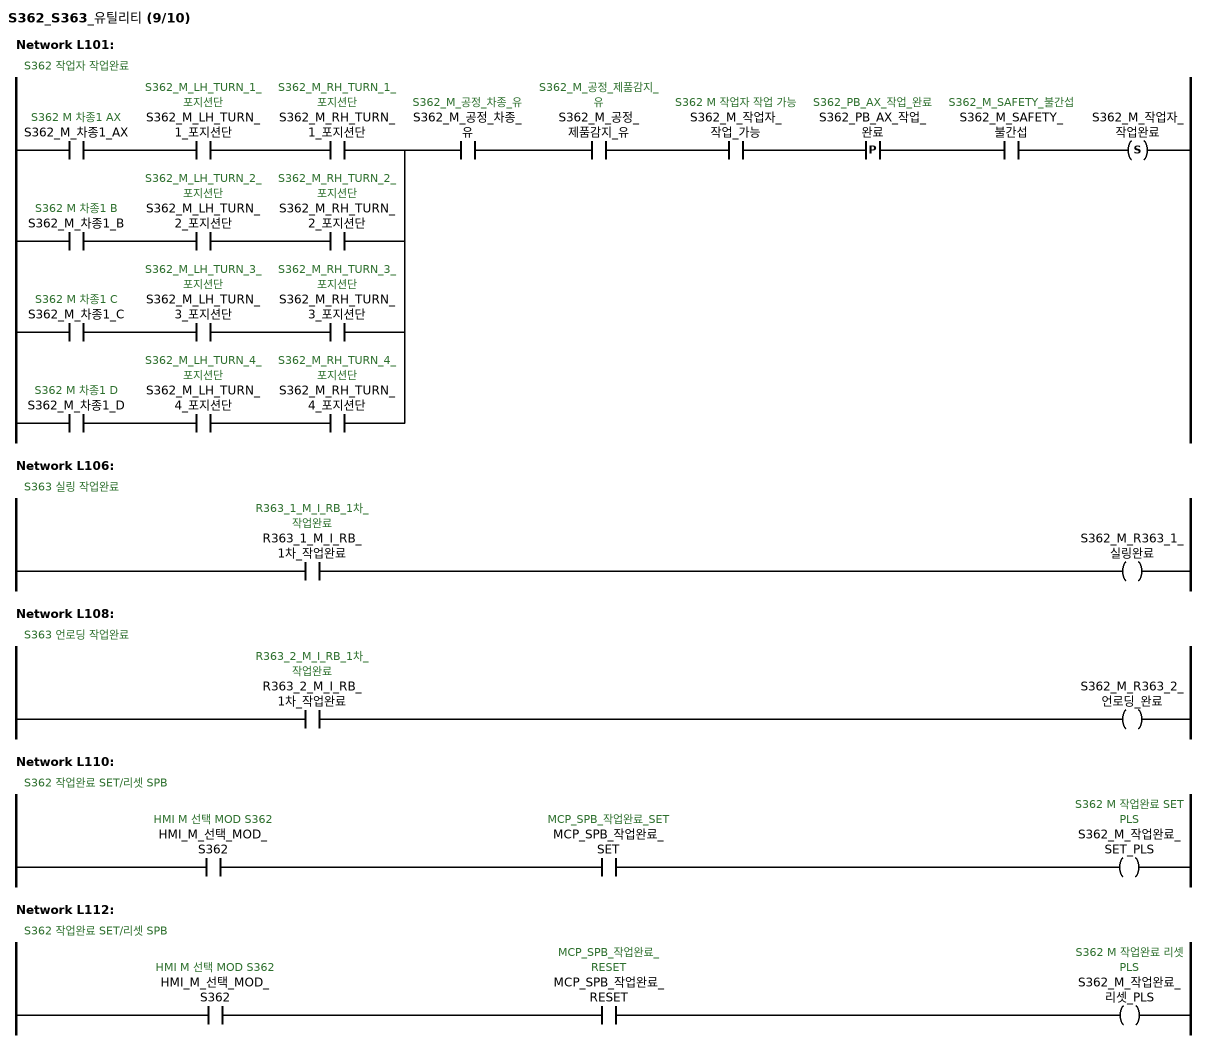
(* S362 작업자 작업완료 *)
(* Rung L101 *)
_e3(CLK := S362_PB_AX_작업_완료);
IF ((S362_M_차종1_AX AND S362_M_LH_TURN_1_포지션단 AND S362_M_RH_TURN_1_포지션단) OR (S362_M_차종1_B AND S362_M_LH_TURN_2_포지션단 AND S362_M_RH_TURN_2_포지션단) OR (S362_M_차종1_C AND S362_M_LH_TURN_3_포지션단 AND S362_M_RH_TURN_3_포지션단) OR (S362_M_차종1_D AND S362_M_LH_TURN_4_포지션단 AND S362_M_RH_TURN_4_포지션단)) AND S362_M_공정_차종_유 AND S362_M_공정_제품감지_유 AND S362_M_작업자_작업_가능 AND _e3.Q AND S362_M_SAFETY_불간섭 THEN
    S362_M_작업자_작업완료 := TRUE;
END_IF;
(* S363 실링 작업완료 *)
(* Rung L106 *)
S362_M_R363_1_실링완료 := R363_1_M_I_RB_1차_작업완료;
(* S363 언로딩 작업완료 *)
(* Rung L108 *)
S362_M_R363_2_언로딩_완료 := R363_2_M_I_RB_1차_작업완료;
(* S362 작업완료 SET/리셋 SPB *)
(* Rung L110 *)
S362_M_작업완료_SET_PLS := HMI_M_선택_MOD_S362 AND MCP_SPB_작업완료_SET;
(* S362 작업완료 SET/리셋 SPB *)
(* Rung L112 *)
S362_M_작업완료_리셋_PLS := HMI_M_선택_MOD_S362 AND MCP_SPB_작업완료_RESET;

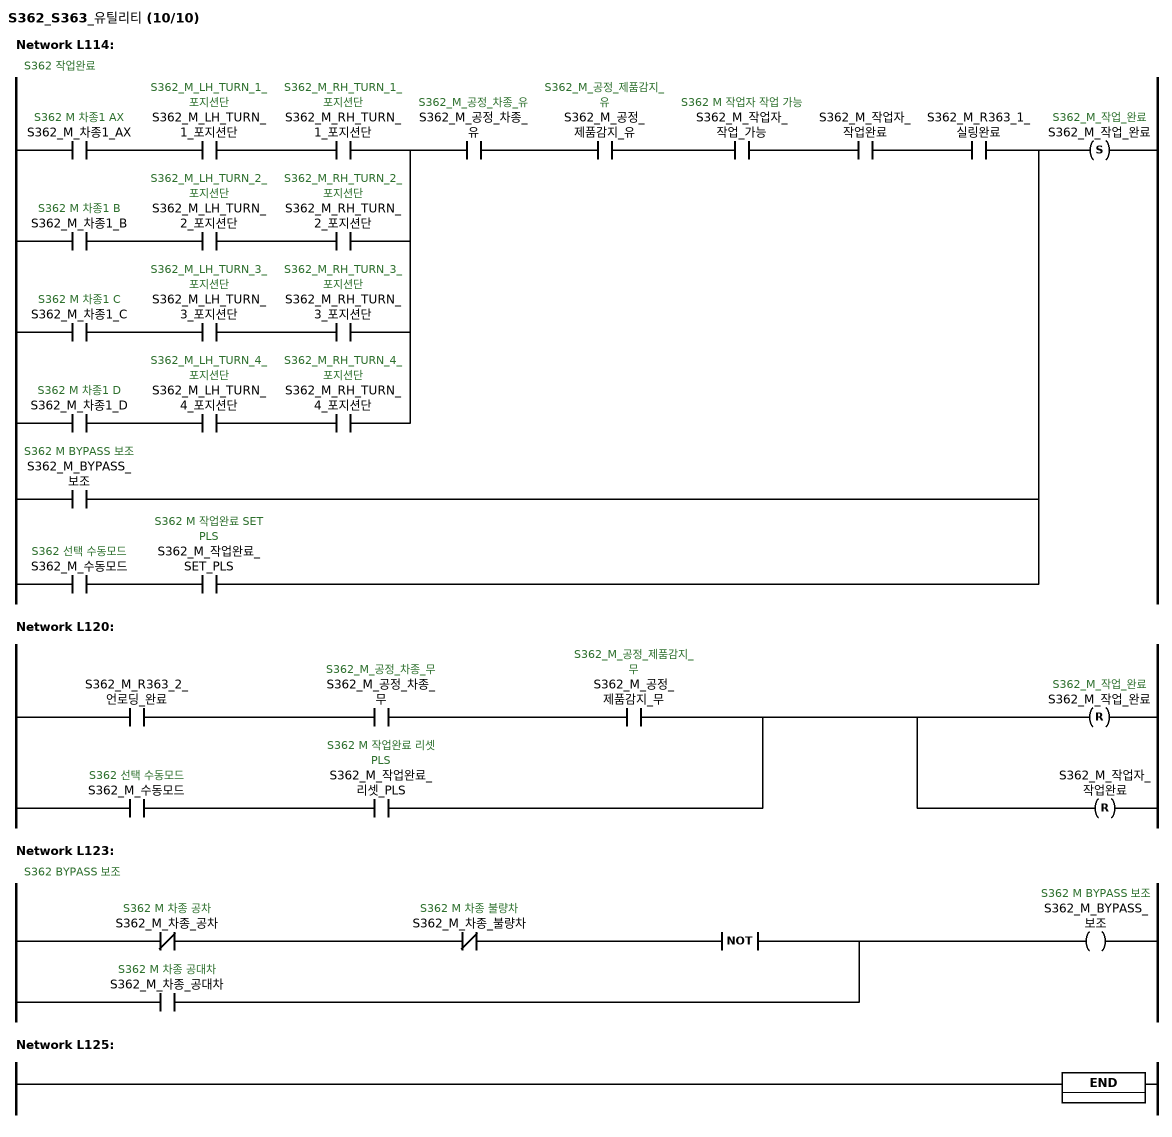
(* S362 작업완료 *)
(* Rung L114 *)
IF (((S362_M_차종1_AX AND S362_M_LH_TURN_1_포지션단 AND S362_M_RH_TURN_1_포지션단) OR (S362_M_차종1_B AND S362_M_LH_TURN_2_포지션단 AND S362_M_RH_TURN_2_포지션단) OR (S362_M_차종1_C AND S362_M_LH_TURN_3_포지션단 AND S362_M_RH_TURN_3_포지션단) OR (S362_M_차종1_D AND S362_M_LH_TURN_4_포지션단 AND S362_M_RH_TURN_4_포지션단)) AND S362_M_공정_차종_유 AND S362_M_공정_제품감지_유 AND S362_M_작업자_작업_가능 AND S362_M_작업자_작업완료 AND S362_M_R363_1_실링완료) OR S362_M_BYPASS_보조 OR (S362_M_수동모드 AND S362_M_작업완료_SET_PLS) THEN
    S362_M_작업_완료 := TRUE;
END_IF;
(* Rung L120 *)
_p4 := (S362_M_R363_2_언로딩_완료 AND S362_M_공정_차종_무 AND S362_M_공정_제품감지_무) OR (S362_M_수동모드 AND S362_M_작업완료_리셋_PLS);
IF _p4 THEN
    S362_M_작업_완료 := FALSE;
    S362_M_작업자_작업완료 := FALSE;
END_IF;
(* S362 BYPASS 보조 *)
(* Rung L123 *)
S362_M_BYPASS_보조 := NOT (NOT S362_M_차종_공차 AND NOT S362_M_차종_불량차) OR S362_M_차종_공대차;
(* Rung L125 *)
END();
END_PROGRAM

PROGRAM S362_S363_동작 (* task: 스캔 프로그램 *)
VAR_EXTERNAL RETAIN
    ALWAYS_OFF : BOOL; (* AT %MW3.0 *) (* 항시 OFF *)
    ALWAYS_ON : BOOL; (* AT %MW3.1 *) (* 항시 ON *)
    S362_HOME : BOOL; (* AT %MW1048.0 *) (* S362_HOME *)
    S362_M_LH_STEP_MOVE_리셋_PLS : BOOL; (* AT %MW1104.14 *) (* S362_M_LH_STEP_MOVE_리셋_PLS *)
    S362_M_LH_TURN_1_포지션단 : BOOL; (* AT %MW1104.3 *) (* S362_M_LH_TURN_1_포지션단 *)
    S362_M_LH_TURN_2_포지션단 : BOOL; (* AT %MW1104.4 *) (* S362_M_LH_TURN_2_포지션단 *)
    S362_M_LH_TURN_3_포지션단 : BOOL; (* AT %MW1104.5 *) (* S362_M_LH_TURN_3_포지션단 *)
    S362_M_LH_TURN_4_포지션단 : BOOL; (* AT %MW1104.6 *) (* S362_M_LH_TURN_4_포지션단 *)
    S362_M_LH_TURN_MOVE_완료 : BOOL; (* AT %MW1104.8 *) (* S362_M_LH_TURN_MOVE_완료 *)
    S362_M_LH_TURN_수동_STEP_전진_보조 : BOOL; (* AT %MW1104.11 *) (* S362_M_LH_TURN_수동_STEP_전진_보조 *)
    S362_M_LH_TURN_수동_STEP_후진_보조 : BOOL; (* AT %MW1104.12 *) (* S362_M_LH_TURN_수동_STEP_후진_보조 *)
    S362_M_LH_TURN_수동_전진_보조 : BOOL; (* AT %MW1104.9 *) (* S362_M_LH_TURN_수동_전진_보조 *)
    S362_M_LH_TURN_수동_후진_보조 : BOOL; (* AT %MW1104.10 *) (* S362_M_LH_TURN_수동_후진_보조 *)
    S362_M_LH_TURN_전진_보조 : BOOL; (* AT %MW1104.1 *) (* S362_M_LH_TURN_전진_보조 *)
    S362_M_LH_TURN_조건 : BOOL; (* AT %MW1104.0 *) (* S362_M_LH_TURN_조건 *)
    S362_M_LH_TURN_후진_보조 : BOOL; (* AT %MW1104.2 *) (* S362_M_LH_TURN_후진_보조 *)
    S362_M_LH_자동_MOVE_리셋_PLS : BOOL; (* AT %MW1104.13 *) (* S362_M_LH_자동_MOVE_리셋_PLS *)
    S362_M_RH_STEP_MOVE_리셋_PLS : BOOL; (* AT %MW1112.14 *) (* S362_M_RH_STEP_MOVE_리셋_PLS *)
    S362_M_RH_TURN_1_포지션단 : BOOL; (* AT %MW1112.3 *) (* S362_M_RH_TURN_1_포지션단 *)
    S362_M_RH_TURN_2_포지션단 : BOOL; (* AT %MW1112.4 *) (* S362_M_RH_TURN_2_포지션단 *)
    S362_M_RH_TURN_3_포지션단 : BOOL; (* AT %MW1112.5 *) (* S362_M_RH_TURN_3_포지션단 *)
    S362_M_RH_TURN_4_포지션단 : BOOL; (* AT %MW1112.6 *) (* S362_M_RH_TURN_4_포지션단 *)
    S362_M_RH_TURN_MOVE_완료 : BOOL; (* AT %MW1112.8 *) (* S362_M_RH_TURN_MOVE_완료 *)
    S362_M_RH_TURN_수동_STEP_전진_보조 : BOOL; (* AT %MW1112.11 *) (* S362_M_RH_TURN_수동_STEP_전진_보조 *)
    S362_M_RH_TURN_수동_STEP_후진_보조 : BOOL; (* AT %MW1112.12 *) (* S362_M_RH_TURN_수동_STEP_후진_보조 *)
    S362_M_RH_TURN_수동_전진_보조 : BOOL; (* AT %MW1112.9 *) (* S362_M_RH_TURN_수동_전진_보조 *)
    S362_M_RH_TURN_수동_후진_보조 : BOOL; (* AT %MW1112.10 *) (* S362_M_RH_TURN_수동_후진_보조 *)
    S362_M_RH_TURN_전진_보조 : BOOL; (* AT %MW1112.1 *) (* S362_M_RH_TURN_전진_보조 *)
    S362_M_RH_TURN_조건 : BOOL; (* AT %MW1112.0 *) (* S362_M_RH_TURN_조건 *)
    S362_M_RH_TURN_후진_보조 : BOOL; (* AT %MW1112.2 *) (* S362_M_RH_TURN_후진_보조 *)
    S362_M_RH_자동_MOVE_리셋_PLS : BOOL; (* AT %MW1112.13 *) (* S362_M_RH_자동_MOVE_리셋_PLS *)
    S362_M_SAFETY_불간섭 : BOOL; (* AT %MW1004.4 *) (* S362_M_SAFETY_불간섭 *)
    S362_M_SLD_LOCK_전진_LS_이상 : BOOL; (* AT %MW1102.5 *) (* S362_M_SLD_LOCK_전진_LS_이상 *)
    S362_M_SLD_LOCK_전진_보조 : BOOL; (* AT %MW1102.1 *) (* S362_M_SLD_LOCK_전진_보조 *)
    S362_M_SLD_LOCK_전진단 : BOOL; (* AT %MW1102.3 *) (* S362_M_SLD_LOCK_전진단 *)
    S362_M_SLD_LOCK_조건 : BOOL; (* AT %MW1102.0 *) (* S362_M_SLD_LOCK_조건 *)
    S362_M_SLD_LOCK_후진_LS_이상 : BOOL; (* AT %MW1102.6 *) (* S362_M_SLD_LOCK_후진_LS_이상 *)
    S362_M_SLD_LOCK_후진_보조 : BOOL; (* AT %MW1102.2 *) (* S362_M_SLD_LOCK_후진_보조 *)
    S362_M_SLD_LOCK_후진단 : BOOL; (* AT %MW1102.4 *) (* S362_M_SLD_LOCK_후진단 *)
    S362_M_SLIDE_전진_LS_이상 : BOOL; (* AT %MW1101.5 *) (* S362_M_SLIDE_전진_LS_이상 *)
    S362_M_SLIDE_전진_보조 : BOOL; (* AT %MW1101.1 *) (* S362_M_SLIDE_전진_보조 *)
    S362_M_SLIDE_전진단 : BOOL; (* AT %MW1101.3 *) (* S362_M_SLIDE_전진단 *)
    S362_M_SLIDE_조건 : BOOL; (* AT %MW1101.0 *) (* S362_M_SLIDE_조건 *)
    S362_M_SLIDE_후진_LS_이상 : BOOL; (* AT %MW1101.6 *) (* S362_M_SLIDE_후진_LS_이상 *)
    S362_M_SLIDE_후진_보조 : BOOL; (* AT %MW1101.2 *) (* S362_M_SLIDE_후진_보조 *)
    S362_M_SLIDE_후진단 : BOOL; (* AT %MW1101.4 *) (* S362_M_SLIDE_후진단 *)
    S362_M_TURN_LOCK_전진_LS_이상 : BOOL; (* AT %MW1100.5 *) (* S362_M_TURN_LOCK_전진_LS_이상 *)
    S362_M_TURN_LOCK_전진_보조 : BOOL; (* AT %MW1100.1 *) (* S362_M_TURN_LOCK_전진_보조 *)
    S362_M_TURN_LOCK_전진단 : BOOL; (* AT %MW1100.3 *) (* S362_M_TURN_LOCK_전진단 *)
    S362_M_TURN_LOCK_조건 : BOOL; (* AT %MW1100.0 *) (* S362_M_TURN_LOCK_조건 *)
    S362_M_TURN_LOCK_후진_LS_이상 : BOOL; (* AT %MW1100.6 *) (* S362_M_TURN_LOCK_후진_LS_이상 *)
    S362_M_TURN_LOCK_후진_보조 : BOOL; (* AT %MW1100.2 *) (* S362_M_TURN_LOCK_후진_보조 *)
    S362_M_TURN_LOCK_후진단 : BOOL; (* AT %MW1100.4 *) (* S362_M_TURN_LOCK_후진단 *)
    S362_M_공정_불간섭 : BOOL; (* AT %MW1004.1 *) (* S362_M_공정_불간섭 *)
    S362_M_공정_제품감지_무 : BOOL; (* AT %MW1001.5 *) (* S362_M_공정_제품감지_무 *)
    S362_M_공정_제품감지_유 : BOOL; (* AT %MW1001.4 *) (* S362_M_공정_제품감지_유 *)
    S362_M_공정_차종_무 : BOOL; (* AT %MW1002.1 *) (* S362_M_공정_차종_무 *)
    S362_M_공정_차종_유 : BOOL; (* AT %MW1002.0 *) (* S362_M_공정_차종_유 *)
    S362_M_동작_선택_1 : BOOL; (* AT %MW1040.0 *) (* S362_M_동작_선택_1 *)
    S362_M_동작_선택_13 : BOOL; (* AT %MW1040.12 *) (* S362_M_동작_선택_13 *)
    S362_M_동작_선택_14 : BOOL; (* AT %MW1040.13 *) (* S362_M_동작_선택_14 *)
    S362_M_동작_선택_15 : BOOL; (* AT %MW1040.14 *) (* S362_M_동작_선택_15 *)
    S362_M_동작_선택_16 : BOOL; (* AT %MW1040.15 *) (* S362_M_동작_선택_16 *)
    S362_M_동작_선택_2 : BOOL; (* AT %MW1040.1 *) (* S362_M_동작_선택_2 *)
    S362_M_동작_선택_3 : BOOL; (* AT %MW1040.2 *) (* S362_M_동작_선택_3 *)
    S362_M_동작_선택_5 : BOOL; (* AT %MW1040.4 *) (* S362_M_동작_선택_5 *)
    S362_M_동작_선택_6 : BOOL; (* AT %MW1040.5 *) (* S362_M_동작_선택_6 *)
    S362_M_동작_선택_7 : BOOL; (* AT %MW1040.6 *) (* S362_M_동작_선택_7 *)
    S362_M_동작_선택_8 : BOOL; (* AT %MW1040.7 *) (* S362_M_동작_선택_8 *)
    S362_M_수동모드 : BOOL; (* AT %MW1000.3 *) (* S362 선택 수동모드 *)
    S362_M_운전준비_ON : BOOL; (* AT %MW1000.0 *) (* S362 운전준비 ON *)
    S362_M_자동_운전중 : BOOL; (* AT %MW1000.4 *) (* S362 자동운전중 *)
    S362_M_작업_완료 : BOOL; (* AT %MW1001.0 *) (* S362_M_작업_완료 *)
    S362_M_작업자_작업완료 : BOOL; (* AT %MW1001.1 *)
    S362_M_차종1_AX : BOOL; (* AT %MW10101.0 *) (* S362 M 차종1 AX *)
    S362_M_차종1_B : BOOL; (* AT %MW10101.1 *) (* S362 M 차종1 B *)
    S362_M_차종1_C : BOOL; (* AT %MW10101.2 *) (* S362 M 차종1 C *)
    S362_M_차종1_D : BOOL; (* AT %MW10101.3 *) (* S362 M 차종1 D *)
    S362_전진_ON : BOOL; (* AT %MW1048.1 *) (* S362_전진_ON *)
    S362_후진_ON : BOOL; (* AT %MW1048.2 *) (* S362_후진_ON *)
    전체_M_이상_리셋 : BOOL; (* AT %MW308.2 *) (* ALL공정 PB 이상리셋 *)
END_VAR
VAR_EXTERNAL
    EGIS_CWS : BOOL;
    S362_6_INV1_BRAKE_CR_ON : BOOL; (* AT %MW95014.7 *) (* S362_6_INV1_BRAKE_CR_ON *)
    S362_6_INV1_RETURN : BOOL; (* AT %MW95014.1 *) (* S362_6_INV1_RETURN *)
    S362_6_INV1_TURN : BOOL; (* AT %MW95014.0 *) (* S362_6_INV1_TURN *)
    S362_6_INV2_BRAKE_CR_ON : BOOL; (* AT %MW95014.15 *) (* S362_6_INV2_BRAKE_CR_ON *)
    S362_6_INV2_RETURN : BOOL; (* AT %MW95014.9 *) (* S362_6_INV2_RETURN *)
    S362_6_INV2_TURN : BOOL; (* AT %MW95014.8 *) (* S362_6_INV2_TURN *)
    S362_INDEX_LH_TURN_감지1 : BOOL; (* AT %MW87102.4 *) (* S362_INDEX_LH_TURN_감지1 *)
    S362_INDEX_LH_TURN_감지2 : BOOL; (* AT %MW87102.5 *) (* S362_INDEX_LH_TURN_감지2 *)
    S362_INDEX_LH_TURN_감지3 : BOOL; (* AT %MW87102.6 *) (* S362_INDEX_LH_TURN_감지3 *)
    S362_INDEX_LH_TURN_원점 : BOOL; (* AT %MW87102.7 *) (* S362_INDEX_LH_TURN_원점 *)
    S362_INDEX_RH_TURN_감지1 : BOOL; (* AT %MW87102.0 *) (* S362_INDEX_RH_TURN_감지1 *)
    S362_INDEX_RH_TURN_감지2 : BOOL; (* AT %MW87102.1 *) (* S362_INDEX_RH_TURN_감지2 *)
    S362_INDEX_RH_TURN_감지3 : BOOL; (* AT %MW87102.2 *) (* S362_INDEX_RH_TURN_감지3 *)
    S362_INDEX_RH_TURN_원점 : BOOL; (* AT %MW87102.3 *) (* S362_INDEX_RH_TURN_원점 *)
    S362_LS_AX_SLIDE_전진 : BOOL; (* AT %MW87100.8 *) (* S362_LS_AX_SLIDE_전진 *)
    S362_LS_AX_SLIDE_후진 : BOOL; (* AT %MW87100.9 *) (* S362_LS_AX_SLIDE_후진 *)
    S362_M_SLD_LOCK_전진_LAMP : WORD; (* AT %MW11104 *) (* S362_M_SLD_LOCK_전진_LAMP *)
    S362_M_SLD_LOCK_후진_LAMP : WORD; (* AT %MW11105 *) (* S362_M_SLD_LOCK_후진_LAMP *)
    S362_M_SLIDE_전진_LAMP : WORD; (* AT %MW11102 *) (* S362_M_SLIDE_전진_LAMP *)
    S362_M_SLIDE_후진_LAMP : WORD; (* AT %MW11103 *) (* S362_M_SLIDE_후진_LAMP *)
    S362_M_TURN_LOCK_전진_LAMP : WORD; (* AT %MW11100 *) (* S362_M_TURN_LOCK_전진_LAMP *)
    S362_M_TURN_LOCK_후진_LAMP : WORD; (* AT %MW11101 *) (* S362_M_TURN_LOCK_후진_LAMP *)
    S362_RS_FRT_SLD_LOCK_전진 : BOOL; (* AT %MW87100.4 *) (* S362_RS_FRT_SLD_LOCK_전진 *)
    S362_RS_FRT_SLD_LOCK_후진 : BOOL; (* AT %MW87100.5 *) (* S362_RS_FRT_SLD_LOCK_후진 *)
    S362_RS_LH_IDX_LOCK_전진 : BOOL; (* AT %MW87100.2 *) (* S362_RS_LH_IDX_LOCK_전진 *)
    S362_RS_LH_IDX_LOCK_후진 : BOOL; (* AT %MW87100.3 *) (* S362_RS_LH_IDX_LOCK_후진 *)
    S362_RS_RH_IDX_LOCK_전진 : BOOL; (* AT %MW87100.0 *) (* S362_RS_RH_IDX_LOCK_전진 *)
    S362_RS_RH_IDX_LOCK_후진 : BOOL; (* AT %MW87100.1 *) (* S362_RS_RH_IDX_LOCK_후진 *)
    S362_RS_RR_SLD_LOCK_전진 : BOOL; (* AT %MW87100.6 *) (* S362_RS_RR_SLD_LOCK_전진 *)
    S362_RS_RR_SLD_LOCK_후진 : BOOL; (* AT %MW87100.7 *) (* S362_RS_RR_SLD_LOCK_후진 *)
    S362_SOL_AX_BRAKE_ON : BOOL; (* AT %MW97103.6 *) (* S362_SOL_AX_BRAKE_ON *)
    S362_SOL_AX_SLIDE_전진 : BOOL; (* AT %MW97103.4 *) (* S362_SOL_AX_SLIDE_전진 *)
    S362_SOL_AX_SLIDE_후진 : BOOL; (* AT %MW97103.5 *) (* S362_SOL_AX_SLIDE_후진 *)
    S362_SOL_AX_SLI_LOCK_전진 : BOOL; (* AT %MW97103.2 *) (* S362_SOL_AX_SLI_LOCK_전진 *)
    S362_SOL_AX_SLI_LOCK_후진 : BOOL; (* AT %MW97103.3 *) (* S362_SOL_AX_SLI_LOCK_후진 *)
    S362_SOL_TURN_LOCK_전진 : BOOL; (* AT %MW97103.0 *) (* S362_SOL_TURN_LOCK_전진 *)
    S362_SOL_TURN_LOCK_후진 : BOOL; (* AT %MW97103.1 *) (* S362_SOL_TURN_LOCK_후진 *)
END_VAR
VAR
    S362_SLIDE : ACT_6_CYL;
    S362_SLIDE_LOCK : ACT_6_CYL;
    S362_TURN_LOCK : ACT_6_CYL;
    T362_LH_TURN_POSI_1 : TON;
    T362_LH_TURN_POSI_2 : TON;
    T362_LH_TURN_POSI_3 : TON;
    T362_LH_TURN_POSI_4 : TON;
    T362_RH_TURN_POSI_17 : TON;
    T362_RH_TURN_POSI_18 : TON;
    T362_RH_TURN_POSI_19 : TON;
    T362_RH_TURN_POSI_20 : TON;
END_VAR

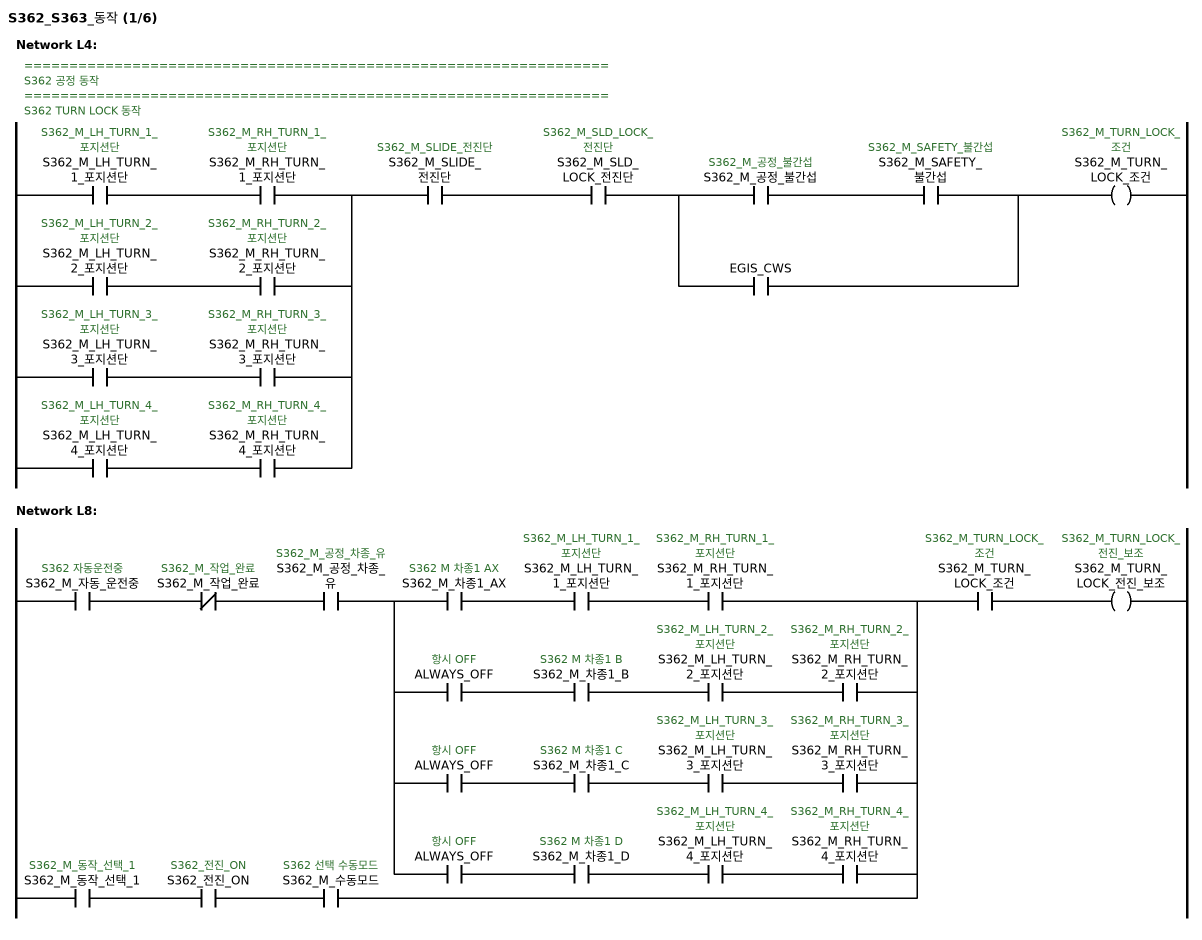
(* ================================================================= *)
(* S362 공정 동작 *)
(* ================================================================= *)
(* S362 TURN LOCK 동작 *)
(* Rung L4 *)
S362_M_TURN_LOCK_조건 := ((S362_M_LH_TURN_1_포지션단 AND S362_M_RH_TURN_1_포지션단) OR (S362_M_LH_TURN_2_포지션단 AND S362_M_RH_TURN_2_포지션단) OR (S362_M_LH_TURN_3_포지션단 AND S362_M_RH_TURN_3_포지션단) OR (S362_M_LH_TURN_4_포지션단 AND S362_M_RH_TURN_4_포지션단)) AND S362_M_SLIDE_전진단 AND S362_M_SLD_LOCK_전진단 AND ((S362_M_공정_불간섭 AND S362_M_SAFETY_불간섭) OR EGIS_CWS);
(* Rung L8 *)
S362_M_TURN_LOCK_전진_보조 := ((S362_M_자동_운전중 AND NOT S362_M_작업_완료 AND S362_M_공정_차종_유 AND ((S362_M_차종1_AX AND S362_M_LH_TURN_1_포지션단 AND S362_M_RH_TURN_1_포지션단) OR (ALWAYS_OFF AND S362_M_차종1_B AND S362_M_LH_TURN_2_포지션단 AND S362_M_RH_TURN_2_포지션단) OR (ALWAYS_OFF AND S362_M_차종1_C AND S362_M_LH_TURN_3_포지션단 AND S362_M_RH_TURN_3_포지션단) OR (ALWAYS_OFF AND S362_M_차종1_D AND S362_M_LH_TURN_4_포지션단 AND S362_M_RH_TURN_4_포지션단))) OR (S362_M_동작_선택_1 AND S362_전진_ON AND S362_M_수동모드)) AND S362_M_TURN_LOCK_조건;

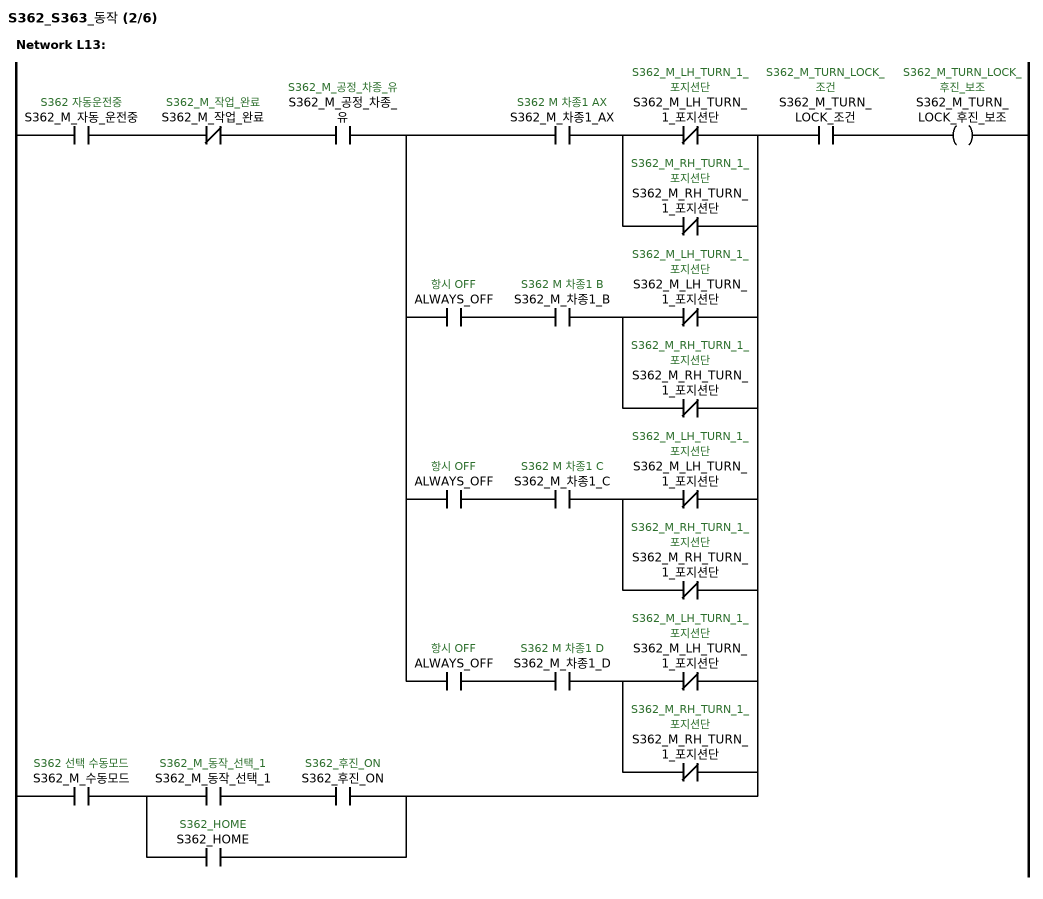
(* Rung L13 *)
S362_M_TURN_LOCK_후진_보조 := ((S362_M_자동_운전중 AND NOT S362_M_작업_완료 AND S362_M_공정_차종_유 AND ((S362_M_차종1_AX AND (NOT S362_M_LH_TURN_1_포지션단 OR NOT S362_M_RH_TURN_1_포지션단)) OR (ALWAYS_OFF AND S362_M_차종1_B AND (NOT S362_M_LH_TURN_1_포지션단 OR NOT S362_M_RH_TURN_1_포지션단)) OR (ALWAYS_OFF AND S362_M_차종1_C AND (NOT S362_M_LH_TURN_1_포지션단 OR NOT S362_M_RH_TURN_1_포지션단)) OR (ALWAYS_OFF AND S362_M_차종1_D AND (NOT S362_M_LH_TURN_1_포지션단 OR NOT S362_M_RH_TURN_1_포지션단)))) OR (S362_M_수동모드 AND ((S362_M_동작_선택_1 AND S362_후진_ON) OR S362_HOME))) AND S362_M_TURN_LOCK_조건;

